(* IEC 61131-3 sources: SIMERLIFT/LOGICAD/SIMERLIFT/src_FBD/BCU/fbdBCU_bess, 5 files *)

(* ---- Balance_isz.iecfbd ---- *)
FUNCTION_BLOCK Balance_isz
  {
    Charge_Status {index := 0};
    Avarage_Cell_Voltage {index := 3};
    Balance_Threshold {index := 4};
    Difference_Tolerance {index := 5};
    Ballance_Interval {index := 6};
    Min_Cell_Voltage {index := 2};
    Max_Cell_Voltage {index := 1};
    Measure_Aux {index := 3};
    Measure_All {index := 2};
    width := 460;
    height := 138;
  }

  VAR
    RS3 : RS;
    TP3 : TP;
    TON4 : TON;
    R_TRIG5 : R_TRIG;
    Meas_Period : TIME := T#48ms;
    Ballance_Pending : BOOL := 0;
    maxVolt : UDINT;
    minVolt : UDINT;
    FLASH1 : FLASH;
    FLASH2 : FLASH;
  END_VAR
  VAR_INPUT
    Max_Cell_Voltage : UDINT := 0;
    Min_Cell_Voltage : UDINT := 0;
    Avarage_Cell_Voltage : UDINT := 0;
    Charge_Status : BOOL := 0;
    Ballance_Interval : TIME := T#30s;
    Difference_Tolerance : UDINT := 0;
    Balance_Threshold : UDINT := 0;
  END_VAR
  VAR_OUTPUT
    Balance_Enable : BOOL := 0;
    Measure_All : BOOL := 0;
    Measure_Aux : BOOL := 0;
    Ballance_Voltage : UDINT := 0;
  END_VAR

  (*

    // Network 1:
    ADD(IN1 := Avarage_Cell_Voltage, IN2 := 1, ADD => @C(4).ADD);
    GE(IN1 := @C(4).ADD, IN2 := Balance_Threshold, GE => @C(29).GE);
    SEL(G := @C(29).GE, IN0 := Balance_Threshold, IN1 := @C(4).ADD, SEL => Ballance_Voltage);

    // Network 2:
    GE(IN1 := Max_Cell_Voltage, IN2 := Balance_Threshold, GE => @C(41).GE);
    SUB(IN1 := Max_Cell_Voltage, IN2 := Min_Cell_Voltage, SUB => @C(20).SUB);
    GT(IN1 := @C(20).SUB, IN2 := Difference_Tolerance, GT => @C(45).GT);
    AND(IN1 := @C(41).GE, IN2 := @C(45).GT, AND => Ballance_Pending);

    // Network 3:
    MUL_TIME(IN1 := Meas_Period, IN2 := 20, MUL_TIME => @C(50).MUL_TIME);
    ADD(IN1 := @C(50).MUL_TIME, IN2 := Ballance_Interval, ADD => @C(54).ADD);
    TP3(IN := RS3.Q1, PT := Ballance_Interval);
    AND(IN1 := Charge_Status, IN2 := TP3.Q, AND => (@C(11).AND, Balance_Enable));
    FLASH1(IN := NOT @C(11).AND, PER := Meas_Period, OUT => Measure_All);
    TON4(IN := RS3.Q1, PT := @C(54).ADD);
    R_TRIG5(CLK := TON4.Q);
    RS3(S := Ballance_Pending, R1 := R_TRIG5.Q);
    FLASH2(IN := @C(11).AND, PER := T#1s, OUT => Measure_Aux);

  *)

  @C(4) : @F(ADD), @R(280.0, 20.0, 40.0, 38.0), UDINT, @I(@N(IN1), @L(9.5)), @I(@N(IN2), @L(29.5)), @O(@N(ADD), @R(9.5));
  @C(8) : @F(AND), @R(520.0, 120.0, 40.0, 38.0), BOOL, @I(@N(IN1), @L(9.5)), @I(@N(IN2), @L(29.5)), @O(@N(AND), @R(9.5));
  @C(11) : @F(AND), @R(1140.0, 250.0, 40.0, 38.0), BOOL, @I(@N(IN1), @L(9.5)), @I(@N(IN2), @L(29.5)), @O(@N(AND), @R(9.5));
  @C(20) : @F(SUB), @R(280.0, 160.0, 40.0, 38.0), UDINT, @I(@N(IN1), @L(9.5)), @I(@N(IN2), @L(29.5)), @O(@N(SUB), @R(9.5));
  @C(25) : @FB(RS3), @R(800.0, 290.0, 80.0, 38.0), @I(@N(S), @L(9.5)), @I(@N(R1), @L(29.5)), @O(@N(Q1), @R(9.5));
  @C(24) : @FB(TP3), @R(960.0, 290.0, 100.0, 38.0), @I(@N(IN), @L(9.5)), @I(@N(PT), @L(29.5)), @O(@N(Q), @R(9.5)), @O(@N(ET), @R(29.5));
  @C(27) : @FB(TON4), @R(480.0, 310.0, 100.0, 38.0), @I(@N(IN), @L(9.5)), @I(@N(PT), @L(29.5)), @O(@N(Q), @R(9.5)), @O(@N(ET), @R(29.5));
  @C(26) : @FB(R_TRIG5), @R(620.0, 310.0, 140.0, 18.0), @I(@N(CLK), @L(9.5)), @O(@N(Q), @R(9.5));
  @C(29) : @F(GE), @R(440.0, 20.0, 40.0, 38.0), UDINT, @I(@N(IN1), @L(9.5)), @I(@N(IN2), @L(29.5)), @O(@N(GE), @R(9.5));
  @C(33) : @F(SEL), @R(560.0, 40.0, 120.0, 58.0), UDINT, @I(@N(G), @L(9.5)), @I(@N(IN0), @L(29.5)), @I(@N(IN1), @L(49.5)), @O(@N(SEL), @R(9.5));
  @C(41) : @F(GE), @R(400.0, 120.0, 40.0, 38.0), UDINT, @I(@N(IN1), @L(9.5)), @I(@N(IN2), @L(29.5)), @O(@N(GE), @R(9.5));
  @C(45) : @F(GT), @R(400.0, 160.0, 40.0, 38.0), UDINT, @I(@N(IN1), @L(9.5)), @I(@N(IN2), @L(29.5)), @O(@N(GT), @R(9.5));
  @C(50) : @F(MUL_TIME), @R(280.0, 330.0, 40.0, 38.0), USINT, @I(@N(IN1), @L(9.5)), @I(@N(IN2), @L(29.5)), @O(@N(MUL_TIME), @R(9.5));
  @C(54) : @F(ADD), @R(400.0, 330.0, 40.0, 38.0), TIME, @I(@N(IN1), @L(9.5)), @I(@N(IN2), @L(29.5)), @O(@N(ADD), @R(9.5));
  @VF(69) : @E(Meas_Period), @R(1340.0, 320.0, 110.0, 19.0);
  @VF(3) : @E(Avarage_Cell_Voltage), @R(20.0, 20.0, 180.0, 19.0);
  @VF(6) : @E(1), @R(110.0, 40.0, 90.0, 19.0), UDINT;
  @VF(7) : @E(Balance_Enable), @R(1640.0, 250.0, 180.0, 19.0);
  @VF(10) : @E(Charge_Status), @R(20.0, 250.0, 180.0, 19.0);
  @VF(78) : @E(Ballance_Interval), @R(20.0, 370.0, 180.0, 19.0);
  @VF(72) : @E(Measure_All), @R(1650.0, 300.0, 180.0, 19.0);
  @VF(18) : @E(Difference_Tolerance), @R(20.0, 200.0, 180.0, 19.0);
  @VF(31) : @E(Balance_Threshold), @R(20.0, 60.0, 180.0, 19.0);
  @VF(239) : @E(Meas_Period), @R(20.0, 330.0, 180.0, 19.0);
  @VF(37) : @E(Ballance_Voltage), @R(750.0, 40.0, 180.0, 19.0);
  @VF(42) : @E(Balance_Threshold), @R(20.0, 140.0, 180.0, 19.0);
  @VF(48) : @E(Ballance_Pending), @R(750.0, 120.0, 180.0, 19.0);
  @VF(52) : @E(20), @R(110.0, 350.0, 90.0, 19.0), USINT;
  @VF(58) : @E(Ballance_Pending), @R(20.0, 290.0, 180.0, 19.0);
  @C(23) : @FB(FLASH1), @R(1480.0, 300.0, 120.0, 38.0), @I(@N(IN), @L(9.5), @NEG), @I(@N(PER), @L(29.5)), @O(@N(OUT), @R(9.5));
  @VF(74) : @E(Max_Cell_Voltage), @R(30.0, 160.0, 160.0, 19.0);
  @VF(83) : @E(Min_Cell_Voltage), @R(30.0, 180.0, 160.0, 19.0);
  @C(14) : @FB(FLASH2), @R(1480.0, 340.0, 120.0, 38.0), @I(@N(IN), @L(9.5)), @I(@N(PER), @L(29.5)), @O(@N(OUT), @R(9.5));
  @VF(15) : @E(T#1s), @R(1340.0, 360.0, 110.0, 19.0);
  @VF(16) : @E(Measure_Aux), @R(1650.0, 340.0, 180.0, 19.0);
  @CP(35) : 399.5, 69.5;
  @CP(36) : 359.5, 29.5;
  @CP(44) : 239.5, 169.5;
  @CP(64) : 359.5, 379.5;
  @CP(66) : 919.5, 299.5;
  @CP(2) : 1289.5, 259.5;

  @G(13) :
     @L(@C(11).AND, @CP(2)),
     @L(@CP(2), @VF(7).i),
     @L(@CP(2), @C(23).IN),
     @L(@CP(2), @C(14).IN)
    ;
  @G(5) :
     @L(@VF(3).o, @C(4).IN1)
    ;
  @G(28) :
     @L(@VF(6).o, @C(4).IN2)
    ;
  @G(30) :
     @L(@C(4).ADD, @CP(36)),
     @L(@CP(36), @C(29).IN1),
     @L(@CP(36), @C(33).IN1)
    ;
  @G(32) :
     @L(@VF(31).o, @CP(35)),
     @L(@CP(35), @C(29).IN2),
     @L(@CP(35), @C(33).IN0)
    ;
  @G(34) :
     @L(@C(29).GE, @C(33).G)
    ;
  @G(38) :
     @L(@C(33).SEL, @VF(37).i)
    ;
  @G(39) :
     @L(@CP(44), @C(20).IN1),
     @L(@CP(44), @C(41).IN1),
     @L(@VF(74).o, @CP(44))
    ;
  @G(46) :
     @L(@C(20).SUB, @C(45).IN1)
    ;
  @G(19) :
     @L(@VF(18).o, @C(45).IN2)
    ;
  @G(49) :
     @L(@C(8).AND, @VF(48).i)
    ;
  @G(51) :
     @L(@VF(239).o, @C(50).IN1)
    ;
  @G(53) :
     @L(@VF(52).o, @C(50).IN2)
    ;
  @G(56) :
     @L(@CP(64), @C(54).IN2),
     @L(@CP(64), @C(24).PT),
     @L(@VF(78).o, @CP(64))
    ;
  @G(57) :
     @L(@C(50).MUL_TIME, @C(54).IN1)
    ;
  @G(59) :
     @L(@VF(58).o, @C(25).S)
    ;
  @G(60) :
     @L(@C(26).Q, @C(25).R1)
    ;
  @G(61) :
     @L(@C(54).ADD, @C(27).PT)
    ;
  @G(62) :
     @L(@C(27).Q, @C(26).CLK)
    ;
  @G(63) :
     @L(@C(25).Q1, @CP(66)),
     @L(@CP(66), @C(24).IN),
     @L(@CP(66), @C(27).IN)
    ;
  @G(65) :
     @L(@C(24).Q, @C(11).IN2)
    ;
  @G(9) :
     @L(@C(41).GE, @C(8).IN1)
    ;
  @G(21) :
     @L(@C(45).GT, @C(8).IN2)
    ;
  @G(22) :
     @L(@VF(42).o, @C(41).IN2)
    ;
  @G(12) :
     @L(@VF(10).o, @C(11).IN1)
    ;
  @G(43) :
     @L(@VF(69).o, @C(23).PER)
    ;
  @G(75) :
     @L(@C(23).OUT, @VF(72).i)
    ;
  @G(1) :
     @L(@VF(83).o, @C(20).IN2)
    ;
  @G(17) :
     @L(@VF(15).o, @C(14).PER)
    ;
  @G(40) :
     @L(@C(14).OUT, @VF(16).i)
    ;
END_FUNCTION_BLOCK

(* ---- CurrentLimiter_ISZ.iecfbd ---- *)
FUNCTION_BLOCK CurrentLimiter_ISZ
  {
    width := 370;
  }

  VAR
    OverCurrent30sec : BOOL;
    OverCurrent10sec : BOOL;
    OverCurrentCont : BOOL;
    CounTimR1 : CounTimR;
    deratingToCont : BOOL;
    maxCurrent : INT;
    RS2 : RS;
    exceed30s : BOOL;
    SR1 : SR;
    FLASH5 : FLASH;
    FLASH6 : FLASH;
    CTUD2 : CTUD;
  END_VAR
  VAR_INPUT
    Lim30s : INT;
    LimCont : INT;
    Current : INT;
  END_VAR
  VAR_OUTPUT
    overCurrent : BOOL;
    Lim : INT;
  END_VAR

  (*

    // Network 1:
    GT(IN1 := Current, IN2 := Lim30s, GT => OverCurrent30sec);
    GT(IN1 := Current, IN2 := LimCont, GT => OverCurrentCont);

    // Network 2:
    CounTimR1(CU := OverCurrentCont, ACCper := T#500ms, DECper := T#2s, CD := NOT OverCurrentCont, PV := 25, QU => exceed30s);
    GE(IN1 := CounTimR1.CV, IN2 := 30, GE => @C(18).GE);
    SR1(S1 := @C(18).GE, R := CounTimR1.QD, Q1 => deratingToCont);

    // Network 3:
    SEL(G := deratingToCont, IN0 := Lim30s, IN1 := LimCont, SEL => maxCurrent);

    // Network 4:
    RS2(S := exceed30s, R1 := NOT OverCurrentCont);
    OR(IN1 := OverCurrent30sec, IN2 := RS2.Q1, OR => OverCurrent);

    // Network 5:
    TO_INT(IN := maxCurrent, TO_INT => @C(173).TO_INT);
    GT(IN1 := maxCurrent, IN2 := Lim, GT => @C(95).GT);
    FLASH5(IN := @C(95).GT, PER := T#5ms);
    LT(IN1 := maxCurrent, IN2 := Lim, LT => @C(98).LT);
    FLASH6(IN := @C(98).LT, PER := T#5ms);
    CTUD2(CU := FLASH5.OUT, CD := FLASH6.OUT, PV := @C(173).TO_INT, CV => Lim);

  *)

  @VF(1) : @E(Lim30s), @R(150.0, 80.0, 140.0, 19.0);
  @VF(2) : @E(LimCont), @R(150.0, 120.0, 140.0, 19.0);
  @VF(4) : @E(Current), @R(150.0, 60.0, 140.0, 19.0);
  @C(19) : @F(GT), @R(400.0, 60.0, 40.0, 38.0), INT, @I(@N(IN1), @L(9.5)), @I(@N(IN2), @L(29.5)), @O(@N(GT), @R(9.5));
  @C(20) : @F(GT), @R(400.0, 100.0, 40.0, 38.0), INT, @I(@N(IN1), @L(9.5)), @I(@N(IN2), @L(29.5)), @O(@N(GT), @R(9.5));
  @VF(28) : @E(OverCurrent30sec), @R(520.0, 60.0, 180.0, 19.0);
  @VF(32) : @E(OverCurrentCont), @R(520.0, 100.0, 180.0, 19.0);
  @C(8) : @FB(CounTimR1), @R(600.0, 250.0, 250.0, 118.0), @I(@N(CU), @L(9.5)), @I(@N(ACCper), @L(49.5)), @I(@N(DECper), @L(69.5)), @I(@N(CD), @L(29.5), @NEG), @I(@N(PV), @L(89.5)), @I(@N(R), @L(109.5)), @O(@N(CV), @R(9.5)), @O(@N(QD), @R(29.5)), @O(@N(QU), @R(49.5));
  @VF(9) : @E(OverCurrentCont), @R(340.0, 250.0, 180.0, 19.0);
  @VF(11) : @E(T#500ms), @R(490.0, 290.0, 80.0, 19.0);
  @VF(14) : @E(T#2s), @R(490.0, 310.0, 80.0, 19.0);
  @VF(16) : @E(25), @R(490.0, 330.0, 80.0, 19.0), INT;
  @C(18) : @F(GE), @R(1090.0, 250.0, 40.0, 38.0), INT, @I(@N(IN1), @L(9.5)), @I(@N(IN2), @L(29.5)), @O(@N(GE), @R(9.5));
  @VF(22) : @E(30), @R(1010.0, 270.0, 60.0, 19.0), INT;
  @VF(124) : @E(deratingToCont), @R(1290.0, 250.0, 140.0, 19.0);
  @C(79) : @F(SEL), @R(670.0, 420.0, 120.0, 58.0), INT, @I(@N(G), @L(9.5)), @I(@N(IN0), @L(29.5)), @I(@N(IN1), @L(49.5)), @O(@N(SEL), @R(9.5));
  @VF(25) : @E(deratingToCont), @R(470.0, 420.0, 140.0, 19.0);
  @VF(109) : @E(LimCont), @R(500.0, 460.0, 140.0, 19.0);
  @VF(76) : @E(maxCurrent), @R(830.0, 420.0, 140.0, 19.0);
  @VF(26) : @E(Lim30s), @R(500.0, 440.0, 140.0, 19.0);
  @C(84) : @FB(RS2), @R(1350.0, 480.0, 80.0, 38.0), @I(@N(S), @L(9.5)), @I(@N(R1), @L(29.5)), @O(@N(Q1), @R(9.5));
  @VF(29) : @E(OverCurrent), @R(1540.0, 460.0, 140.0, 19.0);
  @VF(30) : @E(exceed30s), @R(1170.0, 480.0, 140.0, 19.0);
  @VF(89) : @E(OverCurrentCont), @R(1130.0, 500.0, 180.0, 19.0), @ONEG;
  @C(31) : @F(OR), @R(1460.0, 460.0, 40.0, 38.0), BOOL, @I(@N(IN1), @L(9.5)), @I(@N(IN2), @L(29.5)), @O(@N(OR), @R(9.5));
  @VF(34) : @E(OverCurrent30sec), @R(1130.0, 460.0, 180.0, 19.0);
  @C(24) : @FB(SR1), @R(1180.0, 250.0, 80.0, 38.0), @I(@N(S1), @L(9.5)), @I(@N(R), @L(29.5)), @O(@N(Q1), @R(9.5));
  @C(95) : @F(GT), @R(550.0, 570.0, 40.0, 38.0), INT, @I(@N(IN1), @L(9.5)), @I(@N(IN2), @L(29.5)), @O(@N(GT), @R(9.5));
  @C(98) : @F(LT), @R(550.0, 610.0, 40.0, 38.0), INT, @I(@N(IN1), @L(9.5)), @I(@N(IN2), @L(29.5)), @O(@N(LT), @R(9.5));
  @C(101) : @FB(FLASH5), @R(770.0, 570.0, 120.0, 38.0), @I(@N(IN), @L(9.5)), @I(@N(PER), @L(29.5)), @O(@N(OUT), @R(9.5));
  @C(125) : @FB(FLASH6), @R(770.0, 610.0, 120.0, 38.0), @I(@N(IN), @L(9.5)), @I(@N(PER), @L(29.5)), @O(@N(OUT), @R(9.5));
  @C(173) : @F(TO_INT), @R(770.0, 650.0, 120.0, 18.0), INT, @I(@N(IN), @L(9.5)), @O(@N(TO_INT), @R(9.5));
  @C(1467) : @FB(CTUD2), @R(960.0, 570.0, 100.0, 98.0), @I(@N(CU), @L(9.5)), @I(@N(CD), @L(29.5)), @I(@N(R), @L(49.5)), @I(@N(LD), @L(69.5)), @I(@N(PV), @L(89.5)), @O(@N(QU), @R(9.5)), @O(@N(QD), @R(29.5)), @O(@N(CV), @R(89.5));
  @VF(94) : @E(maxCurrent), @R(320.0, 570.0, 140.0, 19.0);
  @VF(93) : @E(Lim), @R(320.0, 590.0, 140.0, 19.0);
  @VF(178) : @E(T#5ms), @R(600.0, 590.0, 90.0, 19.0);
  @VF(176) : @E(Lim), @R(1140.0, 650.0, 140.0, 19.0);
  @VF(40) : @E(exceed30s), @R(990.0, 300.0, 140.0, 19.0);
  @CP(7) : 369.5, 69.5;
  @CP(13) : 559.5, 259.5;
  @CP(100) : 499.5, 599.5;
  @CP(99) : 529.5, 579.5;
  @CP(172) : 529.5, 619.5;
  @CP(180) : 709.5, 599.5;

  @G(54) :
     @L(@C(19).GT, @VF(28).i)
    ;
  @G(56) :
     @L(@C(20).GT, @VF(32).i)
    ;
  @G(3) :
     @L(@VF(4).o, @CP(7)),
     @L(@CP(7), @C(19).IN1),
     @L(@CP(7), @C(20).IN1)
    ;
  @G(5) :
     @L(@VF(1).o, @C(19).IN2)
    ;
  @G(6) :
     @L(@VF(2).o, @C(20).IN2)
    ;
  @G(10) :
     @L(@VF(9).o, @CP(13)),
     @L(@CP(13), @C(8).CU),
     @L(@CP(13), @C(8).CD)
    ;
  @G(12) :
     @L(@VF(11).o, @C(8).ACCper)
    ;
  @G(15) :
     @L(@VF(14).o, @C(8).DECper)
    ;
  @G(17) :
     @L(@VF(16).o, @C(8).PV)
    ;
  @G(21) :
     @L(@C(8).CV, @C(18).IN1)
    ;
  @G(23) :
     @L(@VF(22).o, @C(18).IN2)
    ;
  @G(83) :
     @L(@VF(25).o, @C(79).G)
    ;
  @G(80) :
     @L(@C(79).SEL, @VF(76).i)
    ;
  @G(110) :
     @L(@VF(109).o, @C(79).IN1)
    ;
  @G(27) :
     @L(@VF(26).o, @C(79).IN0)
    ;
  @G(88) :
     @L(@VF(30).o, @C(84).S)
    ;
  @G(90) :
     @L(@VF(89).o, @C(84).R1)
    ;
  @G(33) :
     @L(@C(84).Q1, @C(31).IN2)
    ;
  @G(35) :
     @L(@VF(34).o, @C(31).IN1)
    ;
  @G(36) :
     @L(@C(31).OR, @VF(29).i)
    ;
  @G(37) :
     @L(@C(18).GE, @C(24).S1)
    ;
  @G(38) :
     @L(@C(24).Q1, @VF(124).i)
    ;
  @G(39) :
     @L(@C(8).QD, @C(24).R)
    ;
  @G(97) :
     @L(@VF(93).o, @CP(100)),
     @L(@CP(100), @C(95).IN2),
     @L(@CP(100), @C(98).IN2)
    ;
  @G(96) :
     @L(@CP(99), @C(95).IN1),
     @L(@CP(99), @CP(172)),
     @L(@CP(172), @C(98).IN1),
     @L(@CP(172), @C(173).IN),
     @L(@VF(94).o, @CP(99))
    ;
  @G(179) :
     @L(@VF(178).o, @CP(180)),
     @L(@CP(180), @C(101).PER),
     @L(@CP(180), @C(125).PER)
    ;
  @G(102) :
     @L(@C(95).GT, @C(101).IN)
    ;
  @G(170) :
     @L(@C(98).LT, @C(125).IN)
    ;
  @G(123) :
     @L(@C(101).OUT, @C(1467).CU)
    ;
  @G(171) :
     @L(@C(125).OUT, @C(1467).CD)
    ;
  @G(174) :
     @L(@C(173).TO_INT, @C(1467).PV)
    ;
  @G(177) :
     @L(@C(1467).CV, @VF(176).i)
    ;
  @G(41) :
     @L(@C(8).QU, @VF(40).i)
    ;
END_FUNCTION_BLOCK

(* ---- essBattState.iecst ---- *)
FUNCTION_BLOCK  essBattState  {
    width := 400;
    bgColor := "mediumseagreen";
  }

VAR_INPUT
	IGNITION : BOOL;
	chargerON:BOOL;
	prechargeOk:BOOL;
	dischargeComplete:BOOL;
	chargeComplete:BOOL;
	shutdownComplete:BOOL;
	contactFbk:BOOL;
	currentAmp:REAL;
	outVoltStatus:BOOL;
	OVfault:BOOL;
    UVfault:BOOL;
	fault:BOOL;
END_VAR

VAR_OUTPUT
	STATE : BATTSTATE;
	prechargeOn:BOOL;
	contact:BOOL;
	contactNeg:BOOL;
END_VAR

VAR
currentCharging:BOOL;
currentDischarging:BOOL;

CURRENTTIMERcharging:TON;
CURRENTTIMERdischarging:TON;

chargeVoltTimer:Tbuffer;
dischargeVoltTimer:Tbuffer;

BATTERYSTATE:BATTSTATE:=BATTSTATE#STANDBY;
PREVSTATE:BATTSTATE:=BATTSTATE#STANDBY;

BATTIMER:TON;
BATSTATEINTERVAL:TIME:=T#10s;
BATSTATETIMEOUT:BOOL;
BATSTATEELAPSEDTIME:TIME;
STANDBYINTERVAL:TIME:=T#2s;
END_VAR

CURRENTTIMERcharging(IN:=currentAmp<-0.5, PT:=T#500ms, Q=>currentCharging);
CURRENTTIMERdischarging(IN:=currentAmp>0.5, PT:=T#500ms, Q=>currentDischarging);
BATTIMER(IN:=BATTERYSTATE=PREVSTATE, PT:=BATSTATEINTERVAL, Q=>BATSTATETIMEOUT, ET=>BATSTATEELAPSEDTIME);

PREVSTATE:=BATTERYSTATE;

CASE BATTERYSTATE OF

	BATTSTATE#STANDBY:  // standby
		STATE:=BATTSTATE#STANDBY;
		BATSTATEINTERVAL:=T#12s;

		prechargeOn:=0;
		contact:=0;
		contactNeg:=0;

		// at the first time wait 2 sec
		IF BATSTATEELAPSEDTIME>STANDBYINTERVAL THEN
		    // then wait 100ms in next sessions
			STANDBYINTERVAL:=T#500ms;
			IF fault THEN
				BATTERYSTATE:=BATTSTATE#FAULT;
			ELSIF IGNITION THEN
				IF chargerON THEN
					IF OVfault OR chargeComplete THEN
						BATTERYSTATE:=BATTSTATE#CHARGECOMPLETE;
					ELSE
						BATTERYSTATE:=BATTSTATE#PRECHARGE;
					END_IF;
				ELSE
					BATTERYSTATE:=BATTSTATE#PRECHARGE;
				END_IF;
			END_IF;

		END_IF;

	BATTSTATE#PRECHARGE:  //discharge
		STATE:=BATTSTATE#PRECHARGE;
		BATSTATEINTERVAL:=T#5s;

		contactNeg:=1;

		IF BATSTATEELAPSEDTIME>T#50ms THEN
			prechargeOn:=1;
		ELSE
			prechargeOn:=0;
		END_IF;

		IF prechargeOk THEN
			contact:=1;
		ELSE
			contact:=0;
		END_IF;

		IF fault OR  NOT IGNITION  THEN
			BATTERYSTATE:=BATTSTATE#SHUTDOWN;
		ELSIF BATSTATETIMEOUT THEN
			BATTERYSTATE:=BATTSTATE#FAULT;
		ELSIF prechargeOk=TRUE AND contactFbk=TRUE THEN
			IF chargerON THEN
				IF OVfault OR chargeComplete THEN
					BATTERYSTATE:=BATTSTATE#CHARGECOMPLETE;
				ELSE
					BATTERYSTATE:=BATTSTATE#CHARGE;
				END_IF;
			ELSE
				BATTERYSTATE:=BATTSTATE#DISCHARGE;
			END_IF;
		END_IF;

	BATTSTATE#DISCHARGE:  //discharge
		STATE:=BATTSTATE#DISCHARGE;
		BATSTATEINTERVAL:=T#120s;

		prechargeOn:=0;
		contact:=1;
		contactNeg:=1;

		IF fault THEN
			BATTERYSTATE:=BATTSTATE#SHUTDOWN;
		ELSIF NOT IGNITION THEN
			BATTERYSTATE:=BATTSTATE#SHUTDOWN;
		ELSIF chargerON THEN
			IF OVfault OR chargeComplete THEN
				BATTERYSTATE:=BATTSTATE#CHARGECOMPLETE;
			ELSE
				BATTERYSTATE:=BATTSTATE#CHARGE;
			END_IF;
		ELSIF BATSTATEELAPSEDTIME>T#10s THEN
			IF currentDischarging THEN
				IF UVfault OR dischargeComplete THEN
					BATTERYSTATE:=BATTSTATE#DISCHARGECOMPLETE;
				END_IF;
			ELSIF currentCharging THEN
				IF OVfault THEN
					BATTERYSTATE:=BATTSTATE#CHARGECOMPLETE;
				END_IF;
			END_IF;
		ELSIF (UVfault OR dischargeComplete) AND currentAmp>10 THEN
			BATTERYSTATE:=BATTSTATE#DISCHARGECOMPLETE;
		ELSIF (OVfault OR chargeComplete) AND currentAmp<-10 THEN
			BATTERYSTATE:=BATTSTATE#CHARGECOMPLETE;
		END_IF;

	BATTSTATE#CHARGE:  // charge
		STATE:=BATTSTATE#CHARGE;
		BATSTATEINTERVAL:=T#120s;

		prechargeOn:=0;
		contact:=1;
		contactNeg:=1;

		IF fault THEN
			BATTERYSTATE:=BATTSTATE#SHUTDOWN;
		ELSIF NOT IGNITION THEN
			BATTERYSTATE:=BATTSTATE#SHUTDOWN;
		ELSIF NOT chargerON THEN
			IF UVfault THEN
				BATTERYSTATE:=BATTSTATE#DISCHARGECOMPLETE;
			ELSIF dischargeComplete THEN
				BATTERYSTATE:=BATTSTATE#DISCHARGECOMPLETE;
			ELSE
				BATTERYSTATE:=BATTSTATE#DISCHARGE;
			END_IF;
		ELSIF OVfault OR chargeComplete THEN
			BATTERYSTATE:=BATTSTATE#CHARGECOMPLETE;
		ELSIF  BATSTATEELAPSEDTIME>T#8s THEN
			IF currentDischarging THEN
				IF UVfault THEN
					BATTERYSTATE:=BATTSTATE#DISCHARGECOMPLETE;
				ELSIF dischargeComplete THEN
					BATTERYSTATE:=BATTSTATE#DISCHARGECOMPLETE;
				END_IF;
			END_IF;
		ELSIF (UVfault OR dischargeComplete) AND currentAmp>10THEN
			BATTERYSTATE:=BATTSTATE#DISCHARGECOMPLETE;
		END_IF;

	BATTSTATE#SHUTDOWN:  // shutdown
		STATE:=BATTSTATE#SHUTDOWN;
		BATSTATEINTERVAL:=T#3000ms;
		prechargeOn:=0;
		IF BATSTATETIMEOUT OR  (shutdownComplete AND (BATSTATEELAPSEDTIME>T#1000ms))  THEN
			contact:=0;
		 	contactNeg:=0;
		 	IF contactFbk=FALSE THEN
				IF fault THEN
					BATTERYSTATE:=BATTSTATE#FAULT;
				ELSIF UVfault THEN
					BATTERYSTATE:=BATTSTATE#DISCHARGECOMPLETE;
				ELSIF OVfault THEN
					BATTERYSTATE:=BATTSTATE#CHARGECOMPLETE;
				ELSIF NOT IGNITION THEN
					BATTERYSTATE:=BATTSTATE#STANDBY;
				END_IF;
			ELSIF BATSTATEELAPSEDTIME>T#2500ms THEN
				BATTERYSTATE:=BATTSTATE#FAULT;
			END_IF;

		END_IF;

	BATTSTATE#FAULT:  //fault
		STATE:=BATTSTATE#FAULT;
		BATSTATEINTERVAL:=T#10s;

		prechargeOn:=0;
		contact:=0;
		contactNeg:=0;

		IF NOT fault AND (NOT IGNITION OR BATSTATETIMEOUT) THEN
			BATTERYSTATE:=BATTSTATE#STANDBY;
		END_IF;

	BATTSTATE#CHARGECOMPLETE:  //charge complete
		STATE:=BATTSTATE#CHARGECOMPLETE;
		BATSTATEINTERVAL:=T#5s;

		prechargeOn:=0;
		contact:=0;
		contactNeg:=0;

		IF fault THEN
			BATTERYSTATE:=BATTSTATE#SHUTDOWN;
		ELSIF NOT IGNITION THEN
			BATTERYSTATE:=BATTSTATE#SHUTDOWN;
		ELSIF NOT outVoltStatus AND BATSTATETIMEOUT THEN
			IF UVfault THEN
				BATTERYSTATE:=BATTSTATE#DISCHARGECOMPLETE;
			ELSIF dischargeComplete THEN
				BATTERYSTATE:=BATTSTATE#DISCHARGECOMPLETE;
			ELSE
				BATTERYSTATE:=BATTSTATE#PRECHARGE;
			END_IF;
		END_IF;

	BATTSTATE#DISCHARGECOMPLETE:  //charge complete
		STATE:=BATTSTATE#DISCHARGECOMPLETE;
		BATSTATEINTERVAL:=T#5s;

		prechargeOn:=0;
		contact:=0;
		contactNeg:=0;

		IF fault THEN
			BATTERYSTATE:=BATTSTATE#SHUTDOWN;
		ELSIF NOT IGNITION THEN
			BATTERYSTATE:=BATTSTATE#SHUTDOWN;
		ELSIF outVoltStatus AND BATSTATETIMEOUT THEN
			IF OVfault THEN
				BATTERYSTATE:=BATTSTATE#CHARGECOMPLETE;
			ELSIF chargeComplete THEN
				BATTERYSTATE:=BATTSTATE#CHARGECOMPLETE;
			ELSE
				BATTERYSTATE:=BATTSTATE#PRECHARGE;   /// because no current will flow unless contact closed
			END_IF;
		END_IF;

END_CASE;

END_FUNCTION_BLOCK

(* ---- SOCisz.iecfbd ---- *)
FUNCTION_BLOCK SOCisz
  {
    width := 340;
  }

  VAR
    socState1 : socState;
    RMEM_REAL1 : RMEM_REAL;
    memReadWh : REAL;
    fMemW_REAL1 : fMemW_REAL;
  END_VAR
  VAR_INPUT
    capacityWh : REAL;
    instantWh : REAL;
    chargeCompleted : BOOL;
    memoryWrite : BOOL;
  END_VAR
  VAR_OUTPUT
    SOC : REAL;
    remainingWh : REAL;
    state : USINT;
  END_VAR

  (*

    // Network 1:
    socState1(whCap := capacityWh, whInstant := instantWh, whMem := memReadWh, chargeComplete := chargeCompleted, memWr := memoryWrite, SOC => SOC, whRem => remainingWh, socState => state);
    fMemW_REAL1(ADDR := 16#100, VAL := socState1.whRem, R := socState1.wrWh);
    RMEM_REAL1(ADDR := 16#100, R := socState1.rdWh, VAL => memReadWh);

  *)

  @VF(3) : @E(16#100), @R(1000.0, 180.0, 80.0, 19.0), UDINT;
  @C(2) : @FB(RMEM_REAL1), @R(1120.0, 240.0, 210.0, 38.0), @I(@N(ADDR), @L(9.5)), @I(@N(R), @L(29.5)), @O(@N(VAL), @R(9.5)), @O(@N(NXT), @R(29.5));
  @VF(6) : @E(memReadWh), @R(1370.0, 240.0, 140.0, 19.0);
  @VF(8) : @E(memReadWh), @R(180.0, 220.0, 140.0, 19.0);
  @VF(10) : @E(capacityWh), @R(180.0, 180.0, 140.0, 19.0);
  @VF(12) : @E(instantWh), @R(180.0, 200.0, 140.0, 19.0);
  @VF(14) : @E(chargeCompleted), @R(180.0, 240.0, 140.0, 19.0);
  @VF(16) : @E(memoryWrite), @R(180.0, 260.0, 140.0, 19.0);
  @C(18) : @FB(fMemW_REAL1), @R(1120.0, 180.0, 250.0, 58.0), @I(@N(ADDR), @L(9.5)), @I(@N(VAL), @L(29.5)), @I(@N(R), @L(49.5)), @O(@N(OK), @R(9.5)), @O(@N(RET), @R(29.5)), @O(@N(NXT), @R(49.5));
  @VF(22) : @E(SOC), @R(780.0, 180.0, 140.0, 19.0);
  @VF(24) : @E(remainingWh), @R(1210.0, 310.0, 140.0, 19.0);
  @C(1) : @FB(socState1), @R(360.0, 180.0, 400.0, 98.0), @I(@N(whCap), @L(9.5)), @I(@N(whInstant), @L(29.5)), @I(@N(whMem), @L(49.5)), @I(@N(chargeComplete), @L(69.5)), @I(@N(memWr), @L(89.5)), @O(@N(SOC), @R(9.5)), @O(@N(whRem), @R(29.5)), @O(@N(wrWh), @R(49.5)), @O(@N(rdWh), @R(69.5)), @O(@N(socState), @R(89.5));
  @VF(26) : @E(state), @R(780.0, 260.0, 140.0, 19.0);
  @CP(21) : 1099.5, 189.5;
  @CP(25) : 969.5, 209.5;

  @G(4) :
     @L(@C(1).rdWh, @C(2).R)
    ;
  @G(7) :
     @L(@C(2).VAL, @VF(6).i)
    ;
  @G(9) :
     @L(@VF(8).o, @C(1).whMem)
    ;
  @G(11) :
     @L(@VF(10).o, @C(1).whCap)
    ;
  @G(13) :
     @L(@VF(12).o, @C(1).whInstant)
    ;
  @G(15) :
     @L(@VF(14).o, @C(1).chargeComplete)
    ;
  @G(17) :
     @L(@VF(16).o, @C(1).memWr)
    ;
  @G(19) :
     @L(@C(1).wrWh, @C(18).R)
    ;
  @G(20) :
     @L(@C(1).whRem, @CP(25)),
     @L(@CP(25), @C(18).VAL),
     @L(@CP(25), @VF(24).i)
    ;
  @G(5) :
     @L(@VF(3).o, @CP(21)),
     @L(@CP(21), @C(18).ADDR),
     @L(@CP(21), @C(2).ADDR)
    ;
  @G(23) :
     @L(@C(1).SOC, @VF(22).i)
    ;
  @G(27) :
     @L(@C(1).socState, @VF(26).i)
    ;
END_FUNCTION_BLOCK

(* ---- HemaBattery.iecfbd ---- *)
PROGRAM HemaBattery
  VAR
    BATTSTACK1 : BATTSTACK;
    GUICFG_INT3 : GUICFG_INT;
    numOfCells1 : numOfCells;
    IOWR2 : IOWR;
    IOWR1 : IOWR;
    Max_Min_Voltage_Status1 : Max_Min_Voltage_Status;
    chargeState1 : chargeState;
    SOCisz1 : SOCisz;
    TON6 : TON;
    GUI1 : GUI;
    TON7 : TON;
    TOF12 : TOF;
    TOF13 : TOF;
    TOF14 : TOF;
    TOF7 : TOF;
    Buffer21 : Buffer;
    TOF5 : TOF;
    TOF4 : TOF;
    TOF3 : TOF;
    Balance_isz1 : Balance_isz;
    TOF2 : TOF;
    CAN_Test2 : CAN_Test;
    Buffer12 : Buffer;
    TOF1 : TOF;
    CAN_Test1 : CAN_Test;
    CMS_IVT1 : CMS_IVT;
    TON16 : TON;
    BCU_Fault_Codes1 : BCU_Fault_Codes;
    CTU2 : CTU;
    CTU1 : CTU;
    FLASH1 : FLASH;
    Buffer11 : Buffer;
    Buffer9 : Buffer;
    ISABELinit1 : ISABELinit;
    F_TRIG1 : F_TRIG;
    SR1 : SR;
    TON10 : TON;
    BCU_Cell_Status1 : BCU_Cell_Status;
    Buffer1 : Buffer;
    BCU_ID1 : BCU_ID;
    Buffer19 : Buffer;
    TON11 : TON;
    TON12 : TON;
    TON13 : TON;
    GUICFG_INT2 : GUICFG_INT;
    TON9 : TON;
    TON8 : TON;
    R_TRIG8 : R_TRIG;
    Buffer2 : Buffer;
    Buffer4 : Buffer;
    Buffer3 : Buffer;
    Cell_Voltage_Max_BMU_Loc : USINT := 0;
    Cell_Voltage_Max_Cell_Loc : USINT := 0;
    Cell_Voltage_Min_BMU_Loc : USINT := 0;
    Cell_Voltage_Min_Cell_Loc : USINT := 0;
    Cell_Voltage_Max : UDINT := 0;
    Number_Of_BMU_cfg : USINT;
    Cell_Voltage : UDINT := 0;
    Cell_Temp : REAL := 0;
    NumOfCells : ARRAY[0..15] OF USINT := [15,10,0,0,0,0,0,0,0,0,0,0,0,0,0,0];
    ChannelSelect : ARRAY[0..15] OF PLCHANNEL := [16#0F00,16#0F00,16#0100,16#0100,16#0100,16#0100,16#0100,16#0100,16#0100,16#0100,16#0100,16#0100,16#0F00,16#0100,16#0100,16#0100];
    Total_Voltage : REAL := 0;
    Number_Of_Cell : UINT;
    Cell_Voltage_Min : UDINT := 0;
    Cell_Voltage_Average : UDINT := 0;
    mainChargeComplete : BOOL;
    Balance_Register : UINT := 0;
    OutputVoltage : REAL;
    BatteryVoltage : REAL;
    Pack_DMDC : UINT := 0;
    Pack_DMCC : UINT := 0;
    forceCharge : BOOL;
    cmdBCU : USINT := 0;
    forceDischarge : BOOL;
    whInstant : REAL;
    Selected_BMU_Loc : USINT := 0;
    cellVolt_chargeOK : UINT;
    CAN_ID_10 : UDINT := 0;
    kWhCapacity : REAL := 0;
    voltSample1 : REAL;
    whCapacity : REAL;
    BMS_State : BATTSTATE := 0;
    SoH : USINT := 0;
    Number_Of_Parallel_Cell : USINT := 3;
    cellVolt_nominal : UDINT := 0;
    Cell_Current_Nominal : UDINT := 0;
    Number_Of_BMU : USINT := 0;
    BatteryCurrent : REAL;
    selectLastOne : BOOL;
    cellVolt_max : UINT := 3500;
    voltsample2 : REAL;
    BCU_Charge_Complete : BOOL := 0;
    SoC_CC : USINT := 0;
    Cell_Voltage_Min_Disharge : UINT := 0;
    Cell_Voltage_Max_Charge : UINT := 0;
    cellVolt_dischargeOK : UINT;
    OV_danger : BOOL;
    UV_danger : BOOL;
    CAN_ID_12 : UDINT := 0;
    CAN_ID_11 : UDINT := 0;
    dischargeComplete : BOOL;
    contactEnable_batt : BOOL;
    Cell_Temp_Min_Cell_Loc : USINT := 0;
    Balance_Enable_Rq : BOOL := 0;
    Cell_Temp_Max_BMU_Loc : USINT := 0;
    Cell_Temp_Max_Cell_Loc : USINT := 0;
    Fault_Cell_Under_Temp_Danger : BOOL := 0;
    Fault_Pack_Discharge_Contactor : BOOL := 0;
    Fault_Cell_Over_Temp_Danger : BOOL := 0;
    contactEnable : BOOL;
    CAN_ID_13 : UDINT := 0;
    Cell_Temp_Max : REAL := 0;
    Cell_Temp_Min : REAL := 0;
    Cell_Temp_Min_BMU_Loc : USINT := 0;
    cellVolt_maxCharge : UINT;
    Pack_Charge_Voltage : REAL;
    Selected_Cell_Loc : USINT := 0;
    contactFbk : BOOL;
    cellVolt_cutOffLow : UINT := 2600;
    cellVolt_balThres : UINT := 0;
    cellTemp_maxLim : REAL := 55;
    Pack_Discharge_Voltage : REAL;
    cellTemp_warningOT : REAL := 0;
    cellTemp_warningUT : REAL := 0;
    UV_fault : BOOL;
    UV_danger_risk : BOOL;
    OV_danger_risk : BOOL;
    OT_danger : BOOL;
    cellVolt_minDischarge : UINT;
    chargeCMD : BOOL;
    cellTemp_minLim : REAL := -5;
    Fault_Cell_Under_Temp_Warning : BOOL := 0;
    Fault_Cell_Over_Temp_Warning : BOOL := 0;
    Fault_Cell_Under_Voltage_Warning : BOOL := 0;
    Fault_Cell_Over_Voltage_Warning : BOOL := 0;
    Board_Fault_Messages : UDINT := 0;
    ChargeOK_Voltage_PACK : REAL := 0;
    Fault_Pack_HVIL_1 : BOOL := 0;
    BCU_CAN_CH : TMS570_CAN := TMS570_CAN#L1;
    BMSdmcc_main : REAL;
    CAN_ID_14 : UDINT := 0;
    Balance_Voltage : UDINT := 0;
    Fault_Pack_CMS : BOOL := 0;
    Pack_Temperature : REAL := 0;
    emergencyBtn : BOOL;
    BalanceStateEnb : BOOL;
    CAN_Fault_07 : BOOL := 0;
    Fault_CAN_Communication : BOOL := 0;
    isolationStatus : USINT;
    BCU_Fault_Warning : BOOL := 0;
    CAN_ID_16 : UDINT;
    Fault_Pack_BMU : BOOL := 0;
    cellVolt_min : UINT := 2800;
    CMD_Voltage_Sense_2 : REAL := 0;
    CMD_Voltage_Sense_3 : REAL := 0;
    Charge_Current : UINT := 0;
    CMD_Voltage_Sense_1 : REAL := 0;
    Measure_All : BOOL := 0;
    Measure_Aux : BOOL := 0;
    tauxCells : ARRAY[0..15] OF USINT := [0,0,0,0,1,1,1,1,2,2,2,2,3,3,3,3];
    BCU_Fault_Danger : BOOL := 0;
    CMD_Current_Sense : REAL := 0;
    Fault_DMDC_Exceed : BOOL := 0;
    Fault_DMCC_Exceed : BOOL := 0;
    Fault_Pack_Charge_Contactor : BOOL := 0;
    Board_Error_Messages : UDINT := 0;
    CMD_Counter_Current : REAL := 0;
    Selected_Pack_Number : USINT := 0;
    CMD_Power : REAL := 0;
    Fault_Pack_HVIL_2 : BOOL := 0;
    CMD_Temp : REAL := 0;
    CAN_Fault_05 : BOOL := 0;
    CAN_Fault_04 : BOOL := 0;
    CAN_Fault_02 : BOOL := 0;
    IGNITION : BOOL;
    balChargeSt : USINT;
    CAN_Fault_06 : BOOL := 0;
    Cell_Series_Connection : USINT := 0;
    GUI_Fault : UDINT := 0;
    cellVolt_cutOffHigh : UINT := 3600;
    EPCS_CAN_CH : TMS570_CAN := TMS570_CAN#L3;
    DichargeOK_Voltage_PACK : REAL := 0;
    batteryID : BYTE := 16#01;
    Fault_Cell_Over_Voltage_Danger : BOOL := 0;
    Fault_Cell_Under_Voltage_Danger : BOOL := 0;
    CAN_ID_15 : UDINT := 0;
    Duty_Cycle : UINT := 0;
    CMD_Overall_Power : LREAL := 0;
    UT_danger : BOOL;
    CMS0volt1 : REAL;
    prechargeComplete : BOOL;
    CMS1volt1 : REAL;
    prechargeEnable : BOOL;
    prechargeError : BOOL;
    prechargeCanErr : BOOL;
    prechargeStatus : USINT;
    sim100_ErrByte : BYTE;
    Pack_CutoffLow_Voltage : REAL;
    instantPower : REAL;
    faultsWord : LWORD;
    CAN_Fault_03 : BOOL := 0;
    masterID : BYTE := 16#80;
    HVCU_State : USINT := 0;
    dischargeTerminate : BOOL;
    OV_fault : BOOL;
    UT_danger_risk : BOOL;
    OT_danger_risk : BOOL;
    BMSdmdc_final : REAL;
    BMSdmcc_final : REAL;
    testRemWh : REAL;
    testSocState : USINT;
    inputSgn1 : BOOL;
    inputSgn2 : BOOL;
    inputSgn3 : BOOL;
    outputSgn1 : BOOL;
    outputSgn2 : BOOL;
    IOWR13 : IOWR;
    ANLG8 : ANLG;
    DoD_rate : REAL := 0;
    usableCapkwh : REAL;
    SoCreal : REAL;
    usableCapwh : REAL;
    PackRemCap_kWh : REAL;
    usableRemWh : REAL;
    usableRemkwh : REAL;
    HVIL1_status : BOOL;
    Buffer10 : Buffer;
    TOF6 : TOF;
    Pack_CutoffHigh_Voltage : REAL;
    GUICFG_INT4 : GUICFG_INT;
    GUICFG_INT5 : GUICFG_INT;
    maxDischargeAmprCfg : UINT;
    Tbuffer2 : Tbuffer;
    Tbuffer7 : Tbuffer;
    Pack_CutoffV_Low : REAL;
    CMD_Voltage_Sense1_volt : REAL;
    CMD_Voltage_Sense2_volt : REAL;
    cellVolt_warningOV : UINT;
    cellVolt_warningUV : UINT;
    PDUCAN : TMS570_CAN := TMS570_CAN#L2;
    GUICFG_INT6 : GUICFG_INT;
    OCwarningAmpr : UINT;
    Tbuffer1 : Tbuffer;
    OC_warning : BOOL;
    Tbuffer4 : Tbuffer;
    OC_fault : BOOL;
    contactNegEnable_batt : BOOL;
    contactEnableCharge_batt : BOOL;
    ChargeInVoltage : REAL;
    contactFbkDischarge : BOOL;
    contactFbkCharge : BOOL;
    TOF8 : TOF;
    Buffer22 : Buffer;
    TOF9 : TOF;
    Buffer23 : Buffer;
    Fault_Pack_Negative_Contactor : BOOL;
    dischargeCMD : BOOL;
    prechargeCompleteCharge : BOOL;
    prechargeEnableCharge : BOOL;
    shutdownComplete : BOOL;
    shutdownCMD : BOOL;
    dischargeOff : BOOL;
    chargeOff : BOOL;
    Tbuffer6 : Tbuffer;
    SR2 : SR;
    pduLED : BOOL;
    inputSgn1Status : USINT;
    inputSgn2Status : USINT;
    GUICFG_INT7 : GUICFG_INT;
    GUICFG_INT8 : GUICFG_INT;
    GUICFG_INT9 : GUICFG_INT;
    GUICFG_INT10 : GUICFG_INT;
    GUICFG_INT11 : GUICFG_INT;
    GUICFG_INT12 : GUICFG_INT;
    GUICFG_INT13 : GUICFG_INT;
    GUICFG_INT14 : GUICFG_INT;
    GUICFG_INT15 : GUICFG_INT;
    GUICFG_INT16 : GUICFG_INT;
    GUICFG_INT17 : GUICFG_INT;
    GUICFG_INT18 : GUICFG_INT;
    GUICFG_INT19 : GUICFG_INT;
    GUICFG_INT20 : GUICFG_INT;
    GUICFG_INT21 : GUICFG_INT;
    GUICFG_INT22 : GUICFG_INT;
    GUICFG_INT23 : GUICFG_INT;
    BalanceDiff_Threshold : UDINT;
    GUICFG_REAL1 : GUICFG_REAL;
    GUICFG_INT24 : GUICFG_INT;
    cyclesPerSOH : UINT;
    selClock : BOOL;
    bmuCellVolt : ARRAY[0..15] OF UINT;
    bmuCellTemp : ARRAY[0..15] OF SINT;
    bmuMaxCellV : UINT;
    bmuMinCellV : UINT;
    bmuMinCellT : SINT;
    bmuMaxCellT : SINT;
    warningMdlBalT : BOOL;
    faultMdlBalT : BOOL;
    FaultForState : BOOL;
    maxChargeAmprCfg : UINT;
    HVIL2_status : BOOL;
    TOF10 : TOF;
    Buffer13 : Buffer;
    IMDenable : BOOL;
    isoRp : UDINT;
    isoRn : UDINT;
    isoOhmPerV : UDINT;
    GUICFG_INT25 : GUICFG_INT;
    prechargeInterval : UDINT;
    forceNegative : BOOL;
    contactNegEnable : BOOL;
    contactEnableCharge : BOOL;
    GUICFG_INT26 : GUICFG_INT;
    ntcBETA : UDINT;
    GUICFG_INT27 : GUICFG_INT;
    OCfaultAmpr : UINT;
    Tbuffer15 : Tbuffer;
    Tbuffer16 : Tbuffer;
    SR5 : SR;
    batteryInCharge : BOOL;
    HVCU_Control_State2 : HVCU_Control_State;
    slaveMode : BOOL := TRUE;
    dischargeENB : BOOL;
    chargeENB : BOOL;
    bessStatus : bessSystemStatus;
    bessOperatingStatus : bessOprStatus;
    bessWorkingMode : bessWorkMode;
    batEpcsAlarm : bessAlarms;
    CMD_Current_Sense_Amp : REAL;
    BatteryCharging : BOOL;
    BatteryDischarging : BOOL;
    currentProtection : BOOL;
    Tbuffer20 : Tbuffer;
    Tbuffer19 : Tbuffer;
    TON17 : TON;
    TON2 : TON;
    TON19 : TON;
    TON18 : TON;
    chargeProtect : BOOL;
    dischargeProtect : BOOL;
    essState11 : essState1;
    shutdownEnb : BOOL := BOOL#FALSE;
    prechargeBoardErr : BOOL;
    sim100NotFound : BOOL;
    BatteryWatt : REAL;
    epcsReqData : BOOL;
    F_TRIG3 : F_TRIG;
    F_TRIG4 : F_TRIG;
    R_TRIG9 : R_TRIG;
    socChComp : REAL;
    R_TRIG2 : R_TRIG;
    socDchComp : REAL;
    R_TRIG3 : R_TRIG;
    HVCU_Config1 : HVCU_Config;
    cmdTmt : BOOL;
    ADDRbit0 : BOOL;
    ADDRbit1 : BOOL;
    multAmpChar : REAL;
    multAmpDisch : REAL;
    ampMultTemp1 : ampMultTemp;
    ampMultTemp2 : ampMultTemp;
    ampMultTempDis1 : ampMultTempDis;
    ampMultTempDis2 : ampMultTempDis;
    ampMultVoltDisc1 : ampMultVoltDisc;
    ampMultVoltChar1 : ampMultVoltChar;
    increaseChargeAmp : BOOL;
    increaseDischargeAmp : BOOL;
    decreaseChargeAmp : BOOL;
    decreaseDischargeAmp : BOOL;
    TON21 : TON;
    dischargeAmpEnb : BOOL;
    dischargeUnitAmp : REAL := 0.25;
    chargeAmpEnb : BOOL;
    TON22 : TON;
    chargeUnitAmp : REAL := 0.25;
    maxChargeAmp : REAL;
    maxDischargeAmp : REAL;
    UpDownCntTim1 : UpDownCntTim;
    UpDownCntTim2 : UpDownCntTim;
    BCU_status21 : BCU_status2;
    BCU_State_Message1 : BCU_State_Message;
    BCU_Battery_Status1 : BCU_Battery_Status;
    GUICFG_INT28 : GUICFG_INT;
    testValue0 : TIME;
    TON4 : TON;
    TON5 : TON;
    IOWR4 : IOWR;
    FLASH3 : FLASH;
    SAFETY_POWER1 : SAFETY_POWER;
    ANLG14 : ANLG;
    TON1 : TON;
    TOF15 : TOF;
    BATTSTACK_DISABLE : BOOL;
    CAN_DISABLE : BOOL;
    RDY_TO_SLEEP : BOOL;
    AN_KL15 : UINT;
    IOWR19 : IOWR;
    IOWR6 : IOWR;
    IOWR5 : IOWR;
    IOWR18 : IOWR;
    IOWR20 : IOWR;
    IOWR21 : IOWR;
    FLASH4 : FLASH;
    HW_version : BYTE;
    IOWR9 : IOWR;
    IOWR7 : IOWR;
    IOWR22 : IOWR;
    IOWR23 : IOWR;
    IOWR10 : IOWR;
    IOWR24 : IOWR;
    ANLG4 : ANLG;
    ANLG3 : ANLG;
    ANLG1 : ANLG;
    ANLG2 : ANLG;
    IORD5 : IORD;
    IORD4 : IORD;
    IORD1 : IORD;
    dgtIn8 : dgtIn;
    dgtIn3 : dgtIn;
    dgtIn4 : dgtIn;
    IORD2 : IORD;
    IORD3 : IORD;
    IGNITION_KL15 : BOOL;
    F_TRIG2 : F_TRIG;
    NTC2 : NTC;
    new_CHG_CONTACT : BOOL;
    new_DCHG_CONTACT : BOOL;
    new_contactFbk1 : BOOL;
    new_contactFbk2 : BOOL;
    hkm_DischargeContact : BOOL;
    hkm_DischargeInVoltage : REAL;
    DischargeInVoltage : REAL;
    Number_Of_MaxCell : UINT;
    Number_Of_MaxCell2 : USINT;
    ARR2VAL2 : ARR2VAL;
    NEWBMU_RESET : BOOL := FALSE;
    prechargeCAN1 : prechargeCAN;
    TON26 : TON;
    TON27 : TON;
    ChannelSelect2 : ARRAY[0..15] OF PLCHANNEL := [16#0700,16#0700,16#0700,16#0700,16#0700,16#0700,16#0700,16#0700,16#0700,16#0700,16#0700,16#0700,16#0700,16#0700,16#0700,16#0700];
    AllcontacstEnable : BOOL;
    GUICFG_INT1 : GUICFG_INT;
  END_VAR

  (*

    // Network 1:
    IOWR5(PORT := TMS570_GIO#HET1, PIN := 24, VAL := 1);

    // Network 2:
    IOWR6(PORT := TMS570_GIO#SPI3, PIN := 8, VAL := 1);

    // Network 3:
    ANLG14(ADC := TMSADC#A1, GRP := TMSADCGRP#G1, CH := 7, VAL => AN_KL15);
    GT(IN1 := ANLG14.VAL, IN2 := 100, GT => @C(1379).GT);
    TON1(IN := @C(1379).GT, PT := T#250ms);
    TOF15(IN := TON1.Q, PT := T#800ms, Q => IGNITION_KL15);

    // Network 4:
    TON5(IN := NOT IGNITION_KL15, PT := T#500ms, Q => BATTSTACK_DISABLE);
    TON4(IN := TON5.Q, PT := T#1500ms, Q => RDY_TO_SLEEP);

    // Network 5:
    SAFETY_POWER1(SLEEP_RDY := RDY_TO_SLEEP);

    // Network 6:
    FLASH3(IN := IGNITION_KL15, PER := T#250ms);
    IOWR4(PORT := TMS570_GIO#HET1, PIN := 28, VAL := FLASH3.OUT);

    // Network 7:
    GUICFG_INT1(CODE := 12, R := 1);
    TO_USINT(IN := GUICFG_INT1.VAL, TO_USINT => Number_Of_Parallel_Cell);

    // Network 8:
    GUICFG_INT16(CODE := 110, R := 1);
    TO_UINT(IN := GUICFG_INT16.VAL, TO_UINT => cellVolt_dischargeOK);

    // Network 9:
    BCU_ID1(PACK_ID => Selected_Pack_Number, CAN_ID_10 => CAN_ID_10, CAN_ID_11 => CAN_ID_11, CAN_ID_12 => CAN_ID_12, CAN_ID_13 => CAN_ID_13, CAN_ID_14 => CAN_ID_14, CAN_ID_15 => CAN_ID_15, CAN_ID_16 => CAN_ID_16);

    // Network 10:
    HVCU_Control_State2(CAN_ID := 16#18FF201E, CAN_CH := BCU_CAN_CH, IMDCtrl_BCU0 => IMDenable, CAN_Error => CAN_Fault_07);
    MUX_USINT(K := Selected_Pack_Number, IN0 := HVCU_Control_State2.Battey_State_BCU_00, IN1 := HVCU_Control_State2.Battey_State_BCU_01, IN2 := HVCU_Control_State2.Battey_State_BCU_02, IN3 := HVCU_Control_State2.Battey_State_BCU_03, MUX_USINT => HVCU_State);
    HVCU_Config1(CAN_CH := BCU_CAN_CH, CAN_ID := 16#18FF01F3, CAN_Error => cmdTmt);
    MUX_USINT(K := Selected_Pack_Number, IN0 := HVCU_Config1.cmd0, IN1 := HVCU_Config1.cmd1, IN2 := HVCU_Config1.cmd2, IN3 := HVCU_Config1.cmd3, MUX_USINT => cmdBCU);

    // Network 11:
    GUICFG_INT2(CODE := 10, R := 1);
    TO_UINT(IN := GUICFG_INT2.VAL, TO_UINT => Cell_Current_Nominal);

    // Network 12:
    GUICFG_INT17(CODE := 111, R := 1);
    TO_UINT(IN := GUICFG_INT17.VAL, TO_UINT => cellVolt_warningUV);

    // Network 13:
    GUICFG_INT3(CODE := 261, R := 1);
    TO_USINT(IN := GUICFG_INT3.VAL, TO_USINT => Number_Of_BMU_cfg);

    // Network 14:
    GUICFG_INT18(CODE := 112, R := 1);
    TO_REAL(IN := GUICFG_INT18.VAL, TO_REAL => cellTemp_maxLim);

    // Network 15:
    GUICFG_INT7(CODE := 101, R := 1);
    TO_UINT(IN := GUICFG_INT7.VAL, TO_UINT => cellVolt_cutOffHigh);

    // Network 16:
    GUICFG_INT19(CODE := 113, R := 1);
    TO_REAL(IN := GUICFG_INT19.VAL, TO_REAL => cellTemp_warningOT);

    // Network 17:
    GUICFG_INT8(CODE := 102, R := 1);
    TO_UINT(IN := GUICFG_INT8.VAL, TO_UINT => cellVolt_max);

    // Network 18:
    GUICFG_INT20(CODE := 114, R := 1);
    TO_REAL(IN := GUICFG_INT20.VAL, TO_REAL => cellTemp_minLim);

    // Network 19:
    GUICFG_INT9(CODE := 103, R := 1);
    TO_UINT(IN := GUICFG_INT9.VAL, TO_UINT => cellVolt_maxCharge);

    // Network 20:
    GUICFG_INT21(CODE := 115, R := 1);
    TO_REAL(IN := GUICFG_INT21.VAL, TO_REAL => cellTemp_warningUT);

    // Network 21:
    GUICFG_INT10(CODE := 104, R := 1);
    TO_UINT(IN := GUICFG_INT10.VAL, TO_UINT => cellVolt_chargeOK);

    // Network 22:
    GUICFG_INT22(CODE := 200, R := 1);
    TO_UINT(IN := GUICFG_INT22.VAL, TO_UINT => cellVolt_nominal);

    // Network 23:
    GUICFG_INT11(CODE := 105, R := 1);
    TO_UINT(IN := GUICFG_INT11.VAL, TO_UINT => cellVolt_warningOV);

    // Network 24:
    GUICFG_INT23(CODE := 253, R := 1);
    TO_UINT(IN := GUICFG_INT23.VAL, TO_UINT => BalanceDiff_Threshold);

    // Network 25:
    GUICFG_INT12(CODE := 254, R := 1);
    TO_UINT(IN := GUICFG_INT12.VAL, TO_UINT => cellVolt_balThres);

    // Network 26:
    GUICFG_REAL1(CODE := 120, R := 1, VAL => DoD_rate);

    // Network 27:
    EQ(IN1 := HVCU_State, IN2 := BATTSTATE#CHARGE, EQ => (@C(1658).EQ, chargeCMD));
    EQ(IN1 := HVCU_State, IN2 := BATTSTATE#DISCHARGE, EQ => (@C(1713).EQ, dischargeCMD));
    OR(IN1 := @C(1658).EQ, IN2 := @C(1713).EQ, OR => IGNITION);

    // Network 28:
    GUICFG_INT13(CODE := 107, R := 1);
    TO_UINT(IN := GUICFG_INT13.VAL, TO_UINT => cellVolt_cutOffLow);

    // Network 29:
    GUICFG_INT24(CODE := 121, R := 1);
    TO_UINT(IN := GUICFG_INT24.VAL, TO_UINT => cyclesPerSOH);

    // Network 30:
    GUICFG_INT14(CODE := 108, R := 1);
    TO_UINT(IN := GUICFG_INT14.VAL, TO_UINT => cellVolt_min);

    // Network 31:
    GUICFG_INT25(CODE := 130, R := 1);
    TO_UDINT(IN := GUICFG_INT25.VAL, TO_UDINT => prechargeInterval);

    // Network 32:
    GUICFG_INT15(CODE := 109, R := 1);
    TO_UINT(IN := GUICFG_INT15.VAL, TO_UINT => cellVolt_minDischarge);

    // Network 33:
    GUICFG_INT26(CODE := 266, R := 1);
    TO_UDINT(IN := GUICFG_INT26.VAL, TO_UDINT => ntcBETA);

    // Network 34:
    numOfCells1(numofBMU := Number_Of_BMU_cfg, cellMap := NumOfCells, numofCell => Number_Of_Cell);

    // Network 35:
    GUICFG_INT27(CODE := 2004, R := 1);
    TO_UINT(IN := GUICFG_INT27.VAL, TO_UINT => OCfaultAmpr);

    // Network 36:
    IOWR1(PORT := TMS570_GIO#A, PIN := 0, VAL := 0);

    // Network 37:
    GUICFG_INT4(CODE := 2001, R := 1);
    TO_UINT(IN := GUICFG_INT4.VAL, TO_UINT => @C(1169).TO_UINT);
    MIN(IN1 := @C(1169).TO_UINT, IN2 := 200, MIN => maxChargeAmprCfg);

    // Network 38:
    GUICFG_INT28(CODE := 400, R := 1);
    TO_UDINT(IN := GUICFG_INT28.VAL, TO_UDINT => @C(733).TO_UDINT);
    TO_TIME(IN := @C(733).TO_UDINT, TO_TIME => @C(1172).TO_TIME);
    DIV_TIME(IN1 := @C(1172).TO_TIME, IN2 := 1000, DIV_TIME => testValue0);

    // Network 39:
    GUICFG_INT5(CODE := 2002, R := 1);
    TO_UINT(IN := GUICFG_INT5.VAL, TO_UINT => @C(1538).TO_UINT);
    MIN(IN1 := @C(1538).TO_UINT, IN2 := 300, MIN => maxDischargeAmprCfg);

    // Network 40:
    IOWR2(PORT := TMS570_GIO#B, PIN := 3, VAL := 1);

    // Network 41:
    EQ(IN1 := cmdBCU, IN2 := 16#AB, EQ => forceDischarge);

    // Network 42:
    GUICFG_INT6(CODE := 2003, R := 1);
    TO_UINT(IN := GUICFG_INT6.VAL, TO_UINT => @C(869).TO_UINT);
    MIN(IN1 := @C(869).TO_UINT, IN2 := 250, MIN => OCwarningAmpr);

    // Network 43:
    EQ(IN1 := cmdBCU, IN2 := 16#AC, EQ => forceCharge);

    // Network 44:
    EQ(IN1 := cmdBCU, IN2 := 16#AD, EQ => forceNegative);

    // Network 45:
    TO_REAL(IN := cellVolt_chargeOK, TO_REAL => @C(962).TO_REAL);
    MUL(IN1 := Number_Of_Cell, IN2 := @C(962).TO_REAL, MUL => @C(958).MUL);
    DIV(IN1 := @C(958).MUL, IN2 := 1000, DIV => ChargeOK_Voltage_PACK);
    TO_REAL(IN := cellVolt_dischargeOK, TO_REAL => @C(972).TO_REAL);
    MUL(IN1 := Number_Of_Cell, IN2 := @C(972).TO_REAL, MUL => @C(971).MUL);
    DIV(IN1 := @C(971).MUL, IN2 := 1000, DIV => DichargeOK_Voltage_PACK);
    MUL(IN1 := Number_Of_Cell, IN2 := cellVolt_maxCharge, MUL => @C(502).MUL);
    DIV(IN1 := @C(502).MUL, IN2 := 1000, DIV => Pack_Charge_Voltage);
    MUL(IN1 := Number_Of_Cell, IN2 := cellVolt_minDischarge, MUL => @C(517).MUL);
    DIV(IN1 := @C(517).MUL, IN2 := 1000, DIV => Pack_Discharge_Voltage);
    MUL(IN1 := Number_Of_Cell, IN2 := cellVolt_cutOffLow, MUL => @C(1353).MUL);
    DIV(IN1 := @C(1353).MUL, IN2 := 1000, DIV => Pack_CutoffLow_Voltage);
    MUL(IN1 := Number_Of_Cell, IN2 := cellVolt_cutOffHigh, MUL => @C(479).MUL);
    DIV(IN1 := @C(479).MUL, IN2 := 1000, DIV => Pack_CutoffHigh_Voltage);

    // Network 46:
    TO_UINT(IN := bmuCellVolt[0], TO_UINT => @C(415).TO_UINT);
    TO_UINT(IN := bmuCellVolt[1], TO_UINT => @C(419).TO_UINT);
    TO_UINT(IN := bmuCellVolt[2], TO_UINT => @C(420).TO_UINT);
    TO_UINT(IN := bmuCellVolt[3], TO_UINT => @C(421).TO_UINT);
    CAN_Test1(IN_1 := @C(415).TO_UINT, IN_2 := @C(419).TO_UINT, IN_3 := @C(420).TO_UINT, IN_4 := @C(421).TO_UINT, CAN_CH := BCU_CAN_CH, CAN_ID := 16#10000001);
    TO_UINT(IN := bmuCellVolt[4], TO_UINT => @C(422).TO_UINT);
    TO_UINT(IN := bmuCellVolt[5], TO_UINT => @C(423).TO_UINT);
    TO_UINT(IN := bmuCellVolt[6], TO_UINT => @C(424).TO_UINT);
    TO_UINT(IN := sim100NotFound, TO_UINT => @C(425).TO_UINT);
    CAN_Test2(IN_1 := @C(422).TO_UINT, IN_2 := @C(423).TO_UINT, IN_3 := @C(424).TO_UINT, IN_4 := @C(425).TO_UINT, CAN_CH := BCU_CAN_CH, CAN_ID := 16#10000002);

    // Network 47:
    SEL();

    // Network 48:
    AND(IN1 := slaveMode, IN2 := CAN_Fault_07, AND => Fault_CAN_Communication);

    // Network 49:
    ISABELinit1(CH := PDUCAN, ENB := 1);
    CMS_IVT1(CAN_CH := PDUCAN, Current_mA => CMD_Current_Sense, Voltage1_mV => CMD_Voltage_Sense_1, Voltage2_mV => CMD_Voltage_Sense_2, Voltage3_mV => CMD_Voltage_Sense_3, Temp => CMD_Temp, Power_kWh => CMD_Power, Current_Counter_Ah => CMD_Counter_Current, Power_Counter_Wh => whInstant, CAN_Error => Fault_Pack_CMS, Overall_Power_kWh => CMD_Overall_Power);
    DIV(IN1 := CMD_Current_Sense, IN2 := 1000, DIV => BatteryCurrent);
    DIV(IN1 := CMD_Voltage_Sense_1, IN2 := 1000, DIV => BatteryVoltage);
    DIV(IN1 := CMD_Voltage_Sense_2, IN2 := 1000, DIV => (OutputVoltage, ChargeInVoltage));
    DIV(IN1 := CMD_Voltage_Sense_3, IN2 := 1000, DIV => DischargeInVoltage);

    // Network 50:
    GE(IN1 := BatteryCurrent, IN2 := 0.5, GE => @C(2595).GE);
    Tbuffer19(I := @C(2595).GE, D := T#500ms, O => BatteryDischarging);
    LE(IN1 := BatteryCurrent, IN2 := -0.5, LE => @C(2605).LE);
    Tbuffer20(I := @C(2605).LE, D := T#500ms, O => BatteryCharging);

    // Network 51:
    LT(IN1 := BatteryCurrent, IN2 := -0.2, LT => @C(753).LT);
    Tbuffer15(I := @C(753).LT, D := T#1s);
    GT(IN1 := BatteryCurrent, IN2 := 0.1, GT => @C(755).GT);
    Tbuffer16(I := @C(755).GT, D := T#1s);
    SR5(S1 := Tbuffer15.O, R := Tbuffer16.O, Q1 => batteryInCharge);

    // Network 52:
    ABS(IN := BatteryCurrent, ABS => @C(2251).ABS);
    GE(IN1 := @C(2251).ABS, IN2 := OCwarningAmpr, GE => @C(897).GE);
    Tbuffer1(I := @C(897).GE, D := T#100ms, O => OC_warning);
    GE(IN1 := @C(2251).ABS, IN2 := OCfaultAmpr, GE => @C(917).GE);
    Tbuffer4(I := @C(917).GE, D := T#100ms, O => OC_fault);

    // Network 53:
    TO_TIME(IN := prechargeInterval, TO_TIME => @C(3224).TO_TIME);
    DIV_TIME(IN1 := @C(3224).TO_TIME, IN2 := 1000, DIV_TIME => @C(3225).DIV_TIME);
    GT(IN1 := BatteryVoltage, IN2 := Pack_CutoffLow_Voltage, GT => @C(3228).GT);
    SUB(IN1 := BatteryVoltage, IN2 := OutputVoltage, SUB => @C(3231).SUB);
    ABS(IN := @C(3231).SUB, ABS => @C(3229).ABS);
    LT(IN1 := @C(3229).ABS, IN2 := 8, LT => @C(3232).LT);
    TON26(IN := @C(3232).LT, PT := @C(3225).DIV_TIME);
    AND(IN1 := @C(3228).GT, IN2 := TON26.Q, AND => prechargeComplete);
    GT(IN1 := BatteryVoltage, IN2 := Pack_CutoffLow_Voltage, GT => @C(3233).GT);
    SUB(IN1 := BatteryVoltage, IN2 := ChargeInVoltage, SUB => @C(3236).SUB);
    ABS(IN := @C(3236).SUB, ABS => @C(3235).ABS);
    LT(IN1 := @C(3235).ABS, IN2 := 8, LT => @C(3237).LT);
    TON27(IN := @C(3237).LT, PT := @C(3225).DIV_TIME);
    AND(IN1 := @C(3233).GT, IN2 := TON27.Q, AND => prechargeCompleteCharge);

    // Network 54:
    ABS(IN := BatteryCurrent, ABS => @C(1258).ABS);
    LT(IN1 := @C(1258).ABS, IN2 := 3, LT => shutdownComplete);

    // Network 55:
    IOWR13(PORT := TMS570_GIO#HET1, PIN := 24, VAL := 1);

    // Network 56:
    ANLG8(ADC := TMSADC#A1, GRP := TMSADCGRP#G1, CH := 10);

    // Network 57:
    IOWR22(PORT := TMS570_GIO#A, PIN := 7);

    // Network 58:
    IOWR23(PORT := TMS570_GIO#A, PIN := 6);

    // Network 59:
    IOWR7(PORT := TMS570_GIO#HET1, PIN := 22);

    // Network 60:
    IOWR9(PORT := TMS570_GIO#HET1, PIN := 8);

    // Network 61:
    dgtIn4(ch := 2);
    EQ(IN1 := 1, IN2 := dgtIn4.stat, EQ => contactFbkDischarge);
    dgtIn3(ch := 3);
    EQ(IN1 := dgtIn3.stat, IN2 := 1, EQ => contactFbkCharge);

    // Network 62:
    EQ(IN1 := HW_version, IN2 := 1, EQ => @C(1957).EQ);
    SEL(G := @C(1957).EQ, IN0 := 0, IN1 := 1, SEL => @C(1958).SEL);
    IOWR19(PORT := TMS570_GIO#SPI2, PIN := 10, VAL := @C(1958).SEL);

    // Network 63:
    dgtIn8(ch := 4);

    // Network 64:
    IORD1(PORT := TMS570_GIO#HET1, PIN := 12);

    // Network 65:
    IORD4(PORT := TMS570_GIO#HET1, PIN := 16);

    // Network 66:
    IORD5(PORT := TMS570_GIO#HET1, PIN := 14);

    // Network 67:
    IORD2(PORT := TMS570_GIO#HET1, PIN := 18);

    // Network 68:
    HVIL1_status := 1;

    // Network 69:
    NOT(IN := HVIL1_status, NOT => @C(510).NOT);
    Buffer10(I := @C(510).NOT);
    TOF6(IN := Buffer10.O, PT := T#3s, Q => Fault_Pack_HVIL_1);

    // Network 70:
    HVIL2_status := 1;

    // Network 71:
    NOT(IN := HVIL2_status, NOT => @C(2154).NOT);
    Buffer13(I := @C(2154).NOT);
    TOF10(IN := Buffer13.O, PT := T#3s, Q => Fault_Pack_HVIL_2);

    // Network 72:
    IORD3(PORT := TMS570_GIO#HET1, PIN := 17);

    // Network 73:
    ANLG1(ADC := TMSADC#A1, GRP := TMSADCGRP#G1, CH := 6);
    NTC2(VOLT := ANLG1.VAL, VSUP := 7000, RS := 10000, BETA := 3950, TNOM := 298.15, RNOM := 10000, TEMP => Pack_Temperature);

    // Network 74:
    IOWR18(PORT := TMS570_GIO#SPI2, PIN := 0, VAL := 1);

    // Network 75:
    ANLG2(ADC := TMSADC#A1, GRP := TMSADCGRP#G1, CH := 5);

    // Network 76:
    OR(IN1 := contactFbkCharge, IN2 := contactFbkDischarge, OR => contactFbk);

    // Network 77:
    IOWR20(PORT := TMS570_GIO#SPI2, PIN := 11, VAL := 1);

    // Network 78:
    ANLG3(ADC := TMSADC#A1, GRP := TMSADCGRP#G1, CH := 8);

    // Network 79:
    FLASH4(IN := 1, PER := T#3s);
    IOWR21(PORT := TMS570_GIO#SPI2, PIN := 9, VAL := FLASH4.OUT);

    // Network 80:
    ANLG4(ADC := TMSADC#A1, GRP := TMSADCGRP#G1, CH := 11);

    // Network 81:
    BCU_State_Message1(CAN_ID := CAN_ID_10, State := BMS_State, Contactor_Status := contactFbk, ChargeContact := contactFbkCharge, Ambient_Temp := Cell_Temp_Min, DMDC := Pack_DMDC, DMCC := Pack_DMCC, CAN_CH := BCU_CAN_CH, NegContact := contactFbkDischarge, isolationStatus := isolationStatus, chargeComplete := chargeProtect, dischargeComplete := dischargeProtect, emergencyButton := prechargeBoardErr, in1Status := inputSgn1Status, in2Status := inputSgn2Status);
    BCU_Cell_Status1(Selected_BMU_Loc := Selected_BMU_Loc, Selected_Cell_Loc := Selected_Cell_Loc, Cell_Voltage := Cell_Voltage, Cell_Temp := Cell_Temp, CAN_ID := CAN_ID_11, CAN_CH := BCU_CAN_CH, Total_Voltage := Total_Voltage, Instant_Current := BatteryCurrent, CAN_Error => CAN_Fault_03);
    Max_Min_Voltage_Status1(Max_Volt_BMU_Loc := Cell_Voltage_Max_BMU_Loc, Max_Volt_Cell_Loc := Cell_Voltage_Max_Cell_Loc, Min_Volt_BMU_Loc := Cell_Voltage_Min_BMU_Loc, Min_Volt_Cell_Loc := Cell_Voltage_Min_Cell_Loc, Max_Cell_Voltage := Cell_Voltage_Max, Min_Cell_Voltage := Cell_Voltage_Min, Average_Cell_Voltage := Cell_Voltage_Average, CAN_ID := CAN_ID_12, CAN_CH := BCU_CAN_CH, CAN_Error => CAN_Fault_04);
    BCU_status21(Max_Temp_BMU_Loc := Cell_Temp_Max_BMU_Loc, Max_Temp_Cell_Loc := Cell_Temp_Max_Cell_Loc, Min_Temp_BMU_Loc := Cell_Temp_Min_BMU_Loc, Min_Temp_Cell_Loc := Cell_Temp_Min_Cell_Loc, Max_Cell_Temp := Cell_Temp_Max, Min_Cell_Temp := Cell_Temp_Min, CAN_ID := CAN_ID_13, CAN_CH := BCU_CAN_CH, outVolt := OutputVoltage, CAN_Error => CAN_Fault_05);
    BCU_Battery_Status1(SoC := SoC_CC, SoH := SoH, Duty_Cycle := Duty_Cycle, Remain_Energy := usableRemkwh, CAN_ID := CAN_ID_14, CAN_CH := BCU_CAN_CH, Available_Energy := usableCapkwh, CAN_Error => CAN_Fault_06);

    // Network 82:
    OR(IN1 := UV_danger, IN2 := dischargeComplete, OR => (@C(1278).OR, dischargeProtect));
    GT(IN1 := BatteryCurrent, IN2 := 5, GT => @C(1296).GT);
    AND(IN1 := @C(1296).GT, IN2 := @C(1278).OR, AND => @C(1291).AND);
    TON17(IN := @C(1291).AND, PT := T#3s);
    AND(IN1 := BatteryDischarging, IN2 := @C(1278).OR, AND => @C(2358).AND);
    TON2(IN := @C(2358).AND, PT := T#120s);
    OR(IN1 := TON17.Q, IN2 := TON2.Q, OR => @C(1304).OR);
    AND(IN1 := @C(1278).OR, IN2 := @C(1304).OR, AND => dischargeOff);

    // Network 83:
    OR(IN1 := OV_danger, IN2 := BCU_Charge_Complete, OR => (@C(1315).OR, chargeProtect));
    LT(IN1 := BatteryCurrent, IN2 := -5, LT => @C(1283).LT);
    AND(IN1 := @C(1283).LT, IN2 := @C(1315).OR, AND => @C(1375).AND);
    TON19(IN := @C(1375).AND, PT := T#3s);
    AND(IN1 := BatteryCharging, IN2 := @C(1315).OR, AND => @C(1313).AND);
    TON18(IN := @C(1313).AND, PT := T#120s);
    OR(IN1 := TON19.Q, IN2 := TON18.Q, OR => @C(1282).OR);
    AND(IN1 := @C(1315).OR, IN2 := @C(1282).OR, AND => chargeOff);

    // Network 84:
    OR(IN1 := chargeOff, IN2 := dischargeOff, IN3 := emergencyBtn, OR => currentProtection);

    // Network 85:
    SEL(G := slaveMode, IN0 := NOT batteryInCharge, IN1 := dischargeCMD, SEL => @C(1642).SEL);
    AND(IN1 := NOT currentProtection, IN2 := @C(1642).SEL, AND => dischargeENB);
    SEL(G := slaveMode, IN0 := batteryInCharge, IN1 := chargeCMD, SEL => @C(1648).SEL);
    AND(IN1 := NOT currentProtection, IN2 := @C(1648).SEL, AND => chargeENB);

    // Network 86:
    TO_REAL(IN := ntcBETA, TO_REAL => @C(265).TO_REAL);
    BATTSTACK1(NBOARDS := Number_Of_BMU_cfg, BAUD := 250000, OVTHRES := Cell_Voltage_Max_Charge, UVTHRES := Cell_Voltage_Min_Disharge, M_ALL_R := Measure_All, M_AUX_R := Measure_Aux, N_CELLS := NumOfCells, T_CELLS := tauxCells, CHSEL := ChannelSelect, BRD := Selected_BMU_Loc, CELL := Selected_Cell_Loc, CH := PLCHANNEL#AUX0, BALV := Balance_Voltage, BALENB := Balance_Enable_Rq, NTCBETA := @C(265).TO_REAL, NTCNOMT_KLV := 298.15, NTCNOMR_OHM := 10000.0, ENB := 1, N_BRD => Number_Of_BMU, VCELL => Cell_Voltage, VAV => Cell_Voltage_Average, VMINCELL => Cell_Voltage_Min, VMAXCELL => Cell_Voltage_Max, VSTACK => Total_Voltage, MAXCELLBRD => Cell_Voltage_Max_BMU_Loc, MAXCELLNUM => Cell_Voltage_Max_Cell_Loc, MINCELLBRD => Cell_Voltage_Min_BMU_Loc, MINCELLNUM => Cell_Voltage_Min_Cell_Loc, BALREG => Balance_Register, TEMPCELL => Cell_Temp, MAXTEMP => Cell_Temp_Max, MINTEMP => Cell_Temp_Min, MAXTEMPBRD => Cell_Temp_Max_BMU_Loc, MAXTEMPCELL => Cell_Temp_Max_Cell_Loc, MINTEMPBRD => Cell_Temp_Min_BMU_Loc, MINTEMPCELL => Cell_Temp_Min_Cell_Loc, FAULT => Board_Fault_Messages, ERR => Board_Error_Messages);

    // Network 87:
    LT(IN1 := Cell_Voltage_Min, IN2 := cellVolt_cutOffLow, LT => @C(803).LT);
    Buffer1(I := @C(803).LT);
    LT(IN1 := Total_Voltage, IN2 := Pack_CutoffLow_Voltage, LT => @C(1669).LT);
    Buffer3(I := @C(1669).LT);
    OR(IN1 := Buffer1.O, IN2 := Buffer3.O, OR => UV_fault);
    GT(IN1 := Cell_Voltage_Max, IN2 := cellVolt_cutOffHigh, GT => @C(1684).GT);
    Buffer2(I := @C(1684).GT);
    GT(IN1 := Total_Voltage, IN2 := Pack_CutoffHigh_Voltage, GT => @C(1825).GT);
    Buffer4(I := @C(1825).GT);
    OR(IN1 := Buffer2.O, IN2 := Buffer4.O, OR => OV_fault);

    // Network 88:
    GE(IN1 := Cell_Voltage_Max, IN2 := cellVolt_warningOV, GE => @C(364).GE);
    TON6(IN := @C(364).GE, PT := T#100ms, Q => OV_danger_risk);
    GE(IN1 := Cell_Voltage_Max, IN2 := cellVolt_max, GE => @C(1580).GE);
    TON8(IN := @C(1580).GE, PT := T#20s, Q => OV_danger);

    // Network 89:
    LE(IN1 := Cell_Voltage_Min, IN2 := cellVolt_warningUV, LE => @C(404).LE);
    TON7(IN := @C(404).LE, PT := T#100ms, Q => UV_danger_risk);
    LE(IN1 := Cell_Voltage_Min, IN2 := cellVolt_min, LE => @C(1582).LE);
    TON9(IN := @C(1582).LE, PT := T#20s, Q => UV_danger);

    // Network 90:
    SUB(IN1 := cellTemp_maxLim, IN2 := 1, SUB => @C(276).SUB);
    GE(IN1 := Cell_Temp_Max, IN2 := @C(276).SUB, GE => @C(279).GE);
    TON10(IN := @C(279).GE, PT := T#500ms, Q => OT_danger_risk);
    GE(IN1 := Cell_Temp_Max, IN2 := cellTemp_maxLim, GE => @C(920).GE);
    TON12(IN := @C(920).GE, PT := T#2s, Q => OT_danger);

    // Network 91:
    ADD(IN1 := cellTemp_minLim, IN2 := 1, ADD => @C(277).ADD);
    LE(IN1 := Cell_Temp_Min, IN2 := @C(277).ADD, LE => @C(919).LE);
    TON11(IN := @C(919).LE, PT := T#500ms, Q => UT_danger_risk);
    LE(IN1 := Cell_Temp_Min, IN2 := cellTemp_minLim, LE => @C(1073).LE);
    TON13(IN := @C(1073).LE, PT := T#2s, Q => UT_danger);

    // Network 92:
    Buffer12(I := OV_danger_risk);
    TOF1(IN := Buffer12.O, PT := T#3s, Q => Fault_Cell_Over_Voltage_Warning);

    // Network 93:
    OR(IN1 := OV_danger, IN2 := OV_fault, OR => @C(259).OR);
    TOF12(IN := @C(259).OR, PT := T#3s, Q => Fault_Cell_Over_Voltage_Danger);

    // Network 94:
    Buffer19(I := UV_danger_risk);
    TOF14(IN := Buffer19.O, PT := T#3s, Q => Fault_Cell_Under_Voltage_Warning);

    // Network 95:
    OR(IN1 := UV_danger, IN2 := UV_fault, OR => @C(1813).OR);
    TOF13(IN := @C(1813).OR, PT := T#3s, Q => Fault_Cell_Under_Voltage_Danger);

    // Network 96:
    GE(IN1 := Cell_Temp_Max, IN2 := cellTemp_warningOT, GE => @C(288).GE);
    Buffer11(I := @C(288).GE);
    TOF3(IN := Buffer11.O, PT := T#3s, Q => Fault_Cell_Over_Temp_Warning);

    // Network 97:
    TOF2(IN := OT_danger, PT := T#3s, Q => Fault_Cell_Over_Temp_Danger);

    // Network 98:
    LE(IN1 := Cell_Temp_Min, IN2 := cellTemp_warningUT, LE => @C(286).LE);
    Buffer9(I := @C(286).LE);
    TOF5(IN := Buffer9.O, PT := T#3s, Q => Fault_Cell_Under_Temp_Warning);

    // Network 99:
    OR(IN1 := Fault_Cell_Over_Voltage_Warning, IN2 := Fault_Cell_Under_Voltage_Warning, IN3 := Fault_Cell_Over_Temp_Warning, IN4 := Fault_Cell_Under_Temp_Warning, IN5 := warningMdlBalT, OR => BCU_Fault_Warning);

    // Network 100:
    NE(IN1 := Number_Of_BMU, IN2 := Number_Of_BMU_cfg, NE => @C(932).NE);
    Tbuffer2(I := @C(932).NE, D := T#3s);
    TO_DWORD(IN := Board_Error_Messages, TO_DWORD => @C(1213).TO_DWORD);
    AND(IN1 := @C(1213).TO_DWORD, IN2 := 16#00000001, AND => @C(1215).AND);
    TO_BOOL(IN := @C(1215).AND, TO_BOOL => @C(1239).TO_BOOL);
    AND(IN1 := @C(1213).TO_DWORD, IN2 := 16#00000002, AND => @C(934).AND);
    TO_BOOL(IN := @C(934).AND, TO_BOOL => @C(1233).TO_BOOL);
    AND(IN1 := @C(1213).TO_DWORD, IN2 := 16#00000004, AND => @C(1229).AND);
    TO_BOOL(IN := @C(1229).AND, TO_BOOL => @C(1227).TO_BOOL);
    OR(IN1 := @C(1239).TO_BOOL, IN2 := @C(1233).TO_BOOL, IN3 := @C(1227).TO_BOOL, OR => @C(1243).OR);
    Tbuffer7(I := @C(1243).OR, D := T#3s);
    OR(IN1 := Tbuffer2.O, IN2 := Tbuffer7.O, OR => Fault_Pack_BMU);

    // Network 101:
    TOF4(IN := UT_danger, PT := T#3s, Q => Fault_Cell_Under_Temp_Danger);

    // Network 102:
    ampMultTemp1(temp := Cell_Temp_Max);
    ampMultTemp2(temp := Cell_Temp_Min);
    MIN(IN1 := ampMultTemp1.mult, IN2 := ampMultTemp2.mult, MIN => @C(838).MIN);
    ampMultVoltChar1(chargeOn := BatteryCharging, maxCell := Cell_Voltage_Max);
    MUL(IN1 := @C(838).MIN, IN2 := ampMultVoltChar1.mult, MUL => multAmpChar);

    // Network 103:
    ampMultTempDis1(temp := Cell_Temp_Max);
    ampMultTempDis2(temp := Cell_Temp_Min);
    MIN(IN1 := ampMultTempDis1.mult, IN2 := ampMultTempDis2.mult, MIN => @C(1195).MIN);
    ampMultVoltDisc1(discOn := BatteryDischarging, minCell := Cell_Voltage_Min);
    MUL(IN1 := @C(1195).MIN, IN2 := ampMultVoltDisc1.mult, MUL => multAmpDisch);

    // Network 104:
    MUL(IN1 := multAmpChar, IN2 := maxChargeAmprCfg, MUL => maxChargeAmp);

    // Network 105:
    MUL(IN1 := multAmpDisch, IN2 := maxDischargeAmprCfg, MUL => maxDischargeAmp);

    // Network 106:
    GT(IN1 := cmdBCU, IN2 := 16#AA, GT => @C(657).GT);
    AND(IN1 := NOT cmdTmt, IN2 := @C(657).GT, AND => @C(672).AND);
    SEL(G := @C(672).AND, IN0 := AllcontacstEnable, IN1 := forceDischarge, SEL => contactEnable);
    SEL(G := @C(672).AND, IN0 := contactNegEnable_batt, IN1 := forceNegative, SEL => contactNegEnable);
    SEL(G := @C(672).AND, IN0 := contactEnable_batt, IN1 := forceCharge, SEL => contactEnableCharge);

    // Network 107:
    NE(IN1 := contactEnable, IN2 := contactFbk, NE => @C(243).NE);
    Buffer21(I := @C(243).NE);
    TOF7(IN := Buffer21.O, PT := T#3s, Q => Fault_Pack_Discharge_Contactor);

    // Network 108:
    NE(IN1 := contactNegEnable, IN2 := contactFbkDischarge, NE => @C(1092).NE);
    Buffer22(I := @C(1092).NE);
    TOF8(IN := Buffer22.O, PT := T#3s, Q => Fault_Pack_Negative_Contactor);

    // Network 109:
    NE(IN1 := contactEnableCharge, IN2 := contactFbkCharge, NE => @C(1109).NE);
    Buffer23(I := @C(1109).NE);
    TOF9(IN := Buffer23.O, PT := T#3s, Q => Fault_Pack_Charge_Contactor);

    // Network 110:
    OR(IN1 := Fault_Cell_Over_Temp_Danger, IN2 := Fault_Cell_Under_Temp_Danger, IN3 := Fault_CAN_Communication, IN4 := Fault_Pack_HVIL_1, IN5 := Fault_Pack_BMU, IN6 := Fault_Pack_Discharge_Contactor, IN7 := Fault_Cell_Over_Voltage_Danger, IN8 := Fault_Cell_Under_Voltage_Danger, IN9 := OC_fault, IN10 := faultMdlBalT, IN11 := Fault_Pack_HVIL_2, IN12 := Fault_Pack_Negative_Contactor, IN13 := Fault_Pack_Charge_Contactor, IN14 := Fault_Pack_CMS, OR => BCU_Fault_Danger);

    // Network 111:
    BCU_Fault_Codes1(CAN_ID := CAN_ID_16, Fault_00 := BCU_Fault_Warning, Fault_01 := BCU_Fault_Danger, Fault_02 := Fault_Cell_Over_Voltage_Warning, Fault_03 := Fault_Cell_Over_Voltage_Danger, Fault_04 := Fault_Cell_Under_Voltage_Warning, Fault_05 := Fault_Cell_Under_Voltage_Danger, Fault_06 := Fault_Cell_Over_Temp_Warning, Fault_07 := Fault_Cell_Over_Temp_Danger, Fault_08 := Fault_Cell_Under_Temp_Warning, Fault_09 := Fault_Cell_Under_Temp_Danger, Fault_10 := OC_warning, Fault_11 := OC_fault, Fault_12 := Fault_Pack_CMS, Fault_13 := Fault_Pack_Discharge_Contactor, Fault_14 := Fault_Pack_Charge_Contactor, Fault_15 := Fault_Pack_HVIL_1, Fault_16 := Fault_Pack_HVIL_2, Fault_20 := Fault_Pack_BMU, Fault_21 := Fault_Pack_Negative_Contactor, Fault_22 := prechargeError, Fault_25 := warningMdlBalT, Fault_26 := faultMdlBalT, Fault_33 := Fault_CAN_Communication, Fault_Byte_5 := Board_Error_Messages, CAN_CH := BCU_CAN_CH, Fault_Byte_6_7 := Board_Fault_Messages, GUI_Fault => GUI_Fault, sum => faultsWord);

    // Network 112:
    OR(IN1 := Fault_Cell_Over_Temp_Danger, IN2 := Fault_Cell_Under_Temp_Danger, IN3 := Fault_CAN_Communication, IN4 := Fault_Pack_HVIL_1, IN5 := Fault_Pack_BMU, IN6 := Fault_Pack_Discharge_Contactor, IN7 := OV_fault, IN8 := UV_fault, IN9 := OC_fault, IN11 := Fault_Pack_Negative_Contactor, IN12 := Fault_Pack_Charge_Contactor, IN13 := Fault_Pack_CMS, OR => FaultForState);

    // Network 113:
    GUI1(Voltage := CMD_Voltage_Sense_1, Current := CMD_Current_Sense, Temp := Pack_Temperature, Humidity := BMSdmcc_final, Fault := GUI_Fault, SoC := SoC_CC, SoH := SoH, Cycle := Duty_Cycle, State := BMS_State, ID := Selected_Pack_Number, CH := BCU_CAN_CH);

    // Network 114:
    MUL(IN1 := Number_Of_Cell, IN2 := Number_Of_Parallel_Cell, IN3 := Cell_Current_Nominal, IN4 := cellVolt_nominal, MUL => @C(74).MUL);
    TO_REAL(IN := @C(74).MUL, TO_REAL => @C(73).TO_REAL);
    DIV(IN1 := @C(73).TO_REAL, IN2 := 1000000, DIV => kWhCapacity);
    MUL(IN1 := kWhCapacity, IN2 := SoCreal, MUL => @C(2073).MUL);
    DIV(IN1 := @C(2073).MUL, IN2 := 100, DIV => PackRemCap_kWh);

    // Network 115:
    MUL(IN1 := DoD_rate, IN2 := kWhCapacity, MUL => (@C(1367).MUL, usableCapkwh));
    MUL(IN1 := @C(1367).MUL, IN2 := 1000, MUL => usableCapwh);

    // Network 116:
    DIV(IN1 := CMD_Overall_Power, IN2 := kWhCapacity, DIV => @C(1978).DIV);
    TO_USINT(IN := @C(1978).DIV, TO_USINT => Duty_Cycle);

    // Network 117:
    DIV(IN1 := Duty_Cycle, IN2 := cyclesPerSOH, DIV => @C(1985).DIV);
    SUB(IN1 := 100, IN2 := @C(1985).DIV, SUB => @C(1990).SUB);
    LIMIT(MN := 0, IN := @C(1990).SUB, MX := 100, LIMIT => @C(1993).LIMIT);
    TO_USINT(IN := @C(1993).LIMIT, TO_USINT => SoH);

    // Network 118:
    ARR2VAL2(MaxBMU := Number_Of_BMU_cfg, indx := Selected_BMU_Loc, Map := NumOfCells, CellCounter := Selected_Cell_Loc, numofCell => Number_Of_MaxCell, Reset => NEWBMU_RESET);

    // Network 119:
    FLASH1(IN := 1, PER := T#250ms, OUT => selClock);
    TO_USINT(IN := Number_Of_MaxCell, TO_USINT => @C(1002).TO_USINT);
    CTU2(CU := CTU1.Q, R := NEWBMU_RESET, PV := Number_Of_BMU_cfg);
    CTU1(CU := FLASH1.OUT, R := CTU1.Q, PV := @C(1002).TO_USINT);
    TO_USINT(IN := CTU2.CV, TO_USINT => Selected_BMU_Loc);
    TO_USINT(IN := CTU1.CV, TO_USINT => Selected_Cell_Loc);

    // Network 120:
    GE(IN1 := Total_Voltage, IN2 := ChargeOK_Voltage_PACK, GE => @C(887).GE);
    GE(IN1 := Cell_Voltage_Max, IN2 := cellVolt_chargeOK, GE => @C(544).GE);
    OR(IN1 := @C(887).GE, IN2 := @C(544).GE, OR => @C(542).OR);
    SUB(IN1 := socChComp, IN2 := SoCreal, SUB => @C(582).SUB);
    GT(IN1 := @C(582).SUB, IN2 := 2, GT => @C(742).GT);
    GE(IN1 := BatteryCurrent, IN2 := -5, GE => @C(757).GE);
    AND(IN1 := @C(542).OR, IN2 := @C(757).GE, AND => @C(1702).AND);
    TON16(IN := @C(1702).AND, PT := T#15s);
    SR1(S1 := TON16.Q, R := @C(742).GT, Q1 => mainChargeComplete);

    // Network 121:
    F_TRIG1(CLK := IGNITION);
    F_TRIG2(CLK := IGNITION_KL15);
    OR(IN1 := F_TRIG1.Q, IN2 := F_TRIG2.Q, OR => @C(223).OR);
    SOCisz1(capacityWh := usableCapwh, instantWh := whInstant, chargeCompleted := mainChargeComplete, memoryWrite := @C(223).OR, SOC => SoCreal, remainingWh => usableRemWh, state => testSocState);
    TO_USINT(IN := SOCisz1.SOC, TO_USINT => SoC_CC);
    DIV(IN1 := SOCisz1.remainingWh, IN2 := 1000, DIV => usableRemkwh);

    // Network 122:
    R_TRIG2(CLK := mainChargeComplete);
    SEL(G := R_TRIG2.Q, IN0 := socChComp, IN1 := SoCreal, SEL => socChComp);

    // Network 123:
    LT(IN1 := Cell_Voltage_Min, IN2 := cellVolt_dischargeOK, LT => @C(246).LT);
    LT(IN1 := Total_Voltage, IN2 := DichargeOK_Voltage_PACK, LT => @C(1324).LT);
    OR(IN1 := @C(246).LT, IN2 := @C(1324).LT, OR => @C(906).OR);
    SUB(IN1 := SoCreal, IN2 := socDchComp, SUB => @C(944).SUB);
    GT(IN1 := @C(944).SUB, IN2 := 4, GT => @C(926).GT);
    LT(IN1 := BatteryCurrent, IN2 := 10, LT => @C(341).LT);
    AND(IN1 := @C(906).OR, IN2 := @C(341).LT, AND => @C(328).AND);
    Tbuffer6(I := @C(328).AND, D := T#500ms);
    SR2(S1 := Tbuffer6.O, R := @C(926).GT, Q1 => dischargeComplete);

    // Network 124:
    R_TRIG3(CLK := dischargeComplete);
    SEL(G := R_TRIG3.Q, IN0 := socDchComp, IN1 := SoCreal, SEL => socDchComp);

    // Network 125:
    EQ(IN1 := BMS_State, IN2 := BATTSTATE#CHARGE, EQ => @C(793).EQ);
    chargeState1(chargeOn := @C(793).EQ, mainComplete := mainChargeComplete, dmcc := BMSdmcc_main, battAmpr := BatteryCurrent, balAmpr := 1, balDiff := BalanceDiff_Threshold, maxCell := Cell_Voltage_Max, minCell := Cell_Voltage_Min, complete => BCU_Charge_Complete, balance => BalanceStateEnb, chargeAmpr => BMSdmcc_final, chState => balChargeSt);

    // Network 126:
    Balance_isz1(Max_Cell_Voltage := Cell_Voltage_Max, Min_Cell_Voltage := Cell_Voltage_Min, Avarage_Cell_Voltage := Cell_Voltage_Average, Charge_Status := BalanceStateEnb, Ballance_Interval := T#15s, Difference_Tolerance := 10, Balance_Threshold := cellVolt_balThres, Balance_Enable => Balance_Enable_Rq, Measure_All => Measure_All, Measure_Aux => Measure_Aux, Ballance_Voltage => Balance_Voltage);

    // Network 127:
    TO_UINT(IN := BMSdmcc_final, TO_UINT => Pack_DMCC);

    // Network 128:
    AND(IN1 := prechargeEnable, IN2 := NOT prechargeBoardErr, AND => @C(1083).AND);
    prechargeCAN1(CAN_CH := PDUCAN, ENB := prechargeEnable, RST := NOT @C(1083).AND, CANerr => prechargeBoardErr);

    // Network 129:
    essState11(discharge := dischargeENB, charge := chargeENB, shutdown := shutdownEnb, prechargeOk := prechargeComplete, contactFbk := contactFbkCharge, contactFbkNeg := contactFbkDischarge, dischargeProtect := dischargeProtect, chargeProtect := chargeProtect, shutdownComplete := shutdownComplete, fault := FaultForState, STATE => BMS_State, prechargeOn => prechargeEnable, contact => contactEnable_batt, contactNeg => contactNegEnable_batt);

    // Network 130:
    OR(IN1 := contactEnable_batt, IN2 := contactNegEnable_batt, OR => AllcontacstEnable);

    // Network 131:
    new_CHG_CONTACT := contactEnable_batt;

    // Network 132:
    new_DCHG_CONTACT := contactNegEnable_batt;

    // Network 133:
    prechargeComplete := prechargeEnable;

    // Network 134:
    IOWR24(PORT := TMS570_GIO#HET1, PIN := 2, VAL := new_DCHG_CONTACT);

    // Network 135:
    IOWR10(PORT := TMS570_GIO#HET1, PIN := 0, VAL := new_CHG_CONTACT);

    // Network 136:
    EQ(IN1 := BMS_State, IN2 := BATTSTATE#DISCHARGE, EQ => @C(303).EQ);
    TON21(IN := @C(303).EQ, PT := T#5s, Q => dischargeAmpEnb);

    // Network 137:
    EQ(IN1 := BMS_State, IN2 := BATTSTATE#CHARGE, EQ => @C(1795).EQ);
    TON22(IN := @C(1795).EQ, PT := T#5s, Q => chargeAmpEnb);

    // Network 138:
    GE(IN1 := Cell_Voltage_Min, IN2 := cellVolt_dischargeOK, GE => @C(874).GE);
    AND(IN1 := @C(874).GE, IN2 := dischargeAmpEnb, AND => increaseDischargeAmp);

    // Network 139:
    LE(IN1 := Cell_Voltage_Max, IN2 := cellVolt_chargeOK, LE => @C(1847).LE);
    AND(IN1 := @C(1847).LE, IN2 := chargeAmpEnb, IN3 := NOT Balance_Enable_Rq, AND => increaseChargeAmp);

    // Network 140:
    LT(IN1 := BatteryVoltage, IN2 := Pack_Discharge_Voltage, LT => @C(1274).LT);
    OR(IN1 := OT_danger_risk, IN2 := UT_danger_risk, OR => @C(1450).OR);
    LE(IN1 := Cell_Voltage_Min, IN2 := cellVolt_minDischarge, LE => @C(1319).LE);
    AND(IN1 := @C(1319).LE, IN2 := dischargeAmpEnb, AND => @C(1640).AND);
    OR(IN1 := @C(1274).LT, IN2 := @C(1450).OR, IN3 := @C(1640).AND, OR => decreaseDischargeAmp);

    // Network 141:
    GT(IN1 := BatteryVoltage, IN2 := Pack_Charge_Voltage, GT => @C(2092).GT);
    GE(IN1 := Cell_Voltage_Max, IN2 := cellVolt_maxCharge, GE => @C(2028).GE);
    AND(IN1 := @C(2028).GE, IN2 := chargeAmpEnb, IN3 := NOT Balance_Enable_Rq, AND => @C(2103).AND);
    OR(IN1 := OT_danger_risk, IN2 := UT_danger_risk, OR => @C(2110).OR);
    OR(IN1 := @C(2092).GT, IN2 := @C(2103).AND, IN3 := @C(2110).OR, OR => decreaseChargeAmp);

    // Network 142:
    DIV(IN1 := maxDischargeAmp, IN2 := dischargeUnitAmp, DIV => @C(1762).DIV);
    TO_INT(IN := @C(1762).DIV, TO_INT => @C(1771).TO_INT);
    R_TRIG9(CLK := dischargeAmpEnb);
    F_TRIG4(CLK := dischargeAmpEnb);
    OR(IN1 := R_TRIG9.Q, IN2 := F_TRIG4.Q, OR => @C(2322).OR);
    UpDownCntTim1(CU := increaseDischargeAmp, CD := decreaseDischargeAmp, uPer := T#125ms, dPer := T#60ms, PV := @C(1771).TO_INT, RST := @C(2322).OR);
    TO_REAL(IN := UpDownCntTim1.CV, TO_REAL => @C(1780).TO_REAL);
    MUL(IN1 := @C(1780).TO_REAL, IN2 := dischargeUnitAmp, MUL => @C(1783).MUL);
    MAX(IN1 := 2, IN2 := @C(1783).MUL, MAX => @C(64).MAX);
    SEL(G := dischargeAmpEnb, IN0 := 2, IN1 := @C(64).MAX, SEL => BMSdmdc_final);

    // Network 143:
    DIV(IN1 := maxChargeAmp, IN2 := chargeUnitAmp, DIV => @C(1770).DIV);
    TO_INT(IN := @C(1770).DIV, TO_INT => @C(1772).TO_INT);
    R_TRIG8(CLK := chargeAmpEnb);
    F_TRIG3(CLK := chargeAmpEnb);
    OR(IN1 := R_TRIG8.Q, IN2 := F_TRIG3.Q, OR => @C(1887).OR);
    UpDownCntTim2(CU := increaseChargeAmp, CD := decreaseChargeAmp, uPer := T#125ms, dPer := T#60ms, PV := @C(1772).TO_INT, RST := @C(1887).OR);
    TO_REAL(IN := UpDownCntTim2.CV, TO_REAL => @C(1781).TO_REAL);
    MUL(IN1 := @C(1781).TO_REAL, IN2 := chargeUnitAmp, MUL => @C(1782).MUL);
    MAX(IN1 := 2, IN2 := @C(1782).MUL, MAX => @C(1848).MAX);
    SEL(G := chargeAmpEnb, IN0 := 2, IN1 := @C(1848).MAX, SEL => BMSdmcc_main);

    // Network 144:
    TO_UINT(IN := BMSdmdc_final, TO_UINT => Pack_DMDC);

  *)

  @C(1) : @FB(BATTSTACK1), @R(1330.0, 640.0, 310.0, 418.0), @I(@N(NBOARDS), @L(9.5)), @I(@N(BAUD), @L(29.5)), @I(@N(OVTHRES), @L(49.5)), @I(@N(UVTHRES), @L(69.5)), @I(@N(M_ALL_R), @L(89.5)), @I(@N(M_AUX_R), @L(109.5)), @I(@N(N_CELLS), @L(129.5)), @I(@N(T_CELLS), @L(149.5)), @I(@N(CHSEL), @L(169.5)), @I(@N(BRD), @L(189.5)), @I(@N(CELL), @L(209.5)), @I(@N(CH), @L(229.5)), @I(@N(BALV), @L(249.5)), @I(@N(BALENB), @L(269.5)), @I(@N(NTCBETA), @L(289.5)), @I(@N(NTCNOMT_KLV), @L(309.5)), @I(@N(NTCNOMR_OHM), @L(329.5)), @I(@N(ENB), @L(349.5)), @O(@N(N_BRD), @R(369.5)), @O(@N(VCH), @R(329.5)), @O(@N(VCELL), @R(269.5)), @O(@N(VAV), @R(129.5)), @O(@N(VMINCELL), @R(109.5)), @O(@N(VMAXCELL), @R(89.5)), @O(@N(VSTACK), @R(309.5)), @O(@N(MAXCELLBRD), @R(9.5)), @O(@N(MAXCELLNUM), @R(29.5)), @O(@N(MINCELLBRD), @R(49.5)), @O(@N(MINCELLNUM), @R(69.5)), @O(@N(BALREG), @R(349.5)), @O(@N(TEMPCELL), @R(289.5)), @O(@N(MAXTEMP), @R(229.5)), @O(@N(MINTEMP), @R(249.5)), @O(@N(MAXTEMPBRD), @R(149.5)), @O(@N(MAXTEMPCELL), @R(169.5)), @O(@N(MINTEMPBRD), @R(189.5)), @O(@N(MINTEMPCELL), @R(209.5)), @O(@N(FAULT), @R(389.5)), @O(@N(ERR), @R(409.5));
  @C(15) : @FB(GUICFG_INT3), @R(70.0, 90.0, 180.0, 38.0), @I(@N(CODE), @L(9.5)), @I(@N(R), @L(29.5)), @O(@N(VAL), @R(9.5));
  @C(32) : @FB(numOfCells1), @R(210.0, 490.0, 220.0, 38.0), @I(@N(numofBMU), @L(9.5)), @I(@N(cellMap), @L(29.5)), @O(@N(numofCell), @R(9.5));
  @C(81) : @FB(IOWR2), @R(1760.0, 570.0, 120.0, 58.0), @I(@N(PORT), @L(9.5)), @I(@N(PIN), @L(29.5)), @I(@N(VAL), @L(49.5));
  @C(97) : @FB(IOWR1), @R(1760.0, 510.0, 120.0, 58.0), @I(@N(PORT), @L(9.5)), @I(@N(PIN), @L(29.5)), @I(@N(VAL), @L(49.5));
  @C(104) : @FB(Max_Min_Voltage_Status1), @R(2220.0, 510.0, 500.0, 178.0), @I(@N(Max_Volt_BMU_Loc), @L(69.5)), @I(@N(Max_Volt_Cell_Loc), @L(49.5)), @I(@N(Min_Volt_BMU_Loc), @L(109.5)), @I(@N(Min_Volt_Cell_Loc), @L(89.5)), @I(@N(Max_Cell_Voltage), @L(149.5)), @I(@N(Min_Cell_Voltage), @L(169.5)), @I(@N(Average_Cell_Voltage), @L(129.5)), @I(@N(CAN_ID), @L(29.5)), @I(@N(CAN_CH), @L(9.5)), @O(@N(CAN_Error), @R(169.5));
  @C(125) : @FB(chargeState1), @R(430.0, 1700.0, 400.0, 158.0), @I(@N(chargeOn), @L(9.5)), @I(@N(mainComplete), @L(29.5)), @I(@N(dmcc), @L(49.5)), @I(@N(battAmpr), @L(69.5)), @I(@N(balAmpr), @L(89.5)), @I(@N(balDiff), @L(109.5)), @I(@N(maxCell), @L(129.5)), @I(@N(minCell), @L(149.5)), @O(@N(complete), @R(9.5)), @O(@N(balance), @R(29.5)), @O(@N(chargeAmpr), @R(49.5)), @O(@N(chState), @R(69.5));
  @C(146) : @FB(SOCisz1), @R(390.0, 1590.0, 340.0, 78.0), @I(@N(capacityWh), @L(9.5)), @I(@N(instantWh), @L(29.5)), @I(@N(chargeCompleted), @L(49.5)), @I(@N(memoryWrite), @L(69.5)), @O(@N(SOC), @R(9.5)), @O(@N(remainingWh), @R(29.5)), @O(@N(state), @R(49.5));
  @C(161) : @FB(TON6), @R(2300.0, 1710.0, 100.0, 38.0), @I(@N(IN), @L(9.5)), @I(@N(PT), @L(29.5)), @O(@N(Q), @R(9.5)), @O(@N(ET), @R(29.5));
  @C(218) : @FB(GUI1), @R(1670.0, 1090.0, 200.0, 218.0), @I(@N(Voltage), @L(49.5)), @I(@N(Current), @L(69.5)), @I(@N(Temp), @L(89.5)), @I(@N(Humidity), @L(109.5)), @I(@N(Fault), @L(129.5)), @I(@N(SoC), @L(9.5)), @I(@N(SoH), @L(29.5)), @I(@N(Cycle), @L(149.5)), @I(@N(State), @L(169.5)), @I(@N(ID), @L(189.5)), @I(@N(CH), @L(209.5));
  @C(234) : @FB(TON7), @R(2300.0, 1790.0, 100.0, 38.0), @I(@N(IN), @L(9.5)), @I(@N(PT), @L(29.5)), @O(@N(Q), @R(9.5)), @O(@N(ET), @R(29.5));
  @C(243) : @F(NE), @R(2090.0, 2080.0, 40.0, 38.0), BOOL, @I(@N(IN1), @L(9.5)), @I(@N(IN2), @L(29.5)), @O(@N(NE), @R(9.5));
  @C(279) : @F(GE), @R(2160.0, 1880.0, 40.0, 38.0), REAL, @I(@N(IN1), @L(9.5)), @I(@N(IN2), @L(29.5)), @O(@N(GE), @R(9.5));
  @C(277) : @F(ADD), @R(2100.0, 2000.0, 40.0, 38.0), REAL, @I(@N(IN1), @L(9.5)), @I(@N(IN2), @L(29.5)), @O(@N(ADD), @R(9.5));
  @C(276) : @F(SUB), @R(2100.0, 1900.0, 40.0, 38.0), REAL, @I(@N(IN1), @L(9.5)), @I(@N(IN2), @L(29.5)), @O(@N(SUB), @R(9.5));
  @C(281) : @FB(TOF12), @R(2300.0, 2240.0, 100.0, 38.0), @I(@N(IN), @L(9.5)), @I(@N(PT), @L(29.5)), @O(@N(Q), @R(9.5)), @O(@N(ET), @R(29.5));
  @C(286) : @F(LE), @R(2090.0, 2440.0, 40.0, 38.0), REAL, @I(@N(IN1), @L(9.5)), @I(@N(IN2), @L(29.5)), @O(@N(LE), @R(9.5));
  @C(258) : @FB(TOF13), @R(2300.0, 2320.0, 100.0, 38.0), @I(@N(IN), @L(9.5)), @I(@N(PT), @L(29.5)), @O(@N(Q), @R(9.5)), @O(@N(ET), @R(29.5));
  @C(259) : @F(OR), @R(2090.0, 2240.0, 40.0, 38.0), BOOL, @I(@N(IN1), @L(9.5)), @I(@N(IN2), @L(29.5)), @O(@N(OR), @R(9.5));
  @C(288) : @F(GE), @R(2090.0, 2360.0, 40.0, 38.0), REAL, @I(@N(IN1), @L(9.5)), @I(@N(IN2), @L(29.5)), @O(@N(GE), @R(9.5));
  @C(297) : @FB(TOF14), @R(2300.0, 2280.0, 100.0, 38.0), @I(@N(IN), @L(9.5)), @I(@N(PT), @L(29.5)), @O(@N(Q), @R(9.5)), @O(@N(ET), @R(29.5));
  @C(336) : @F(DIV), @R(760.0, 790.0, 40.0, 38.0), REAL, @I(@N(IN1), @L(9.5)), @I(@N(IN2), @L(29.5)), @O(@N(DIV), @R(9.5));
  @C(324) : @FB(TOF7), @R(2300.0, 2080.0, 100.0, 38.0), @I(@N(IN), @L(9.5)), @I(@N(PT), @L(29.5)), @O(@N(Q), @R(9.5)), @O(@N(ET), @R(29.5));
  @C(322) : @FB(Buffer21), @R(2170.0, 2080.0, 100.0, 18.0), @I(@N(I), @L(9.5)), @O(@N(O), @R(9.5));
  @C(369) : @FB(TOF5), @R(2300.0, 2440.0, 100.0, 38.0), @I(@N(IN), @L(9.5)), @I(@N(PT), @L(29.5)), @O(@N(Q), @R(9.5)), @O(@N(ET), @R(29.5));
  @C(368) : @FB(TOF4), @R(2300.0, 2480.0, 100.0, 38.0), @I(@N(IN), @L(9.5)), @I(@N(PT), @L(29.5)), @O(@N(Q), @R(9.5)), @O(@N(ET), @R(29.5));
  @C(364) : @F(GE), @R(2160.0, 1710.0, 40.0, 38.0), UDINT, @I(@N(IN1), @L(9.5)), @I(@N(IN2), @L(29.5)), @O(@N(GE), @R(9.5));
  @C(366) : @FB(TOF3), @R(2300.0, 2360.0, 100.0, 38.0), @I(@N(IN), @L(9.5)), @I(@N(PT), @L(29.5)), @O(@N(Q), @R(9.5)), @O(@N(ET), @R(29.5));
  @C(415) : @F(TO_UINT), @R(1460.0, 1610.0, 120.0, 18.0), UINT, @I(@N(IN), @L(9.5)), @O(@N(TO_UINT), @R(9.5));
  @C(413) : @FB(Balance_isz1), @R(430.0, 1870.0, 460.0, 138.0), @I(@N(Max_Cell_Voltage), @L(29.5)), @I(@N(Min_Cell_Voltage), @L(49.5)), @I(@N(Avarage_Cell_Voltage), @L(69.5)), @I(@N(Charge_Status), @L(9.5)), @I(@N(Ballance_Interval), @L(129.5)), @I(@N(Difference_Tolerance), @L(109.5)), @I(@N(Balance_Threshold), @L(89.5)), @O(@N(Balance_Enable), @R(9.5)), @O(@N(Measure_All), @R(49.5)), @O(@N(Measure_Aux), @R(69.5)), @O(@N(Ballance_Voltage), @R(29.5));
  @C(404) : @F(LE), @R(2160.0, 1790.0, 40.0, 38.0), UDINT, @I(@N(IN1), @L(9.5)), @I(@N(IN2), @L(29.5)), @O(@N(LE), @R(9.5));
  @C(405) : @FB(TOF2), @R(2300.0, 2400.0, 100.0, 38.0), @I(@N(IN), @L(9.5)), @I(@N(PT), @L(29.5)), @O(@N(Q), @R(9.5)), @O(@N(ET), @R(29.5));
  @C(395) : @FB(CAN_Test2), @R(1640.0, 1690.0, 200.0, 118.0), @I(@N(IN_1), @L(49.5)), @I(@N(IN_2), @L(69.5)), @I(@N(IN_3), @L(89.5)), @I(@N(IN_4), @L(109.5)), @I(@N(CAN_CH), @L(9.5)), @I(@N(CAN_ID), @L(29.5));
  @C(394) : @FB(Buffer12), @R(2170.0, 2200.0, 100.0, 18.0), @I(@N(I), @L(9.5)), @O(@N(O), @R(9.5));
  @C(393) : @FB(TOF1), @R(2300.0, 2200.0, 100.0, 38.0), @I(@N(IN), @L(9.5)), @I(@N(PT), @L(29.5)), @O(@N(Q), @R(9.5)), @O(@N(ET), @R(29.5));
  @C(388) : @FB(CAN_Test1), @R(1640.0, 1570.0, 200.0, 118.0), @I(@N(IN_1), @L(49.5)), @I(@N(IN_2), @L(69.5)), @I(@N(IN_3), @L(89.5)), @I(@N(IN_4), @L(109.5)), @I(@N(CAN_CH), @L(9.5)), @I(@N(CAN_ID), @L(29.5));
  @C(425) : @F(TO_UINT), @R(1460.0, 1790.0, 120.0, 18.0), BOOL, @I(@N(IN), @L(9.5)), @O(@N(TO_UINT), @R(9.5));
  @C(424) : @F(TO_UINT), @R(1460.0, 1770.0, 120.0, 18.0), UINT, @I(@N(IN), @L(9.5)), @O(@N(TO_UINT), @R(9.5));
  @C(419) : @F(TO_UINT), @R(1460.0, 1630.0, 120.0, 18.0), UINT, @I(@N(IN), @L(9.5)), @O(@N(TO_UINT), @R(9.5));
  @C(421) : @F(TO_UINT), @R(1460.0, 1670.0, 120.0, 18.0), UINT, @I(@N(IN), @L(9.5)), @O(@N(TO_UINT), @R(9.5));
  @C(420) : @F(TO_UINT), @R(1460.0, 1650.0, 120.0, 18.0), UINT, @I(@N(IN), @L(9.5)), @O(@N(TO_UINT), @R(9.5));
  @C(423) : @F(TO_UINT), @R(1460.0, 1750.0, 120.0, 18.0), UINT, @I(@N(IN), @L(9.5)), @O(@N(TO_UINT), @R(9.5));
  @C(422) : @F(TO_UINT), @R(1460.0, 1730.0, 120.0, 18.0), UINT, @I(@N(IN), @L(9.5)), @O(@N(TO_UINT), @R(9.5));
  @C(466) : @FB(CMS_IVT1), @R(140.0, 2760.0, 300.0, 278.0), @I(@N(CAN_CH), @L(9.5)), @O(@N(Current_mA), @R(9.5)), @O(@N(Voltage1_mV), @R(29.5)), @O(@N(Voltage2_mV), @R(49.5)), @O(@N(Voltage3_mV), @R(69.5)), @O(@N(Temp), @R(109.5)), @O(@N(Power_kWh), @R(129.5)), @O(@N(Current_Counter_Ah), @R(169.5)), @O(@N(Power_Counter_Wh), @R(189.5)), @O(@N(CMS_Error), @R(249.5)), @O(@N(CAN_Error), @R(269.5)), @O(@N(Overall_Power_kWh), @R(209.5));
  @C(509) : @F(DIV), @R(760.0, 750.0, 40.0, 38.0), REAL, @I(@N(IN1), @L(9.5)), @I(@N(IN2), @L(29.5)), @O(@N(DIV), @R(9.5));
  @C(502) : @F(MUL), @R(660.0, 750.0, 40.0, 38.0), REAL, @I(@N(IN1), @L(9.5)), @I(@N(IN2), @L(29.5)), @O(@N(MUL), @R(9.5));
  @C(548) : @FB(TON16), @R(500.0, 1360.0, 100.0, 38.0), @I(@N(IN), @L(9.5)), @I(@N(PT), @L(29.5)), @O(@N(Q), @R(9.5)), @O(@N(ET), @R(29.5));
  @C(544) : @F(GE), @R(240.0, 1400.0, 40.0, 38.0), UDINT, @I(@N(IN1), @L(9.5)), @I(@N(IN2), @L(29.5)), @O(@N(GE), @R(9.5));
  @C(570) : @FB(BCU_Fault_Codes1), @R(3360.0, 1400.0, 300.0, 878.0), @I(@N(CAN_ID), @L(29.5)), @I(@N(Fault_00), @L(49.5)), @I(@N(Fault_01), @L(69.5)), @I(@N(Fault_02), @L(89.5)), @I(@N(Fault_03), @L(109.5)), @I(@N(Fault_04), @L(129.5)), @I(@N(Fault_05), @L(149.5)), @I(@N(Fault_06), @L(169.5)), @I(@N(Fault_07), @L(189.5)), @I(@N(Fault_08), @L(209.5)), @I(@N(Fault_09), @L(229.5)), @I(@N(Fault_10), @L(249.5)), @I(@N(Fault_11), @L(269.5)), @I(@N(Fault_12), @L(289.5)), @I(@N(Fault_13), @L(309.5)), @I(@N(Fault_14), @L(329.5)), @I(@N(Fault_15), @L(349.5)), @I(@N(Fault_16), @L(369.5)), @I(@N(Fault_17), @L(389.5)), @I(@N(Fault_18), @L(409.5)), @I(@N(Fault_19), @L(429.5)), @I(@N(Fault_20), @L(449.5)), @I(@N(Fault_21), @L(469.5)), @I(@N(Fault_22), @L(489.5)), @I(@N(Fault_23), @L(509.5)), @I(@N(Fault_24), @L(529.5)), @I(@N(Fault_25), @L(549.5)), @I(@N(Fault_26), @L(569.5)), @I(@N(Fault_27), @L(589.5)), @I(@N(Fault_28), @L(609.5)), @I(@N(Fault_29), @L(629.5)), @I(@N(Fault_30), @L(649.5)), @I(@N(Fault_31), @L(669.5)), @I(@N(Fault_32), @L(689.5)), @I(@N(Fault_33), @L(709.5)), @I(@N(Fault_34), @L(729.5)), @I(@N(Fault_35), @L(749.5)), @I(@N(Fault_36), @L(769.5)), @I(@N(Fault_37), @L(789.5)), @I(@N(Fault_38), @L(809.5)), @I(@N(Fault_39), @L(829.5)), @I(@N(Fault_Byte_5), @L(849.5)), @I(@N(CAN_CH), @L(9.5)), @I(@N(Fault_Byte_6_7), @L(869.5)), @O(@N(CAN_Error), @R(29.5)), @O(@N(GUI_Fault), @R(9.5)), @O(@N(sum), @R(49.5));
  @C(517) : @F(MUL), @R(660.0, 790.0, 40.0, 38.0), REAL, @I(@N(IN1), @L(9.5)), @I(@N(IN2), @L(29.5)), @O(@N(MUL), @R(9.5));
  @C(542) : @F(OR), @R(300.0, 1360.0, 40.0, 38.0), BOOL, @I(@N(IN1), @L(9.5)), @I(@N(IN2), @L(29.5)), @O(@N(OR), @R(9.5));
  @C(762) : @FB(CTU2), @R(540.0, 980.0, 100.0, 58.0), @I(@N(CU), @L(9.5)), @I(@N(R), @L(29.5)), @I(@N(PV), @L(49.5)), @O(@N(Q), @R(9.5)), @O(@N(CV), @R(49.5));
  @C(763) : @FB(CTU1), @R(340.0, 990.0, 100.0, 58.0), @I(@N(CU), @L(9.5)), @I(@N(R), @L(29.5)), @I(@N(PV), @L(49.5)), @O(@N(Q), @R(9.5)), @O(@N(CV), @R(49.5));
  @C(766) : @F(TO_USINT), @R(650.0, 1030.0, 120.0, 18.0), INT, @I(@N(IN), @L(9.5)), @O(@N(TO_USINT), @R(9.5));
  @C(765) : @F(TO_USINT), @R(650.0, 1010.0, 120.0, 18.0), INT, @I(@N(IN), @L(9.5)), @O(@N(TO_USINT), @R(9.5));
  @C(706) : @FB(FLASH1), @R(180.0, 990.0, 120.0, 38.0), @I(@N(IN), @L(9.5)), @I(@N(PER), @L(29.5)), @O(@N(OUT), @R(9.5));
  @C(728) : @FB(Buffer11), @R(2170.0, 2360.0, 100.0, 18.0), @I(@N(I), @L(9.5)), @O(@N(O), @R(9.5));
  @C(826) : @FB(Buffer9), @R(2170.0, 2440.0, 100.0, 18.0), @I(@N(I), @L(9.5)), @O(@N(O), @R(9.5));
  @C(800) : @FB(ISABELinit1), @R(140.0, 2720.0, 300.0, 38.0), @I(@N(CH), @L(9.5)), @I(@N(ENB), @L(29.5)), @O(@N(ERR), @R(9.5));
  @C(803) : @F(LT), @R(2170.0, 1400.0, 40.0, 38.0), UDINT, @I(@N(IN1), @L(9.5)), @I(@N(IN2), @L(29.5)), @O(@N(LT), @R(9.5));
  @C(815) : @FB(F_TRIG1), @R(180.0, 1650.0, 140.0, 18.0), @I(@N(CLK), @L(9.5)), @O(@N(Q), @R(9.5));
  @C(793) : @F(EQ), @R(200.0, 1700.0, 40.0, 38.0), USINT, @I(@N(IN1), @L(9.5)), @I(@N(IN2), @L(29.5)), @O(@N(EQ), @R(9.5));
  @C(778) : @F(DIV), @R(740.0, 2760.0, 40.0, 38.0), REAL, @I(@N(IN1), @L(9.5)), @I(@N(IN2), @L(29.5)), @O(@N(DIV), @R(9.5));
  @C(887) : @F(GE), @R(240.0, 1360.0, 40.0, 38.0), REAL, @I(@N(IN1), @L(9.5)), @I(@N(IN2), @L(29.5)), @O(@N(GE), @R(9.5));
  @C(895) : @FB(SR1), @R(660.0, 1360.0, 80.0, 38.0), @I(@N(S1), @L(9.5)), @I(@N(R), @L(29.5)), @O(@N(Q1), @R(9.5));
  @C(958) : @F(MUL), @R(660.0, 670.0, 40.0, 38.0), REAL, @I(@N(IN1), @L(9.5)), @I(@N(IN2), @L(29.5)), @O(@N(MUL), @R(9.5));
  @C(959) : @F(DIV), @R(760.0, 670.0, 40.0, 38.0), REAL, @I(@N(IN1), @L(9.5)), @I(@N(IN2), @L(29.5)), @O(@N(DIV), @R(9.5));
  @C(933) : @F(TO_USINT), @R(780.0, 1570.0, 120.0, 18.0), REAL, @I(@N(IN), @L(9.5)), @O(@N(TO_USINT), @R(9.5));
  @C(920) : @F(GE), @R(2100.0, 1940.0, 40.0, 38.0), REAL, @I(@N(IN1), @L(9.5)), @I(@N(IN2), @L(29.5)), @O(@N(GE), @R(9.5));
  @C(921) : @FB(TON10), @R(2300.0, 1880.0, 100.0, 38.0), @I(@N(IN), @L(9.5)), @I(@N(PT), @L(29.5)), @O(@N(Q), @R(9.5)), @O(@N(ET), @R(29.5));
  @C(919) : @F(LE), @R(2160.0, 1980.0, 40.0, 38.0), REAL, @I(@N(IN1), @L(9.5)), @I(@N(IN2), @L(29.5)), @O(@N(LE), @R(9.5));
  @C(1004) : @FB(BCU_Cell_Status1), @R(2220.0, 350.0, 500.0, 158.0), @I(@N(Selected_BMU_Loc), @L(89.5)), @I(@N(Selected_Cell_Loc), @L(109.5)), @I(@N(Cell_Voltage), @L(129.5)), @I(@N(Cell_Temp), @L(149.5)), @I(@N(CAN_ID), @L(29.5)), @I(@N(CAN_CH), @L(9.5)), @I(@N(Total_Voltage), @L(49.5)), @I(@N(Instant_Current), @L(69.5)), @O(@N(CAN_Error), @R(149.5));
  @C(997) : @FB(Buffer1), @R(2220.0, 1400.0, 100.0, 18.0), @I(@N(I), @L(9.5)), @O(@N(O), @R(9.5));
  @C(979) : @FB(BCU_ID1), @R(1400.0, 10.0, 290.0, 158.0), @I(@N(ADDR_BIT0), @L(9.5)), @I(@N(ADDR_BIT1), @L(29.5)), @I(@N(ADDR_BIT2), @L(49.5)), @O(@N(PACK_ID), @R(9.5)), @O(@N(CAN_ID_10), @R(29.5)), @O(@N(CAN_ID_11), @R(49.5)), @O(@N(CAN_ID_12), @R(69.5)), @O(@N(CAN_ID_13), @R(89.5)), @O(@N(CAN_ID_14), @R(109.5)), @O(@N(CAN_ID_15), @R(129.5)), @O(@N(CAN_ID_16), @R(149.5));
  @C(971) : @F(MUL), @R(660.0, 710.0, 40.0, 38.0), REAL, @I(@N(IN1), @L(9.5)), @I(@N(IN2), @L(29.5)), @O(@N(MUL), @R(9.5));
  @C(975) : @F(DIV), @R(760.0, 710.0, 40.0, 38.0), REAL, @I(@N(IN1), @L(9.5)), @I(@N(IN2), @L(29.5)), @O(@N(DIV), @R(9.5));
  @C(972) : @F(TO_REAL), @R(510.0, 730.0, 120.0, 18.0), UINT, @I(@N(IN), @L(9.5)), @O(@N(TO_REAL), @R(9.5));
  @C(962) : @F(TO_REAL), @R(510.0, 690.0, 120.0, 18.0), UINT, @I(@N(IN), @L(9.5)), @O(@N(TO_REAL), @R(9.5));
  @C(1071) : @FB(Buffer19), @R(2170.0, 2280.0, 100.0, 18.0), @I(@N(I), @L(9.5)), @O(@N(O), @R(9.5));
  @C(1058) : @FB(TON11), @R(2300.0, 1980.0, 100.0, 38.0), @I(@N(IN), @L(9.5)), @I(@N(PT), @L(29.5)), @O(@N(Q), @R(9.5)), @O(@N(ET), @R(29.5));
  @C(1060) : @FB(TON12), @R(2300.0, 1940.0, 100.0, 38.0), @I(@N(IN), @L(9.5)), @I(@N(PT), @L(29.5)), @O(@N(Q), @R(9.5)), @O(@N(ET), @R(29.5));
  @C(1073) : @F(LE), @R(2100.0, 2040.0, 40.0, 38.0), REAL, @I(@N(IN1), @L(9.5)), @I(@N(IN2), @L(29.5)), @O(@N(LE), @R(9.5));
  @C(1352) : @F(DIV), @R(760.0, 830.0, 40.0, 38.0), REAL, @I(@N(IN1), @L(9.5)), @I(@N(IN2), @L(29.5)), @O(@N(DIV), @R(9.5));
  @C(1353) : @F(MUL), @R(660.0, 830.0, 40.0, 38.0), REAL, @I(@N(IN1), @L(9.5)), @I(@N(IN2), @L(29.5)), @O(@N(MUL), @R(9.5));
  @C(1347) : @FB(TON13), @R(2300.0, 2040.0, 100.0, 38.0), @I(@N(IN), @L(9.5)), @I(@N(PT), @L(29.5)), @O(@N(Q), @R(9.5)), @O(@N(ET), @R(29.5));
  @C(1520) : @F(DIV), @R(740.0, 2840.0, 40.0, 38.0), REAL, @I(@N(IN1), @L(9.5)), @I(@N(IN2), @L(29.5)), @O(@N(DIV), @R(9.5));
  @C(1530) : @FB(GUICFG_INT2), @R(70.0, 50.0, 180.0, 38.0), @I(@N(CODE), @L(9.5)), @I(@N(R), @L(29.5)), @O(@N(VAL), @R(9.5));
  @C(1658) : @F(EQ), @R(3230.0, 370.0, 40.0, 38.0), USINT, @I(@N(IN1), @L(9.5)), @I(@N(IN2), @L(29.5)), @O(@N(EQ), @R(9.5));
  @C(1582) : @F(LE), @R(2160.0, 1830.0, 40.0, 38.0), UDINT, @I(@N(IN1), @L(9.5)), @I(@N(IN2), @L(29.5)), @O(@N(LE), @R(9.5));
  @C(1583) : @FB(TON9), @R(2300.0, 1830.0, 100.0, 38.0), @I(@N(IN), @L(9.5)), @I(@N(PT), @L(29.5)), @O(@N(Q), @R(9.5)), @O(@N(ET), @R(29.5));
  @C(1580) : @F(GE), @R(2160.0, 1750.0, 40.0, 38.0), UDINT, @I(@N(IN1), @L(9.5)), @I(@N(IN2), @L(29.5)), @O(@N(GE), @R(9.5));
  @C(1581) : @FB(TON8), @R(2300.0, 1750.0, 100.0, 38.0), @I(@N(IN), @L(9.5)), @I(@N(PT), @L(29.5)), @O(@N(Q), @R(9.5)), @O(@N(ET), @R(29.5));
  @C(1762) : @F(DIV), @R(240.0, 3550.0, 40.0, 38.0), REAL, @I(@N(IN1), @L(9.5)), @I(@N(IN2), @L(29.5)), @O(@N(DIV), @R(9.5));
  @C(1771) : @F(TO_INT), @R(300.0, 3550.0, 120.0, 18.0), REAL, @I(@N(IN), @L(9.5)), @O(@N(TO_INT), @R(9.5));
  @C(1770) : @F(DIV), @R(250.0, 3780.0, 40.0, 38.0), REAL, @I(@N(IN1), @L(9.5)), @I(@N(IN2), @L(29.5)), @O(@N(DIV), @R(9.5));
  @C(1772) : @F(TO_INT), @R(310.0, 3780.0, 120.0, 18.0), REAL, @I(@N(IN), @L(9.5)), @O(@N(TO_INT), @R(9.5));
  @C(1779) : @FB(R_TRIG8), @R(250.0, 3830.0, 140.0, 18.0), @I(@N(CLK), @L(9.5)), @O(@N(Q), @R(9.5));
  @C(1782) : @F(MUL), @R(840.0, 3770.0, 40.0, 38.0), REAL, @I(@N(IN1), @L(9.5)), @I(@N(IN2), @L(29.5)), @O(@N(MUL), @R(9.5));
  @C(1783) : @F(MUL), @R(840.0, 3540.0, 40.0, 38.0), REAL, @I(@N(IN1), @L(9.5)), @I(@N(IN2), @L(29.5)), @O(@N(MUL), @R(9.5));
  @C(1780) : @F(TO_REAL), @R(710.0, 3540.0, 120.0, 18.0), INT, @I(@N(IN), @L(9.5)), @O(@N(TO_REAL), @R(9.5));
  @C(1781) : @F(TO_REAL), @R(710.0, 3770.0, 120.0, 18.0), INT, @I(@N(IN), @L(9.5)), @O(@N(TO_REAL), @R(9.5));
  @C(1787) : @F(SEL), @R(1020.0, 3710.0, 120.0, 58.0), REAL, @I(@N(G), @L(9.5)), @I(@N(IN0), @L(29.5)), @I(@N(IN1), @L(49.5)), @O(@N(SEL), @R(9.5));
  @C(1790) : @F(SEL), @R(1010.0, 3480.0, 120.0, 58.0), REAL, @I(@N(G), @L(9.5)), @I(@N(IN0), @L(29.5)), @I(@N(IN1), @L(49.5)), @O(@N(SEL), @R(9.5));
  @C(1788) : @F(TO_UINT), @R(840.0, 3970.0, 120.0, 18.0), REAL, @I(@N(IN), @L(9.5)), @O(@N(TO_UINT), @R(9.5));
  @C(1789) : @F(TO_UINT), @R(840.0, 3950.0, 120.0, 18.0), REAL, @I(@N(IN), @L(9.5)), @O(@N(TO_UINT), @R(9.5));
  @C(1702) : @F(AND), @R(360.0, 1360.0, 40.0, 38.0), BOOL, @I(@N(IN1), @L(9.5)), @I(@N(IN2), @L(29.5)), @O(@N(AND), @R(9.5));
  @C(1706) : @F(OR), @R(2340.0, 1500.0, 40.0, 38.0), BOOL, @I(@N(IN1), @L(9.5)), @I(@N(IN2), @L(29.5)), @O(@N(OR), @R(9.5));
  @C(1719) : @F(OR), @R(3380.0, 330.0, 40.0, 38.0), BOOL, @I(@N(IN1), @L(9.5)), @I(@N(IN2), @L(29.5)), @O(@N(OR), @R(9.5));
  @C(1713) : @F(EQ), @R(3230.0, 410.0, 40.0, 38.0), USINT, @I(@N(IN1), @L(9.5)), @I(@N(IN2), @L(29.5)), @O(@N(EQ), @R(9.5));
  @C(1669) : @F(LT), @R(2170.0, 1440.0, 40.0, 38.0), REAL, @I(@N(IN1), @L(9.5)), @I(@N(IN2), @L(29.5)), @O(@N(LT), @R(9.5));
  @C(1684) : @F(GT), @R(2170.0, 1500.0, 40.0, 38.0), UDINT, @I(@N(IN1), @L(9.5)), @I(@N(IN2), @L(29.5)), @O(@N(GT), @R(9.5));
  @C(1683) : @FB(Buffer2), @R(2220.0, 1500.0, 100.0, 18.0), @I(@N(I), @L(9.5)), @O(@N(O), @R(9.5));
  @C(1880) : @F(DIV), @R(740.0, 2880.0, 40.0, 38.0), REAL, @I(@N(IN1), @L(9.5)), @I(@N(IN2), @L(29.5)), @O(@N(DIV), @R(9.5));
  @C(1830) : @FB(Buffer4), @R(2220.0, 1550.0, 100.0, 18.0), @I(@N(I), @L(9.5)), @O(@N(O), @R(9.5));
  @C(1825) : @F(GT), @R(2170.0, 1550.0, 40.0, 38.0), REAL, @I(@N(IN1), @L(9.5)), @I(@N(IN2), @L(29.5)), @O(@N(GT), @R(9.5));
  @C(1819) : @F(OR), @R(2340.0, 1400.0, 40.0, 38.0), BOOL, @I(@N(IN1), @L(9.5)), @I(@N(IN2), @L(29.5)), @O(@N(OR), @R(9.5));
  @C(1817) : @FB(Buffer3), @R(2220.0, 1440.0, 100.0, 18.0), @I(@N(I), @L(9.5)), @O(@N(O), @R(9.5));
  @C(1813) : @F(OR), @R(2090.0, 2320.0, 40.0, 38.0), BOOL, @I(@N(IN1), @L(9.5)), @I(@N(IN2), @L(29.5)), @O(@N(OR), @R(9.5));
  @C(1985) : @F(DIV), @R(200.0, 1290.0, 40.0, 38.0), UINT, @I(@N(IN1), @L(9.5)), @I(@N(IN2), @L(29.5)), @O(@N(DIV), @R(9.5));
  @C(1990) : @F(SUB), @R(340.0, 1270.0, 40.0, 38.0), UINT, @I(@N(IN1), @L(9.5)), @I(@N(IN2), @L(29.5)), @O(@N(SUB), @R(9.5));
  @C(1995) : @F(TO_USINT), @R(730.0, 1250.0, 120.0, 18.0), UINT, @I(@N(IN), @L(9.5)), @O(@N(TO_USINT), @R(9.5));
  @C(1993) : @F(LIMIT), @R(600.0, 1250.0, 120.0, 58.0), UINT, @I(@N(MN), @L(9.5)), @I(@N(IN), @L(29.5)), @I(@N(MX), @L(49.5)), @O(@N(LIMIT), @R(9.5));
  @C(1981) : @F(TO_USINT), @R(260.0, 1250.0, 120.0, 18.0), LREAL, @I(@N(IN), @L(9.5)), @O(@N(TO_USINT), @R(9.5));
  @C(1978) : @F(DIV), @R(200.0, 1250.0, 40.0, 38.0), LREAL, @I(@N(IN1), @L(9.5)), @I(@N(IN2), @L(29.5)), @O(@N(DIV), @R(9.5));
  @VF(4) : @E(Cell_Voltage_Max_BMU_Loc), @R(1660.0, 640.0, 220.0, 19.0);
  @VF(5) : @E(Cell_Voltage_Max_Cell_Loc), @R(1660.0, 660.0, 220.0, 19.0);
  @VF(6) : @E(Cell_Voltage_Min_BMU_Loc), @R(1660.0, 680.0, 220.0, 19.0);
  @VF(7) : @E(Cell_Voltage_Min_Cell_Loc), @R(1660.0, 700.0, 220.0, 19.0);
  @VF(12) : @E(Cell_Voltage_Max), @R(1660.0, 720.0, 220.0, 19.0);
  @VF(17) : @E(Number_Of_BMU_cfg), @R(410.0, 90.0, 160.0, 19.0);
  @VF(16) : @E(1), @R(10.0, 110.0, 50.0, 19.0), BOOL;
  @VF(19) : @E(250000), @R(1210.0, 660.0, 100.0, 19.0), UDINT;
  @VF(18) : @E(Cell_Voltage), @R(1660.0, 900.0, 220.0, 19.0);
  @VF(20) : @E(261), @R(10.0, 90.0, 50.0, 19.0), UDINT;
  @VF(25) : @E(Cell_Temp), @R(1660.0, 920.0, 220.0, 19.0);
  @VF(24) : @E(NumOfCells), @R(1100.0, 760.0, 210.0, 19.0);
  @VF(26) : @E(ChannelSelect), @R(1100.0, 800.0, 210.0, 19.0);
  @VF(29) : @E(Total_Voltage), @R(1660.0, 940.0, 220.0, 19.0);
  @VF(28) : @E(Number_Of_Cell), @R(460.0, 490.0, 140.0, 19.0);
  @VF(30) : @E(Cell_Voltage_Min), @R(1660.0, 740.0, 220.0, 19.0);
  @VF(34) : @E(Number_Of_BMU_cfg), @R(20.0, 490.0, 160.0, 19.0);
  @VF(35) : @E(PLCHANNEL#AUX0), @R(1100.0, 860.0, 210.0, 19.0);
  @VF(39) : @E(Number_Of_BMU_cfg), @R(1110.0, 640.0, 200.0, 19.0);
  @VF(37) : @E(NumOfCells), @R(20.0, 510.0, 160.0, 19.0);
  @VF(40) : @E(1), @R(1210.0, 980.0, 100.0, 19.0), BOOL;
  @VF(48) : @E(Cell_Voltage_Average), @R(1660.0, 760.0, 220.0, 19.0);
  @VF(68) : @E(mainChargeComplete), @R(750.0, 1360.0, 170.0, 19.0);
  @VF(66) : @E(Cell_Voltage_Max), @R(230.0, 1890.0, 180.0, 19.0);
  @VF(72) : @E(Balance_Register), @R(1660.0, 980.0, 220.0, 19.0);
  @VF(85) : @E(Pack_DMDC), @R(1960.0, 170.0, 220.0, 19.0);
  @VF(87) : @E(Pack_DMCC), @R(1960.0, 190.0, 220.0, 19.0);
  @VF(94) : @E(Cell_Voltage_Max_Cell_Loc), @R(1960.0, 550.0, 220.0, 19.0);
  @VF(103) : @E(Cell_Voltage_Max_BMU_Loc), @R(1960.0, 570.0, 220.0, 19.0);
  @VF(100) : @E(TMS570_GIO#B), @R(1590.0, 570.0, 140.0, 19.0);
  @VF(101) : @E(1), @R(1590.0, 610.0, 140.0, 19.0), BOOL;
  @VF(98) : @E(0), @R(1590.0, 550.0, 140.0, 19.0), BOOL;
  @VF(99) : @E(3), @R(1590.0, 590.0, 140.0, 19.0), UINT;
  @VF(111) : @E(2500), @R(1530.0, 330.0, 80.0, 19.0), WORD;
  @VF(108) : @E(Cell_Voltage_Min_BMU_Loc), @R(1960.0, 610.0, 220.0, 19.0);
  @VF(105) : @E(Cell_Voltage_Min_Cell_Loc), @R(1960.0, 590.0, 220.0, 19.0);
  @VF(119) : @E(298.15), @R(1210.0, 940.0, 100.0, 19.0), REAL;
  @VF(115) : @E(Cell_Voltage_Min), @R(1960.0, 670.0, 220.0, 19.0);
  @VF(114) : @E(Cell_Voltage_Max), @R(1960.0, 650.0, 220.0, 19.0);
  @VF(113) : @E(Cell_Voltage_Average), @R(1960.0, 630.0, 220.0, 19.0);
  @VF(126) : @E(Selected_BMU_Loc), @R(1100.0, 820.0, 210.0, 19.0);
  @VF(124) : @E(cellVolt_chargeOK), @R(320.0, 690.0, 180.0, 19.0);
  @VF(122) : @E(CAN_ID_10), @R(1960.0, 70.0, 220.0, 19.0);
  @VF(121) : @E(10000.0), @R(1210.0, 960.0, 100.0, 19.0), REAL;
  @VF(143) : @E(BMS_State), @R(1960.0, 90.0, 220.0, 19.0);
  @VF(129) : @E(SoH), @R(860.0, 1250.0, 90.0, 19.0);
  @VF(154) : @E(Number_Of_BMU), @R(1660.0, 1000.0, 220.0, 19.0);
  @VF(156) : @E(BatteryCurrent), @R(250.0, 1760.0, 160.0, 19.0);
  @VF(157) : @E(cellVolt_max), @R(1640.0, 230.0, 150.0, 19.0);
  @VF(158) : @E(whInstant), @R(200.0, 1610.0, 170.0, 19.0);
  @VF(159) : @E(mainChargeComplete), @R(200.0, 1630.0, 170.0, 19.0);
  @VF(151) : @E(BCU_Charge_Complete), @R(850.0, 1700.0, 170.0, 19.0);
  @VF(168) : @E(3660), @R(1530.0, 230.0, 80.0, 19.0), WORD;
  @VF(172) : @E(SoC_CC), @R(910.0, 1570.0, 80.0, 19.0);
  @VF(160) : @E(BMS_State), @R(40.0, 1700.0, 150.0, 19.0);
  @VF(167) : @E(Cell_Voltage_Min_Disharge), @R(1100.0, 700.0, 210.0, 19.0);
  @VF(165) : @E(Cell_Voltage_Max_Charge), @R(1100.0, 680.0, 210.0, 19.0);
  @VF(164) : @E(cellVolt_dischargeOK), @R(320.0, 730.0, 180.0, 19.0);
  @VF(190) : @E(CAN_ID_12), @R(1960.0, 530.0, 220.0, 19.0);
  @VF(188) : @E(CAN_ID_11), @R(1960.0, 370.0, 220.0, 19.0);
  @VF(182) : @E(BatteryCurrent), @R(430.0, 2480.0, 130.0, 19.0);
  @VF(205) : @E(contactEnable_batt), @R(780.0, 2110.0, 190.0, 19.0);
  @VF(204) : @E(Cell_Temp_Min_Cell_Loc), @R(1960.0, 770.0, 220.0, 19.0);
  @VF(201) : @E(Balance_Enable_Rq), @R(1100.0, 900.0, 210.0, 19.0);
  @VF(203) : @E(Cell_Temp_Max_BMU_Loc), @R(1960.0, 750.0, 220.0, 19.0);
  @VF(202) : @E(Cell_Temp_Max_Cell_Loc), @R(1960.0, 730.0, 220.0, 19.0);
  @VF(220) : @E(CAN_ID_13), @R(1960.0, 710.0, 220.0, 19.0);
  @VF(216) : @E(Cell_Temp_Max), @R(1960.0, 810.0, 220.0, 19.0);
  @VF(219) : @E(Cell_Temp_Min), @R(1960.0, 830.0, 220.0, 19.0);
  @VF(215) : @E(Cell_Temp_Min_BMU_Loc), @R(1960.0, 790.0, 220.0, 19.0);
  @VF(235) : @E(Selected_Cell_Loc), @R(1100.0, 840.0, 210.0, 19.0);
  @VF(250) : @E(contactFbk), @R(1910.0, 2100.0, 140.0, 19.0);
  @VF(251) : @E(cellVolt_cutOffLow), @R(1640.0, 330.0, 160.0, 19.0);
  @VF(248) : @E(contactEnable), @R(1910.0, 2080.0, 140.0, 19.0);
  @VF(249) : @E(3400), @R(1530.0, 310.0, 80.0, 19.0), WORD;
  @VF(244) : @E(SoC_CC), @R(1960.0, 910.0, 220.0, 19.0);
  @VF(245) : @E(cellVolt_balThres), @R(1640.0, 310.0, 220.0, 19.0);
  @VF(275) : @E(cellTemp_maxLim), @R(1640.0, 430.0, 140.0, 19.0);
  @VF(274) : @E(Cell_Temp_Min), @R(1910.0, 2440.0, 140.0, 19.0);
  @VF(273) : @E(Cell_Temp_Max), @R(1910.0, 2360.0, 140.0, 19.0);
  @VF(278) : @E(Pack_Discharge_Voltage), @R(810.0, 790.0, 200.0, 19.0);
  @VF(282) : @E(cellTemp_warningOT), @R(1910.0, 2380.0, 140.0, 19.0);
  @VF(280) : @E(cellTemp_warningUT), @R(1910.0, 2460.0, 140.0, 19.0);
  @VF(284) : @E(56), @R(1530.0, 430.0, 70.0, 19.0), BYTE;
  @VF(262) : @E(UV_fault), @R(1910.0, 2340.0, 140.0, 19.0);
  @VF(263) : @E(UV_danger_risk), @R(1910.0, 2280.0, 140.0, 19.0);
  @VF(260) : @E(SoH), @R(1960.0, 930.0, 220.0, 19.0);
  @VF(261) : @E(T#3s), @R(2170.0, 2340.0, 100.0, 19.0);
  @VF(266) : @E(OV_danger_risk), @R(1910.0, 2200.0, 140.0, 19.0);
  @VF(267) : @E(UT_danger), @R(1910.0, 2480.0, 140.0, 19.0);
  @VF(264) : @E(UV_danger), @R(1910.0, 2320.0, 140.0, 19.0);
  @VF(270) : @E(cellVolt_dischargeOK), @R(1640.0, 410.0, 220.0, 19.0);
  @VF(268) : @E(OV_danger), @R(1910.0, 2240.0, 140.0, 19.0);
  @VF(269) : @E(cellVolt_minDischarge), @R(1640.0, 390.0, 220.0, 19.0);
  @VF(313) : @E(54), @R(1530.0, 450.0, 70.0, 19.0), BYTE;
  @VF(315) : @E(cellTemp_minLim), @R(1640.0, 470.0, 140.0, 19.0);
  @VF(316) : @E(-30), @R(1530.0, 470.0, 70.0, 19.0), SINT;
  @VF(319) : @E(-10), @R(1530.0, 490.0, 70.0, 19.0), SINT;
  @VF(318) : @E(cellTemp_warningUT), @R(1640.0, 490.0, 220.0, 19.0);
  @VF(291) : @E(cellTemp_warningOT), @R(1640.0, 450.0, 220.0, 19.0);
  @VF(292) : @E(OT_danger), @R(1910.0, 2400.0, 140.0, 19.0);
  @VF(295) : @E(cellVolt_maxCharge), @R(1640.0, 270.0, 220.0, 19.0);
  @VF(296) : @E(3640), @R(1530.0, 270.0, 80.0, 19.0), WORD;
  @VF(300) : @E(T#3s), @R(2170.0, 2300.0, 100.0, 19.0);
  @VF(340) : @E(Fault_Cell_Under_Temp_Danger), @R(2430.0, 2480.0, 260.0, 19.0);
  @VF(339) : @E(Fault_Cell_Under_Temp_Warning), @R(2430.0, 2440.0, 260.0, 19.0);
  @VF(338) : @E(Fault_Cell_Over_Temp_Danger), @R(2430.0, 2400.0, 260.0, 19.0);
  @VF(337) : @E(Fault_Cell_Over_Temp_Warning), @R(2430.0, 2360.0, 260.0, 19.0);
  @VF(346) : @E(Cell_Temp_Min), @R(1660.0, 880.0, 220.0, 19.0);
  @VF(344) : @E(Cell_Temp_Max), @R(1660.0, 860.0, 220.0, 19.0);
  @VF(325) : @E(T#3s), @R(2170.0, 2100.0, 100.0, 19.0);
  @VF(334) : @E(Fault_Cell_Under_Voltage_Warning), @R(2430.0, 2280.0, 260.0, 19.0);
  @VF(332) : @E(Fault_Cell_Over_Voltage_Warning), @R(2430.0, 2200.0, 260.0, 19.0);
  @VF(372) : @E(Board_Fault_Messages), @R(1660.0, 1020.0, 220.0, 19.0);
  @VF(371) : @E(T#3s), @R(2170.0, 2460.0, 100.0, 19.0);
  @VF(370) : @E(T#3s), @R(2170.0, 2500.0, 100.0, 19.0);
  @VF(361) : @E(Fault_Pack_Discharge_Contactor), @R(2430.0, 2080.0, 260.0, 19.0);
  @VF(414) : @E(Balance_Enable_Rq), @R(910.0, 1870.0, 220.0, 19.0);
  @VF(398) : @E(T#3s), @R(2170.0, 2220.0, 100.0, 19.0);
  @VF(391) : @E(16#10000002), @R(1460.0, 1710.0, 120.0, 19.0), UDINT;
  @VF(390) : @E(16#10000001), @R(1460.0, 1590.0, 120.0, 19.0), UDINT;
  @VF(389) : @E(BCU_CAN_CH), @R(1460.0, 1570.0, 120.0, 19.0);
  @VF(440) : @E(BMSdmcc_main), @R(250.0, 1740.0, 160.0, 19.0);
  @VF(441) : @E(CAN_ID_14), @R(1960.0, 890.0, 220.0, 19.0);
  @VF(445) : @E(Balance_Voltage), @R(1100.0, 880.0, 210.0, 19.0);
  @VF(447) : @E(Balance_Voltage), @R(910.0, 1890.0, 220.0, 19.0);
  @VF(2348) : @E(T#125ms), @R(350.0, 3740.0, 80.0, 19.0);
  @VF(2349) : @E(T#60ms), @R(350.0, 3760.0, 80.0, 19.0);
  @VF(2355) : @E(2), @R(840.0, 3730.0, 40.0, 19.0), REAL;
  @VF(478) : @E(Fault_Pack_CMS), @R(470.0, 3020.0, 220.0, 19.0);
  @VF(470) : @E(Cell_Voltage_Average), @R(230.0, 1930.0, 180.0, 19.0);
  @VF(465) : @E(Cell_Voltage_Min), @R(230.0, 1910.0, 180.0, 19.0);
  @VF(463) : @E(TMS570_GIO#A), @R(1590.0, 510.0, 140.0, 19.0);
  @VF(462) : @E(0), @R(1590.0, 530.0, 140.0, 19.0), UINT;
  @VF(506) : @E(Pack_Charge_Voltage), @R(810.0, 750.0, 200.0, 19.0);
  @VF(497) : @E(cellVolt_maxCharge), @R(320.0, 770.0, 180.0, 19.0);
  @VF(499) : @E(mainChargeComplete), @R(250.0, 1720.0, 160.0, 19.0);
  @VF(493) : @E(1000), @R(710.0, 810.0, 40.0, 19.0), REAL;
  @VF(492) : @E(BalanceStateEnb), @R(270.0, 1870.0, 140.0, 19.0);
  @VF(495) : @E(cellVolt_balThres), @R(230.0, 1950.0, 180.0, 19.0);
  @VF(485) : @E(1000), @R(710.0, 770.0, 40.0, 19.0), REAL;
  @VF(483) : @E(1000), @R(710.0, 730.0, 40.0, 19.0), REAL;
  @VF(550) : @E(3600), @R(1530.0, 290.0, 80.0, 19.0), WORD;
  @VF(551) : @E(Cell_Voltage_Max), @R(30.0, 1400.0, 190.0, 19.0);
  @VF(549) : @E(cellVolt_chargeOK), @R(1640.0, 290.0, 220.0, 19.0);
  @VF(558) : @E(CAN_Fault_07), @R(2110.0, 2550.0, 140.0, 19.0);
  @VF(556) : @E(Fault_CAN_Communication), @R(2410.0, 2530.0, 210.0, 19.0);
  @VF(575) : @E(BCU_Fault_Warning), @R(3060.0, 1440.0, 260.0, 19.0);
  @VF(574) : @E(CAN_ID_16), @R(3100.0, 1420.0, 220.0, 19.0);
  @VF(573) : @E(BCU_CAN_CH), @R(3100.0, 1400.0, 220.0, 19.0);
  @VF(572) : @E(Fault_Cell_Under_Voltage_Warning), @R(3060.0, 1520.0, 260.0, 19.0);
  @VF(571) : @E(Fault_Cell_Over_Voltage_Warning), @R(3060.0, 1480.0, 260.0, 19.0);
  @VF(516) : @E(3050), @R(1530.0, 410.0, 80.0, 19.0), WORD;
  @VF(519) : @E(2720), @R(1530.0, 350.0, 80.0, 19.0), WORD;
  @VF(514) : @E(cellVolt_min), @R(1640.0, 350.0, 150.0, 19.0);
  @VF(515) : @E(3000), @R(1530.0, 390.0, 80.0, 19.0), WORD;
  @VF(524) : @E(CMD_Voltage_Sense_2), @R(460.0, 2800.0, 170.0, 19.0);
  @VF(525) : @E(CMD_Voltage_Sense_3), @R(460.0, 2820.0, 170.0, 19.0);
  @VF(523) : @E(CMD_Voltage_Sense_1), @R(460.0, 2780.0, 170.0, 19.0);
  @VF(532) : @E(Measure_All), @R(910.0, 1910.0, 220.0, 19.0);
  @VF(534) : @E(Measure_Aux), @R(910.0, 1930.0, 220.0, 19.0);
  @VF(530) : @E(T#15s), @R(330.0, 1990.0, 80.0, 19.0);
  @VF(537) : @E(Measure_Aux), @R(1100.0, 740.0, 210.0, 19.0);
  @VF(536) : @E(Measure_All), @R(1100.0, 720.0, 210.0, 19.0);
  @VF(610) : @E(Cell_Current_Nominal), @R(410.0, 50.0, 180.0, 19.0);
  @VF(638) : @E(BCU_CAN_CH), @R(1960.0, 50.0, 220.0, 19.0);
  @VF(636) : @E(tauxCells), @R(1100.0, 780.0, 210.0, 19.0);
  @VF(576) : @E(BCU_Fault_Danger), @R(3060.0, 1460.0, 260.0, 19.0);
  @VF(577) : @E(Fault_Cell_Over_Temp_Warning), @R(3060.0, 1560.0, 260.0, 19.0);
  @VF(578) : @E(Fault_Cell_Over_Temp_Danger), @R(3060.0, 1580.0, 260.0, 19.0);
  @VF(579) : @E(Fault_Cell_Under_Temp_Warning), @R(3060.0, 1600.0, 260.0, 19.0);
  @VF(581) : @E(Number_Of_Parallel_Cell), @R(410.0, 10.0, 200.0, 19.0);
  @VF(583) : @E(Fault_Cell_Under_Temp_Danger), @R(3060.0, 1620.0, 260.0, 19.0);
  @VF(584) : @E(CMD_Current_Sense), @R(460.0, 2760.0, 170.0, 19.0);
  @VF(587) : @E(Fault_DMDC_Exceed), @R(3130.0, 2010.0, 180.0, 19.0);
  @VF(588) : @E(Fault_DMCC_Exceed), @R(3140.0, 2030.0, 180.0, 19.0);
  @VF(589) : @E(Fault_Pack_CMS), @R(3060.0, 1680.0, 260.0, 19.0);
  @VF(590) : @E(Fault_Pack_Discharge_Contactor), @R(3060.0, 1700.0, 260.0, 19.0);
  @VF(591) : @E(Fault_Pack_Charge_Contactor), @R(3060.0, 1720.0, 260.0, 19.0);
  @VF(593) : @E(T#3s), @R(2170.0, 2420.0, 100.0, 19.0);
  @VF(594) : @E(Fault_Pack_HVIL_1), @R(3060.0, 1740.0, 260.0, 19.0);
  @VF(596) : @E(Board_Fault_Messages), @R(3060.0, 2260.0, 260.0, 19.0);
  @VF(602) : @E(T#3s), @R(2170.0, 2380.0, 100.0, 19.0);
  @VF(605) : @E(cellVolt_nominal), @R(1640.0, 170.0, 220.0, 19.0);
  @VF(606) : @E(3200), @R(1530.0, 170.0, 80.0, 19.0), WORD;
  @VF(679) : @E(Board_Error_Messages), @R(3060.0, 2240.0, 260.0, 19.0);
  @VF(678) : @E(CMD_Counter_Current), @R(460.0, 2920.0, 170.0, 19.0);
  @VF(677) : @E(T#3s), @R(2170.0, 2260.0, 100.0, 19.0);
  @VF(676) : @E(Total_Voltage), @R(2040.0, 390.0, 140.0, 19.0);
  @VF(693) : @E(Number_Of_Cell), @R(360.0, 670.0, 140.0, 19.0);
  @VF(653) : @E(Total_Voltage), @R(30.0, 1360.0, 190.0, 19.0);
  @VF(654) : @E(Board_Error_Messages), @R(1660.0, 1040.0, 220.0, 19.0);
  @VF(664) : @E(CMD_Power), @R(460.0, 2880.0, 170.0, 19.0);
  @VF(660) : @E(Fault_Pack_HVIL_2), @R(3060.0, 1760.0, 260.0, 19.0);
  @VF(663) : @E(CMD_Temp), @R(460.0, 2860.0, 170.0, 19.0);
  @VF(746) : @E(CAN_Fault_05), @R(2730.0, 830.0, 120.0, 19.0);
  @VF(745) : @E(CAN_Fault_04), @R(2740.0, 670.0, 120.0, 19.0);
  @VF(736) : @E(Fault_CAN_Communication), @R(3060.0, 2100.0, 260.0, 19.0);
  @VF(743) : @E(CAN_Fault_02), @R(2730.0, 190.0, 120.0, 19.0);
  @VF(767) : @E(1), @R(350.0, 1780.0, 60.0, 19.0), REAL;
  @VF(709) : @E(cellVolt_minDischarge), @R(320.0, 810.0, 180.0, 19.0);
  @VF(824) : @E(1), @R(20.0, 2740.0, 80.0, 19.0), BOOL;
  @VF(814) : @E(IGNITION), @R(30.0, 1650.0, 130.0, 19.0);
  @VF(786) : @E(Selected_Cell_Loc), @R(780.0, 1030.0, 160.0, 19.0);
  @VF(785) : @E(Selected_BMU_Loc), @R(780.0, 1010.0, 160.0, 19.0);
  @VF(797) : @E(BMS_State), @R(780.0, 2050.0, 160.0, 19.0);
  @VF(792) : @E(BATTSTATE#CHARGE), @R(40.0, 1720.0, 150.0, 19.0), USINT;
  @VF(774) : @E(T#250ms), @R(80.0, 1010.0, 80.0, 19.0);
  @VF(772) : @E(BalanceStateEnb), @R(850.0, 1720.0, 170.0, 19.0);
  @VF(773) : @E(balChargeSt), @R(850.0, 1760.0, 170.0, 19.0);
  @VF(768) : @E(1), @R(110.0, 990.0, 50.0, 19.0), BOOL;
  @VF(769) : @E(Cell_Voltage_Max), @R(230.0, 1820.0, 180.0, 19.0);
  @VF(780) : @E(CAN_Fault_06), @R(2730.0, 990.0, 120.0, 19.0);
  @VF(781) : @E(1000), @R(660.0, 2790.0, 40.0, 19.0), REAL;
  @VF(779) : @E(BatteryCurrent), @R(800.0, 2760.0, 140.0, 19.0);
  @VF(877) : @E(3670), @R(1530.0, 210.0, 80.0, 19.0), WORD;
  @VF(862) : @E(GUI_Fault), @R(3440.0, 1350.0, 220.0, 19.0);
  @VF(860) : @E(cellVolt_cutOffHigh), @R(1640.0, 210.0, 200.0, 19.0);
  @VF(832) : @E(cellVolt_chargeOK), @R(30.0, 1420.0, 190.0, 19.0);
  @VF(954) : @E(ChargeOK_Voltage_PACK), @R(810.0, 670.0, 200.0, 19.0);
  @VF(955) : @E(DichargeOK_Voltage_PACK), @R(810.0, 710.0, 200.0, 19.0);
  @VF(929) : @E(Fault_Cell_Over_Voltage_Danger), @R(3060.0, 1500.0, 260.0, 19.0);
  @VF(928) : @E(Fault_Cell_Under_Voltage_Danger), @R(3060.0, 1540.0, 260.0, 19.0);
  @VF(924) : @E(Fault_Cell_Over_Voltage_Danger), @R(2430.0, 2240.0, 260.0, 19.0);
  @VF(925) : @E(Fault_Cell_Under_Voltage_Danger), @R(2430.0, 2320.0, 260.0, 19.0);
  @VF(993) : @E(CAN_ID_10), @R(1710.0, 30.0, 180.0, 19.0);
  @VF(992) : @E(CAN_ID_11), @R(1710.0, 50.0, 180.0, 19.0);
  @VF(995) : @E(CAN_ID_15), @R(1710.0, 130.0, 180.0, 19.0);
  @VF(994) : @E(CAN_ID_14), @R(1710.0, 110.0, 180.0, 19.0);
  @VF(996) : @E(CAN_ID_16), @R(1710.0, 150.0, 180.0, 19.0);
  @VF(986) : @E(Duty_Cycle), @R(390.0, 1250.0, 110.0, 19.0);
  @VF(984) : @E(CMD_Overall_Power), @R(20.0, 1250.0, 160.0, 19.0);
  @VF(990) : @E(Duty_Cycle), @R(1960.0, 950.0, 220.0, 19.0);
  @VF(988) : @E(CAN_ID_12), @R(1710.0, 70.0, 180.0, 19.0);
  @VF(982) : @E(CMD_Overall_Power), @R(460.0, 2960.0, 170.0, 19.0);
  @VF(980) : @E(Selected_Pack_Number), @R(1710.0, 10.0, 180.0, 19.0);
  @VF(981) : @E(CAN_ID_13), @R(1710.0, 90.0, 180.0, 19.0);
  @VF(968) : @E(1000), @R(710.0, 690.0, 40.0, 19.0), REAL;
  @VF(964) : @E(ChargeOK_Voltage_PACK), @R(30.0, 1380.0, 190.0, 19.0);
  @VF(1100) : @E(Cell_Temp_Min_Cell_Loc), @R(1660.0, 840.0, 220.0, 19.0);
  @VF(1101) : @E(Cell_Temp_Min_BMU_Loc), @R(1660.0, 820.0, 220.0, 19.0);
  @VF(1102) : @E(Cell_Temp_Max_BMU_Loc), @R(1660.0, 780.0, 220.0, 19.0);
  @VF(1103) : @E(Cell_Temp_Max_Cell_Loc), @R(1660.0, 800.0, 220.0, 19.0);
  @VF(1118) : @E(dischargeComplete), @R(1730.0, 1360.0, 160.0, 19.0);
  @VF(1128) : @E(Cell_Voltage), @R(1960.0, 470.0, 220.0, 19.0);
  @VF(1124) : @E(Selected_BMU_Loc), @R(1960.0, 430.0, 220.0, 19.0);
  @VF(1123) : @E(Selected_Cell_Loc), @R(1960.0, 450.0, 220.0, 19.0);
  @VF(1120) : @E(BatteryCurrent), @R(1960.0, 410.0, 220.0, 19.0);
  @VF(1147) : @E(Cell_Temp), @R(1960.0, 490.0, 220.0, 19.0);
  @VF(1141) : @E(Cell_Voltage_Min), @R(230.0, 1840.0, 180.0, 19.0);
  @VF(1038) : @E(BCU_CAN_CH), @R(1430.0, 1290.0, 220.0, 19.0);
  @VF(1050) : @E(cellVolt_cutOffLow), @R(1960.0, 1420.0, 160.0, 19.0);
  @VF(1056) : @E(Cell_Voltage_Min), @R(1960.0, 1400.0, 160.0, 19.0);
  @VF(1356) : @E(cellVolt_cutOffLow), @R(320.0, 850.0, 180.0, 19.0);
  @VF(1354) : @E(1000), @R(710.0, 850.0, 40.0, 19.0), REAL;
  @VF(1355) : @E(Pack_CutoffLow_Voltage), @R(810.0, 830.0, 200.0, 19.0);
  @VF(1348) : @E(1), @R(1960.0, 1920.0, 90.0, 19.0), REAL;
  @VF(1399) : @E(faultsWord), @R(3680.0, 1440.0, 110.0, 19.0);
  @VF(1389) : @E(Duty_Cycle), @R(1430.0, 1230.0, 220.0, 19.0);
  @VF(1390) : @E(BMS_State), @R(1430.0, 1250.0, 220.0, 19.0);
  @VF(1391) : @E(Selected_Pack_Number), @R(1430.0, 1270.0, 220.0, 19.0);
  @VF(1290) : @E(prechargeEnable), @R(780.0, 2090.0, 190.0, 19.0);
  @VF(1325) : @E(CAN_Fault_03), @R(2740.0, 490.0, 120.0, 19.0);
  @VF(1492) : @E(Pack_Temperature), @R(1430.0, 1170.0, 220.0, 19.0);
  @VF(1490) : @E(CMD_Current_Sense), @R(1430.0, 1150.0, 220.0, 19.0);
  @VF(1500) : @E(SoH), @R(1430.0, 1110.0, 220.0, 19.0);
  @VF(1498) : @E(CMD_Voltage_Sense_1), @R(1430.0, 1130.0, 220.0, 19.0);
  @VF(1499) : @E(GUI_Fault), @R(1430.0, 1210.0, 220.0, 19.0);
  @VF(1476) : @E(12), @R(10.0, 10.0, 50.0, 19.0), UDINT;
  @VF(1526) : @E(SoC_CC), @R(1430.0, 1090.0, 220.0, 19.0);
  @VF(1532) : @E(10), @R(10.0, 50.0, 50.0, 19.0), UDINT;
  @VF(1533) : @E(1), @R(10.0, 70.0, 50.0, 19.0), BOOL;
  @VF(1528) : @E(1), @R(10.0, 30.0, 50.0, 19.0), BOOL;
  @VF(1519) : @E(BatteryVoltage), @R(800.0, 2840.0, 140.0, 19.0);
  @VF(1659) : @E(Cell_Temp_Max), @R(1910.0, 1880.0, 140.0, 19.0);
  @VF(1663) : @E(1), @R(1960.0, 2020.0, 90.0, 19.0), REAL;
  @VF(1662) : @E(cellTemp_maxLim), @R(1910.0, 1900.0, 140.0, 19.0);
  @VF(1661) : @E(cellTemp_minLim), @R(1910.0, 2000.0, 140.0, 19.0);
  @VF(1660) : @E(Cell_Temp_Min), @R(1910.0, 1980.0, 140.0, 19.0);
  @VF(1575) : @E(T#100ms), @R(2210.0, 1730.0, 80.0, 19.0);
  @VF(1569) : @E(cellVolt_max), @R(1900.0, 1770.0, 150.0, 19.0);
  @VF(1594) : @E(UV_danger), @R(2420.0, 1830.0, 140.0, 19.0);
  @VF(1593) : @E(OV_danger), @R(2420.0, 1750.0, 140.0, 19.0);
  @VF(1591) : @E(T#20s), @R(2220.0, 1850.0, 70.0, 19.0);
  @VF(1588) : @E(T#20s), @R(2220.0, 1770.0, 70.0, 19.0);
  @VF(1564) : @E(T#100ms), @R(2210.0, 1810.0, 80.0, 19.0);
  @VF(1560) : @E(Cell_Voltage_Min), @R(1900.0, 1790.0, 150.0, 19.0);
  @VF(1556) : @E(UV_danger_risk), @R(2420.0, 1790.0, 140.0, 19.0);
  @VF(1559) : @E(cellVolt_min), @R(1900.0, 1850.0, 150.0, 19.0);
  @VF(1558) : @E(Cell_Voltage_Max), @R(1900.0, 1710.0, 150.0, 19.0);
  @VF(1555) : @E(OV_danger_risk), @R(2420.0, 1710.0, 140.0, 19.0);
  @VF(1730) : @E(BatteryCurrent), @R(30.0, 1440.0, 190.0, 19.0);
  @VF(1743) : @E(-5), @R(170.0, 1460.0, 50.0, 19.0), REAL;
  @VF(1751) : @E(contactFbk), @R(2070.0, 110.0, 110.0, 19.0);
  @VF(1701) : @E(BATTSTATE#CHARGE), @R(3000.0, 390.0, 170.0, 19.0), USINT;
  @VF(1699) : @E(OV_fault), @R(2390.0, 1500.0, 90.0, 19.0);
  @VF(1711) : @E(T#15s), @R(430.0, 1380.0, 50.0, 19.0);
  @VF(1718) : @E(IGNITION), @R(3440.0, 330.0, 140.0, 19.0);
  @VF(1715) : @E(BATTSTATE#DISCHARGE), @R(3000.0, 430.0, 170.0, 19.0), USINT;
  @VF(1668) : @E(T#2s), @R(2210.0, 1960.0, 80.0, 19.0);
  @VF(1671) : @E(T#2s), @R(2210.0, 2060.0, 80.0, 19.0);
  @VF(1670) : @E(UV_fault), @R(2390.0, 1400.0, 90.0, 19.0);
  @VF(1665) : @E(T#500ms), @R(2210.0, 1900.0, 80.0, 19.0);
  @VF(1666) : @E(T#500ms), @R(2210.0, 2000.0, 80.0, 19.0);
  @VF(1673) : @E(UT_danger_risk), @R(2420.0, 1980.0, 140.0, 19.0);
  @VF(1672) : @E(OT_danger_risk), @R(2420.0, 1880.0, 140.0, 19.0);
  @VF(1675) : @E(UT_danger), @R(2420.0, 2040.0, 140.0, 19.0);
  @VF(1674) : @E(OT_danger), @R(2420.0, 1940.0, 140.0, 19.0);
  @VF(1685) : @E(Cell_Voltage_Max), @R(1960.0, 1500.0, 160.0, 19.0);
  @VF(1695) : @E(cellVolt_cutOffHigh), @R(1960.0, 1520.0, 160.0, 19.0);
  @VF(1882) : @E(OutputVoltage), @R(800.0, 2880.0, 140.0, 19.0);
  @VF(1838) : @E(OV_fault), @R(1910.0, 2260.0, 140.0, 19.0);
  @VF(1829) : @E(BMSdmdc_final), @R(1150.0, 3480.0, 130.0, 19.0);
  @VF(1826) : @E(Pack_DMDC), @R(980.0, 3950.0, 140.0, 19.0);
  @VF(1827) : @E(Pack_DMCC), @R(980.0, 3970.0, 140.0, 19.0);
  @VF(1816) : @E(BMSdmcc_main), @R(1160.0, 3710.0, 120.0, 19.0);
  @VF(1815) : @E(BMSdmcc_final), @R(680.0, 3970.0, 140.0, 19.0);
  @VF(1814) : @E(BMSdmdc_final), @R(680.0, 3950.0, 140.0, 19.0);
  @VF(1810) : @E(2), @R(830.0, 3500.0, 40.0, 19.0), REAL;
  @VF(1806) : @E(T#60ms), @R(340.0, 3530.0, 80.0, 19.0);
  @VF(1805) : @E(T#125ms), @R(340.0, 3510.0, 80.0, 19.0);
  @VF(2000) : @E(0), @R(520.0, 1250.0, 60.0, 19.0), UINT;
  @VF(2006) : @E(testSocState), @R(910.0, 1630.0, 140.0, 19.0);
  @VF(1984) : @E(Duty_Cycle), @R(70.0, 1290.0, 110.0, 19.0);
  @VF(1989) : @E(100), @R(260.0, 1270.0, 60.0, 19.0), UINT;
  @VF(1998) : @E(100), @R(520.0, 1290.0, 60.0, 19.0), UINT;
  @VF(1977) : @E(kWhCapacity), @R(30.0, 1270.0, 150.0, 19.0);
  @CF(457) : @R(1020.0, 1740.0, 100.0, 19.0), @T("charger Amp");
  @CF(725) : @R(510.0, 2690.0, 370.0, 49.0), @T("sense_1: total voltage$Nsense_2: charge contactor (battery side)$Nsense_3: charge contactor (charge input side)");
  @CF(1842) : @R(740.0, 3500.0, 90.0, 19.0), @T("testAmper");
  @C(1419) : @FB(IOWR13), @R(3120.0, 2740.0, 120.0, 58.0), @I(@N(PORT), @L(9.5)), @I(@N(PIN), @L(29.5)), @I(@N(VAL), @L(49.5));
  @C(1344) : @FB(ANLG8), @R(3120.0, 2810.0, 120.0, 58.0), @I(@N(ADC), @L(9.5)), @I(@N(GRP), @L(29.5)), @I(@N(CH), @L(49.5)), @O(@N(VAL), @R(9.5));
  @VF(1420) : @E(TMS570_GIO#HET1), @R(2940.0, 2740.0, 140.0, 19.0);
  @VF(1421) : @E(24), @R(3020.0, 2760.0, 60.0, 19.0), UINT;
  @VF(1422) : @E(1), @R(3020.0, 2780.0, 60.0, 19.0), BOOL;
  @VF(1346) : @E(TMSADC#A1), @R(2960.0, 2810.0, 120.0, 19.0);
  @VF(1349) : @E(TMSADCGRP#G1), @R(2960.0, 2830.0, 120.0, 19.0);
  @VF(1351) : @E(10), @R(3020.0, 2850.0, 60.0, 19.0), USINT;
  @CF(1403) : @R(2960.0, 2850.0, 60.0, 19.0), @T("AIN8");
  @C(73) : @F(TO_REAL), @R(290.0, 1100.0, 120.0, 18.0), UDINT, @I(@N(IN), @L(9.5)), @O(@N(TO_REAL), @R(9.5));
  @C(74) : @F(MUL), @R(240.0, 1100.0, 40.0, 78.0), UDINT, @I(@N(IN1), @L(9.5)), @I(@N(IN2), @L(29.5)), @I(@N(IN3), @L(49.5)), @I(@N(IN4), @L(69.5)), @O(@N(MUL), @R(9.5));
  @C(75) : @F(DIV), @R(420.0, 1100.0, 40.0, 38.0), REAL, @I(@N(IN1), @L(9.5)), @I(@N(IN2), @L(29.5)), @O(@N(DIV), @R(9.5));
  @C(2073) : @F(MUL), @R(620.0, 1100.0, 40.0, 38.0), REAL, @I(@N(IN1), @L(9.5)), @I(@N(IN2), @L(29.5)), @O(@N(MUL), @R(9.5));
  @C(2077) : @F(DIV), @R(740.0, 1100.0, 40.0, 38.0), REAL, @I(@N(IN1), @L(9.5)), @I(@N(IN2), @L(29.5)), @O(@N(DIV), @R(9.5));
  @C(1367) : @F(MUL), @R(240.0, 1180.0, 40.0, 38.0), REAL, @I(@N(IN1), @L(9.5)), @I(@N(IN2), @L(29.5)), @O(@N(MUL), @R(9.5));
  @C(77) : @F(MUL), @R(380.0, 1200.0, 40.0, 38.0), REAL, @I(@N(IN1), @L(9.5)), @I(@N(IN2), @L(29.5)), @O(@N(MUL), @R(9.5));
  @VF(78) : @E(Number_Of_Cell), @R(90.0, 1100.0, 140.0, 19.0);
  @VF(79) : @E(Number_Of_Parallel_Cell), @R(30.0, 1120.0, 200.0, 19.0);
  @VF(80) : @E(Cell_Current_Nominal), @R(30.0, 1140.0, 200.0, 19.0);
  @VF(96) : @E(1000000), @R(310.0, 1120.0, 100.0, 19.0), REAL;
  @VF(102) : @E(cellVolt_nominal), @R(30.0, 1160.0, 200.0, 19.0);
  @VF(177) : @E(DoD_rate), @R(60.0, 1180.0, 160.0, 19.0);
  @VF(179) : @E(usableCapkwh), @R(450.0, 1180.0, 140.0, 19.0);
  @VF(2075) : @E(SoCreal), @R(510.0, 1120.0, 90.0, 19.0);
  @VF(186) : @E(usableCapwh), @R(450.0, 1200.0, 140.0, 19.0);
  @VF(2079) : @E(100), @R(680.0, 1120.0, 50.0, 19.0), REAL;
  @VF(2081) : @E(PackRemCap_kWh), @R(800.0, 1100.0, 140.0, 19.0);
  @VF(1452) : @E(1000), @R(310.0, 1220.0, 50.0, 19.0), REAL;
  @VF(183) : @E(kWhCapacity), @R(480.0, 1100.0, 120.0, 19.0);
  @VF(187) : @E(kWhCapacity), @R(100.0, 1200.0, 120.0, 19.0);
  @VF(456) : @E(DoD_rate), @R(1640.0, 190.0, 140.0, 19.0);
  @VF(460) : @E(0.90), @R(1530.0, 190.0, 80.0, 19.0), REAL;
  @VF(468) : @E(SoCreal), @R(910.0, 1590.0, 80.0, 19.0);
  @VF(2002) : @E(usableRemWh), @R(910.0, 1610.0, 140.0, 19.0);
  @VF(173) : @E(usableCapwh), @R(200.0, 1590.0, 170.0, 19.0);
  @VF(58) : @E(usableCapkwh), @R(2040.0, 970.0, 140.0, 19.0);
  @C(816) : @F(DIV), @R(770.0, 1650.0, 40.0, 38.0), REAL, @I(@N(IN1), @L(9.5)), @I(@N(IN2), @L(29.5)), @O(@N(DIV), @R(9.5));
  @VF(118) : @E(usableRemkwh), @R(910.0, 1650.0, 140.0, 19.0);
  @VF(120) : @E(1000), @R(670.0, 1670.0, 60.0, 19.0), REAL;
  @VF(133) : @E(usableRemkwh), @R(2040.0, 990.0, 140.0, 19.0);
  @VF(137) : @E(chargeCMD), @R(3440.0, 370.0, 140.0, 19.0);
  @VF(149) : @E(HVIL1_status), @R(2410.0, 3370.0, 140.0, 19.0);
  @VF(504) : @E(HVIL1_status), @R(1910.0, 2590.0, 140.0, 19.0);
  @C(505) : @FB(Buffer10), @R(2170.0, 2590.0, 100.0, 18.0), @I(@N(I), @L(9.5)), @O(@N(O), @R(9.5));
  @C(507) : @FB(TOF6), @R(2300.0, 2590.0, 100.0, 38.0), @I(@N(IN), @L(9.5)), @I(@N(PT), @L(29.5)), @O(@N(Q), @R(9.5)), @O(@N(ET), @R(29.5));
  @VF(511) : @E(Fault_Pack_HVIL_1), @R(2430.0, 2590.0, 220.0, 19.0);
  @VF(547) : @E(T#3s), @R(2220.0, 2610.0, 50.0, 19.0);
  @C(510) : @F(NOT), @R(2080.0, 2590.0, 60.0, 18.0), BOOL, @I(@N(IN), @L(9.5)), @O(@N(NOT), @R(9.5));
  @VF(628) : @E(BMSdmcc_final), @R(850.0, 1740.0, 140.0, 19.0);
  @VF(635) : @E(BMSdmcc_final), @R(1510.0, 1190.0, 140.0, 19.0);
  @CF(627) : @R(2340.0, 1440.0, 200.0, 29.0), @T("cut-off voltage faults");
  @VF(799) : @E(Number_Of_BMU_cfg), @R(20.0, 950.0, 180.0, 19.0);
  @VF(170) : @E(Pack_CutoffHigh_Voltage), @R(1920.0, 1570.0, 200.0, 19.0);
  @VF(458) : @E(Pack_CutoffLow_Voltage), @R(1920.0, 1460.0, 200.0, 19.0);
  @C(459) : @F(DIV), @R(760.0, 870.0, 40.0, 38.0), REAL, @I(@N(IN1), @L(9.5)), @I(@N(IN2), @L(29.5)), @O(@N(DIV), @R(9.5));
  @C(479) : @F(MUL), @R(660.0, 870.0, 40.0, 38.0), REAL, @I(@N(IN1), @L(9.5)), @I(@N(IN2), @L(29.5)), @O(@N(MUL), @R(9.5));
  @VF(521) : @E(1000), @R(710.0, 890.0, 40.0, 19.0), REAL;
  @VF(522) : @E(Pack_CutoffHigh_Voltage), @R(810.0, 870.0, 200.0, 19.0);
  @VF(586) : @E(cellVolt_cutOffHigh), @R(320.0, 890.0, 180.0, 19.0);
  @C(1161) : @FB(GUICFG_INT4), @R(90.0, 530.0, 180.0, 38.0), @I(@N(CODE), @L(9.5)), @I(@N(R), @L(29.5)), @O(@N(VAL), @R(9.5));
  @C(1169) : @F(TO_UINT), @R(280.0, 530.0, 120.0, 18.0), DINT, @I(@N(IN), @L(9.5)), @O(@N(TO_UINT), @R(9.5));
  @C(1538) : @F(TO_UINT), @R(280.0, 570.0, 120.0, 18.0), DINT, @I(@N(IN), @L(9.5)), @O(@N(TO_UINT), @R(9.5));
  @C(1539) : @FB(GUICFG_INT5), @R(90.0, 570.0, 180.0, 38.0), @I(@N(CODE), @L(9.5)), @I(@N(R), @L(29.5)), @O(@N(VAL), @R(9.5));
  @C(1184) : @F(MIN), @R(410.0, 530.0, 80.0, 38.0), UINT, @I(@N(IN1), @L(9.5)), @I(@N(IN2), @L(29.5)), @O(@N(MIN), @R(9.5));
  @C(1194) : @F(MIN), @R(410.0, 570.0, 80.0, 38.0), UINT, @I(@N(IN1), @L(9.5)), @I(@N(IN2), @L(29.5)), @O(@N(MIN), @R(9.5));
  @VF(1177) : @E(2001), @R(20.0, 530.0, 50.0, 19.0), UDINT;
  @VF(1179) : @E(1), @R(20.0, 550.0, 50.0, 19.0), BOOL;
  @VF(1541) : @E(2002), @R(20.0, 570.0, 50.0, 19.0), UDINT;
  @VF(1197) : @E(200), @R(330.0, 550.0, 50.0, 19.0), UINT;
  @VF(1199) : @E(300), @R(350.0, 590.0, 50.0, 19.0), UINT;
  @VF(1542) : @E(1), @R(20.0, 590.0, 50.0, 19.0), BOOL;
  @VF(912) : @E(maxDischargeAmprCfg), @R(500.0, 570.0, 160.0, 19.0);
  @C(932) : @F(NE), @R(2970.0, 2440.0, 40.0, 38.0), USINT, @I(@N(IN1), @L(9.5)), @I(@N(IN2), @L(29.5)), @O(@N(NE), @R(9.5));
  @C(1213) : @F(TO_DWORD), @R(2970.0, 2480.0, 120.0, 18.0), UDINT, @I(@N(IN), @L(9.5)), @O(@N(TO_DWORD), @R(9.5));
  @C(934) : @F(AND), @R(3140.0, 2520.0, 40.0, 38.0), DWORD, @I(@N(IN1), @L(9.5)), @I(@N(IN2), @L(29.5)), @O(@N(AND), @R(9.5));
  @C(1215) : @F(AND), @R(3140.0, 2480.0, 40.0, 38.0), DWORD, @I(@N(IN1), @L(9.5)), @I(@N(IN2), @L(29.5)), @O(@N(AND), @R(9.5));
  @C(1229) : @F(AND), @R(3140.0, 2560.0, 40.0, 38.0), DWORD, @I(@N(IN1), @L(9.5)), @I(@N(IN2), @L(29.5)), @O(@N(AND), @R(9.5));
  @C(935) : @FB(Tbuffer2), @R(3200.0, 2440.0, 120.0, 38.0), @I(@N(I), @L(9.5)), @I(@N(D), @L(29.5)), @O(@N(O), @R(9.5));
  @C(1227) : @F(TO_BOOL), @R(3200.0, 2560.0, 120.0, 18.0), DWORD, @I(@N(IN), @L(9.5)), @O(@N(TO_BOOL), @R(9.5));
  @C(1239) : @F(TO_BOOL), @R(3200.0, 2480.0, 120.0, 18.0), DWORD, @I(@N(IN), @L(9.5)), @O(@N(TO_BOOL), @R(9.5));
  @C(1233) : @F(TO_BOOL), @R(3200.0, 2520.0, 120.0, 18.0), DWORD, @I(@N(IN), @L(9.5)), @O(@N(TO_BOOL), @R(9.5));
  @C(1243) : @F(OR), @R(3340.0, 2500.0, 40.0, 58.0), BOOL, @I(@N(IN1), @L(9.5)), @I(@N(IN2), @L(29.5)), @I(@N(IN3), @L(49.5)), @O(@N(OR), @R(9.5));
  @C(1242) : @FB(Tbuffer7), @R(3450.0, 2500.0, 120.0, 38.0), @I(@N(I), @L(9.5)), @I(@N(D), @L(29.5)), @O(@N(O), @R(9.5));
  @C(1226) : @F(OR), @R(3590.0, 2440.0, 40.0, 48.0), BOOL, @I(@N(IN1), @L(9.5)), @I(@N(IN2), @L(29.5)), @O(@N(OR), @R(9.5));
  @VF(936) : @E(Number_Of_BMU), @R(2790.0, 2440.0, 160.0, 19.0);
  @VF(937) : @E(Number_Of_BMU_cfg), @R(2790.0, 2460.0, 160.0, 19.0);
  @VF(1212) : @E(Board_Error_Messages), @R(2770.0, 2480.0, 180.0, 19.0);
  @VF(1218) : @E(16#00000001), @R(2950.0, 2500.0, 140.0, 19.0), DWORD;
  @VF(1224) : @E(16#00000002), @R(2950.0, 2540.0, 140.0, 19.0), DWORD;
  @VF(938) : @E(T#3s), @R(3130.0, 2460.0, 50.0, 19.0);
  @VF(1230) : @E(16#00000004), @R(2950.0, 2580.0, 140.0, 19.0), DWORD;
  @VF(1950) : @E(T#3s), @R(3390.0, 2520.0, 50.0, 19.0);
  @VF(939) : @E(Fault_Pack_BMU), @R(3640.0, 2440.0, 140.0, 19.0);
  @VF(585) : @E(prechargeComplete), @R(150.0, 2130.0, 160.0, 19.0);
  @VF(651) : @E(cellVolt_warningOV), @R(1640.0, 250.0, 220.0, 19.0);
  @VF(652) : @E(3650), @R(1530.0, 250.0, 80.0, 19.0), WORD;
  @VF(553) : @E(cellVolt_warningOV), @R(1900.0, 1730.0, 150.0, 19.0);
  @VF(724) : @E(cellVolt_warningUV), @R(1640.0, 370.0, 220.0, 19.0);
  @VF(726) : @E(2730), @R(1530.0, 370.0, 80.0, 19.0), WORD;
  @VF(658) : @E(cellVolt_warningUV), @R(1900.0, 1810.0, 150.0, 19.0);
  @VF(822) : @E(PDUCAN), @R(20.0, 2720.0, 80.0, 19.0);
  @C(868) : @F(MIN), @R(410.0, 610.0, 80.0, 38.0), UINT, @I(@N(IN1), @L(9.5)), @I(@N(IN2), @L(29.5)), @O(@N(MIN), @R(9.5));
  @C(869) : @F(TO_UINT), @R(280.0, 610.0, 120.0, 18.0), DINT, @I(@N(IN), @L(9.5)), @O(@N(TO_UINT), @R(9.5));
  @C(870) : @FB(GUICFG_INT6), @R(90.0, 610.0, 180.0, 38.0), @I(@N(CODE), @L(9.5)), @I(@N(R), @L(29.5)), @O(@N(VAL), @R(9.5));
  @VF(872) : @E(250), @R(350.0, 630.0, 50.0, 19.0), UINT;
  @VF(875) : @E(2003), @R(20.0, 610.0, 50.0, 19.0), UDINT;
  @VF(876) : @E(1), @R(20.0, 630.0, 50.0, 19.0), BOOL;
  @VF(893) : @E(OCwarningAmpr), @R(500.0, 610.0, 140.0, 19.0);
  @VF(880) : @E(BatteryCurrent), @R(1910.0, 1610.0, 140.0, 19.0);
  @C(897) : @F(GE), @R(2160.0, 1610.0, 40.0, 38.0), REAL, @I(@N(IN1), @L(9.5)), @I(@N(IN2), @L(29.5)), @O(@N(GE), @R(9.5));
  @VF(900) : @E(OCwarningAmpr), @R(1910.0, 1630.0, 140.0, 19.0);
  @C(903) : @FB(Tbuffer1), @R(2300.0, 1610.0, 120.0, 38.0), @I(@N(I), @L(9.5)), @I(@N(D), @L(29.5)), @O(@N(O), @R(9.5));
  @VF(913) : @E(T#100ms), @R(2210.0, 1630.0, 80.0, 19.0);
  @VF(915) : @E(OC_warning), @R(2430.0, 1610.0, 110.0, 19.0);
  @C(917) : @F(GE), @R(2160.0, 1650.0, 40.0, 38.0), REAL, @I(@N(IN1), @L(9.5)), @I(@N(IN2), @L(29.5)), @O(@N(GE), @R(9.5));
  @VF(965) : @E(T#100ms), @R(2210.0, 1670.0, 80.0, 19.0);
  @C(961) : @FB(Tbuffer4), @R(2300.0, 1650.0, 120.0, 38.0), @I(@N(I), @L(9.5)), @I(@N(D), @L(29.5)), @O(@N(O), @R(9.5));
  @VF(970) : @E(OC_fault), @R(2430.0, 1650.0, 110.0, 19.0);
  @VF(977) : @E(Fault_Pack_BMU), @R(3190.0, 1840.0, 140.0, 19.0);
  @VF(991) : @E(isolationStatus), @R(2040.0, 230.0, 140.0, 19.0);
  @VF(999) : @E(contactNegEnable_batt), @R(780.0, 2130.0, 190.0, 19.0);
  @VF(694) : @E(ChargeInVoltage), @R(800.0, 2900.0, 140.0, 19.0);
  @VF(1048) : @E(prechargeError), @R(3190.0, 1880.0, 140.0, 19.0);
  @C(1092) : @F(NE), @R(2090.0, 2120.0, 40.0, 38.0), BOOL, @I(@N(IN1), @L(9.5)), @I(@N(IN2), @L(29.5)), @O(@N(NE), @R(9.5));
  @C(1093) : @FB(TOF8), @R(2300.0, 2120.0, 100.0, 38.0), @I(@N(IN), @L(9.5)), @I(@N(PT), @L(29.5)), @O(@N(Q), @R(9.5)), @O(@N(ET), @R(29.5));
  @C(1094) : @FB(Buffer22), @R(2170.0, 2120.0, 100.0, 18.0), @I(@N(I), @L(9.5)), @O(@N(O), @R(9.5));
  @VF(1095) : @E(T#3s), @R(2170.0, 2140.0, 100.0, 19.0);
  @VF(1096) : @E(contactFbkDischarge), @R(1910.0, 2140.0, 140.0, 19.0);
  @VF(1097) : @E(contactNegEnable), @R(1910.0, 2120.0, 160.0, 19.0);
  @VF(1098) : @E(Fault_Pack_Negative_Contactor), @R(2430.0, 2120.0, 260.0, 19.0);
  @C(1109) : @F(NE), @R(2090.0, 2160.0, 40.0, 38.0), BOOL, @I(@N(IN1), @L(9.5)), @I(@N(IN2), @L(29.5)), @O(@N(NE), @R(9.5));
  @C(1110) : @FB(TOF9), @R(2300.0, 2160.0, 100.0, 38.0), @I(@N(IN), @L(9.5)), @I(@N(PT), @L(29.5)), @O(@N(Q), @R(9.5)), @O(@N(ET), @R(29.5));
  @C(1111) : @FB(Buffer23), @R(2170.0, 2160.0, 100.0, 18.0), @I(@N(I), @L(9.5)), @O(@N(O), @R(9.5));
  @VF(1112) : @E(T#3s), @R(2170.0, 2180.0, 100.0, 19.0);
  @VF(1113) : @E(contactFbkCharge), @R(1910.0, 2180.0, 140.0, 19.0);
  @VF(1114) : @E(contactEnableCharge), @R(1910.0, 2160.0, 140.0, 19.0);
  @VF(1116) : @E(Fault_Pack_Charge_Contactor), @R(2430.0, 2160.0, 260.0, 19.0);
  @VF(1127) : @E(Fault_Pack_Negative_Contactor), @R(3070.0, 1860.0, 260.0, 19.0);
  @VF(1130) : @E(contactFbkDischarge), @R(2030.0, 210.0, 150.0, 19.0);
  @VF(1131) : @E(contactFbkCharge), @R(2030.0, 130.0, 150.0, 19.0);
  @VF(362) : @E(dischargeCMD), @R(3440.0, 410.0, 140.0, 19.0);
  @C(1258) : @F(ABS), @R(580.0, 2480.0, 60.0, 18.0), REAL, @I(@N(IN), @L(9.5)), @O(@N(ABS), @R(9.5));
  @C(1259) : @F(LT), @R(660.0, 2480.0, 40.0, 38.0), REAL, @I(@N(IN1), @L(9.5)), @I(@N(IN2), @L(29.5)), @O(@N(LT), @R(9.5));
  @VF(1262) : @E(3), @R(580.0, 2500.0, 60.0, 19.0), REAL;
  @VF(1264) : @E(shutdownComplete), @R(720.0, 2480.0, 160.0, 19.0);
  @VF(1266) : @E(shutdownComplete), @R(150.0, 2270.0, 150.0, 19.0);
  @VF(180) : @E(OC_fault), @R(3180.0, 1660.0, 140.0, 19.0);
  @VF(184) : @E(OC_warning), @R(3180.0, 1640.0, 140.0, 19.0);
  @OLT(1024) : @R(1010.0, 670.0, 80.0, 19.0), @S(954);
  @OLT(1025) : @R(1010.0, 710.0, 80.0, 19.0), @S(955);
  @OLT(1026) : @R(1010.0, 750.0, 80.0, 19.0), @S(506);
  @OLT(1027) : @R(1010.0, 790.0, 80.0, 19.0), @S(278);
  @OLT(1028) : @R(1010.0, 830.0, 80.0, 19.0), @S(1355);
  @OLT(1029) : @R(1010.0, 870.0, 80.0, 19.0), @S(522);
  @OLT(1031) : @R(510.0, 1080.0, 80.0, 19.0), @S(183);
  @OLT(1032) : @R(480.0, 1160.0, 80.0, 19.0), @S(179);
  @VF(76) : @E(Cell_Voltage_Min), @R(980.0, 1360.0, 200.0, 19.0);
  @C(246) : @F(LT), @R(1200.0, 1360.0, 40.0, 38.0), UDINT, @I(@N(IN1), @L(9.5)), @I(@N(IN2), @L(29.5)), @O(@N(LT), @R(9.5));
  @C(327) : @FB(Tbuffer6), @R(1490.0, 1360.0, 120.0, 38.0), @I(@N(I), @L(9.5)), @I(@N(D), @L(29.5)), @O(@N(O), @R(9.5));
  @VF(331) : @E(T#500ms), @R(1400.0, 1380.0, 80.0, 19.0);
  @C(341) : @F(LT), @R(1200.0, 1440.0, 40.0, 38.0), REAL, @I(@N(IN1), @L(9.5)), @I(@N(IN2), @L(29.5)), @O(@N(LT), @R(9.5));
  @VF(655) : @E(BatteryCurrent), @R(980.0, 1440.0, 200.0, 19.0);
  @C(328) : @F(AND), @R(1320.0, 1360.0, 40.0, 38.0), BOOL, @I(@N(IN1), @L(9.5)), @I(@N(IN2), @L(29.5)), @O(@N(AND), @R(9.5));
  @VF(323) : @E(cellVolt_dischargeOK), @R(980.0, 1380.0, 200.0, 19.0);
  @C(329) : @FB(SR2), @R(1640.0, 1360.0, 80.0, 38.0), @I(@N(S1), @L(9.5)), @I(@N(R), @L(29.5)), @O(@N(Q1), @R(9.5));
  @C(906) : @F(OR), @R(1260.0, 1360.0, 40.0, 38.0), BOOL, @I(@N(IN1), @L(9.5)), @I(@N(IN2), @L(29.5)), @O(@N(OR), @R(9.5));
  @VF(1322) : @E(Total_Voltage), @R(980.0, 1400.0, 200.0, 19.0);
  @C(1324) : @F(LT), @R(1200.0, 1400.0, 40.0, 38.0), REAL, @I(@N(IN1), @L(9.5)), @I(@N(IN2), @L(29.5)), @O(@N(LT), @R(9.5));
  @VF(1338) : @E(DichargeOK_Voltage_PACK), @R(980.0, 1420.0, 200.0, 19.0);
  @CF(840) : @R(2960.0, 2780.0, 60.0, 19.0), @T("AIN8on");
  @VF(335) : @E(HVCU_State), @R(3040.0, 370.0, 130.0, 19.0);
  @VF(241) : @E(inputSgn1Status), @R(2040.0, 310.0, 140.0, 19.0);
  @VF(242) : @E(inputSgn2Status), @R(2040.0, 330.0, 140.0, 19.0);
  @C(23) : @F(TO_UINT), @R(260.0, 50.0, 120.0, 18.0), DINT, @I(@N(IN), @L(9.5)), @O(@N(TO_UINT), @R(9.5));
  @C(61) : @F(TO_USINT), @R(260.0, 90.0, 120.0, 18.0), DINT, @I(@N(IN), @L(9.5)), @O(@N(TO_USINT), @R(9.5));
  @C(998) : @F(TO_UINT), @R(260.0, 130.0, 120.0, 18.0), DINT, @I(@N(IN), @L(9.5)), @O(@N(TO_UINT), @R(9.5));
  @C(1132) : @FB(GUICFG_INT7), @R(70.0, 130.0, 180.0, 38.0), @I(@N(CODE), @L(9.5)), @I(@N(R), @L(29.5)), @O(@N(VAL), @R(9.5));
  @VF(1133) : @E(101), @R(10.0, 130.0, 50.0, 19.0), UDINT;
  @VF(1134) : @E(1), @R(10.0, 150.0, 50.0, 19.0), BOOL;
  @VF(1394) : @E(cellVolt_cutOffHigh), @R(390.0, 130.0, 160.0, 19.0);
  @C(1401) : @F(TO_UINT), @R(260.0, 170.0, 120.0, 18.0), DINT, @I(@N(IN), @L(9.5)), @O(@N(TO_UINT), @R(9.5));
  @C(1402) : @FB(GUICFG_INT8), @R(70.0, 170.0, 180.0, 38.0), @I(@N(CODE), @L(9.5)), @I(@N(R), @L(29.5)), @O(@N(VAL), @R(9.5));
  @VF(1405) : @E(1), @R(10.0, 190.0, 50.0, 19.0), BOOL;
  @VF(1406) : @E(102), @R(10.0, 170.0, 50.0, 19.0), UDINT;
  @C(1426) : @F(TO_UINT), @R(260.0, 210.0, 120.0, 18.0), DINT, @I(@N(IN), @L(9.5)), @O(@N(TO_UINT), @R(9.5));
  @C(1428) : @FB(GUICFG_INT9), @R(70.0, 210.0, 180.0, 38.0), @I(@N(CODE), @L(9.5)), @I(@N(R), @L(29.5)), @O(@N(VAL), @R(9.5));
  @VF(1429) : @E(1), @R(10.0, 230.0, 50.0, 19.0), BOOL;
  @VF(1430) : @E(103), @R(10.0, 210.0, 50.0, 19.0), UDINT;
  @C(1466) : @F(TO_UINT), @R(260.0, 250.0, 120.0, 18.0), DINT, @I(@N(IN), @L(9.5)), @O(@N(TO_UINT), @R(9.5));
  @C(1468) : @FB(GUICFG_INT10), @R(70.0, 250.0, 180.0, 38.0), @I(@N(CODE), @L(9.5)), @I(@N(R), @L(29.5)), @O(@N(VAL), @R(9.5));
  @VF(1469) : @E(1), @R(10.0, 270.0, 50.0, 19.0), BOOL;
  @VF(1470) : @E(104), @R(10.0, 250.0, 50.0, 19.0), UDINT;
  @C(1477) : @F(TO_UINT), @R(260.0, 290.0, 120.0, 18.0), DINT, @I(@N(IN), @L(9.5)), @O(@N(TO_UINT), @R(9.5));
  @C(1478) : @FB(GUICFG_INT11), @R(70.0, 290.0, 180.0, 38.0), @I(@N(CODE), @L(9.5)), @I(@N(R), @L(29.5)), @O(@N(VAL), @R(9.5));
  @VF(1479) : @E(1), @R(10.0, 310.0, 50.0, 19.0), BOOL;
  @VF(1480) : @E(105), @R(10.0, 290.0, 50.0, 19.0), UDINT;
  @C(1486) : @F(TO_UINT), @R(260.0, 330.0, 120.0, 18.0), DINT, @I(@N(IN), @L(9.5)), @O(@N(TO_UINT), @R(9.5));
  @C(1487) : @FB(GUICFG_INT12), @R(70.0, 330.0, 180.0, 38.0), @I(@N(CODE), @L(9.5)), @I(@N(R), @L(29.5)), @O(@N(VAL), @R(9.5));
  @VF(1488) : @E(1), @R(10.0, 350.0, 50.0, 19.0), BOOL;
  @VF(1489) : @E(254), @R(10.0, 330.0, 50.0, 19.0), UDINT;
  @C(1497) : @F(TO_UINT), @R(260.0, 370.0, 120.0, 18.0), DINT, @I(@N(IN), @L(9.5)), @O(@N(TO_UINT), @R(9.5));
  @C(1501) : @FB(GUICFG_INT13), @R(70.0, 370.0, 180.0, 38.0), @I(@N(CODE), @L(9.5)), @I(@N(R), @L(29.5)), @O(@N(VAL), @R(9.5));
  @VF(1502) : @E(1), @R(10.0, 390.0, 50.0, 19.0), BOOL;
  @VF(1503) : @E(107), @R(10.0, 370.0, 50.0, 19.0), UDINT;
  @VF(1407) : @E(cellVolt_max), @R(390.0, 170.0, 150.0, 19.0);
  @VF(1431) : @E(cellVolt_maxCharge), @R(390.0, 210.0, 200.0, 19.0);
  @VF(1471) : @E(cellVolt_chargeOK), @R(390.0, 250.0, 190.0, 19.0);
  @VF(1481) : @E(cellVolt_warningOV), @R(390.0, 290.0, 170.0, 19.0);
  @VF(1491) : @E(cellVolt_balThres), @R(390.0, 330.0, 190.0, 19.0);
  @VF(1504) : @E(cellVolt_cutOffLow), @R(390.0, 370.0, 160.0, 19.0);
  @C(1509) : @F(TO_UINT), @R(260.0, 410.0, 120.0, 18.0), DINT, @I(@N(IN), @L(9.5)), @O(@N(TO_UINT), @R(9.5));
  @C(1510) : @FB(GUICFG_INT14), @R(70.0, 410.0, 180.0, 38.0), @I(@N(CODE), @L(9.5)), @I(@N(R), @L(29.5)), @O(@N(VAL), @R(9.5));
  @VF(1512) : @E(1), @R(10.0, 430.0, 50.0, 19.0), BOOL;
  @VF(1513) : @E(108), @R(10.0, 410.0, 50.0, 19.0), UDINT;
  @C(1534) : @F(TO_UINT), @R(260.0, 450.0, 120.0, 18.0), DINT, @I(@N(IN), @L(9.5)), @O(@N(TO_UINT), @R(9.5));
  @C(1537) : @FB(GUICFG_INT15), @R(70.0, 450.0, 180.0, 38.0), @I(@N(CODE), @L(9.5)), @I(@N(R), @L(29.5)), @O(@N(VAL), @R(9.5));
  @VF(1540) : @E(1), @R(10.0, 470.0, 50.0, 19.0), BOOL;
  @VF(1543) : @E(109), @R(10.0, 450.0, 50.0, 19.0), UDINT;
  @VF(1547) : @E(cellVolt_min), @R(390.0, 410.0, 150.0, 19.0);
  @VF(1549) : @E(cellVolt_minDischarge), @R(390.0, 450.0, 220.0, 19.0);
  @C(1551) : @FB(GUICFG_INT16), @R(690.0, 10.0, 180.0, 38.0), @I(@N(CODE), @L(9.5)), @I(@N(R), @L(29.5)), @O(@N(VAL), @R(9.5));
  @VF(1552) : @E(110), @R(630.0, 10.0, 50.0, 19.0), UDINT;
  @VF(1554) : @E(1), @R(630.0, 30.0, 50.0, 19.0), BOOL;
  @C(1567) : @F(TO_UINT), @R(890.0, 10.0, 120.0, 18.0), DINT, @I(@N(IN), @L(9.5)), @O(@N(TO_UINT), @R(9.5));
  @C(1570) : @FB(GUICFG_INT17), @R(690.0, 50.0, 180.0, 38.0), @I(@N(CODE), @L(9.5)), @I(@N(R), @L(29.5)), @O(@N(VAL), @R(9.5));
  @C(1574) : @F(TO_UINT), @R(890.0, 50.0, 120.0, 18.0), DINT, @I(@N(IN), @L(9.5)), @O(@N(TO_UINT), @R(9.5));
  @VF(1585) : @E(111), @R(630.0, 50.0, 50.0, 19.0), UDINT;
  @VF(1586) : @E(1), @R(630.0, 70.0, 50.0, 19.0), BOOL;
  @VF(1596) : @E(cellVolt_dischargeOK), @R(1020.0, 10.0, 220.0, 19.0);
  @VF(1605) : @E(cellVolt_warningUV), @R(1020.0, 50.0, 220.0, 19.0);
  @C(1608) : @FB(GUICFG_INT18), @R(690.0, 90.0, 180.0, 38.0), @I(@N(CODE), @L(9.5)), @I(@N(R), @L(29.5)), @O(@N(VAL), @R(9.5));
  @VF(1609) : @E(1), @R(630.0, 110.0, 50.0, 19.0), BOOL;
  @VF(1610) : @E(112), @R(630.0, 90.0, 50.0, 19.0), UDINT;
  @C(1613) : @F(TO_REAL), @R(890.0, 90.0, 120.0, 18.0), DINT, @I(@N(IN), @L(9.5)), @O(@N(TO_REAL), @R(9.5));
  @C(1615) : @FB(GUICFG_INT19), @R(690.0, 130.0, 180.0, 38.0), @I(@N(CODE), @L(9.5)), @I(@N(R), @L(29.5)), @O(@N(VAL), @R(9.5));
  @C(1616) : @F(TO_REAL), @R(890.0, 130.0, 120.0, 18.0), DINT, @I(@N(IN), @L(9.5)), @O(@N(TO_REAL), @R(9.5));
  @VF(1617) : @E(1), @R(630.0, 150.0, 50.0, 19.0), BOOL;
  @VF(1618) : @E(113), @R(630.0, 130.0, 50.0, 19.0), UDINT;
  @C(1622) : @FB(GUICFG_INT20), @R(690.0, 170.0, 180.0, 38.0), @I(@N(CODE), @L(9.5)), @I(@N(R), @L(29.5)), @O(@N(VAL), @R(9.5));
  @C(1623) : @F(TO_REAL), @R(890.0, 170.0, 120.0, 18.0), DINT, @I(@N(IN), @L(9.5)), @O(@N(TO_REAL), @R(9.5));
  @VF(1624) : @E(1), @R(630.0, 190.0, 50.0, 19.0), BOOL;
  @VF(1625) : @E(114), @R(630.0, 170.0, 50.0, 19.0), UDINT;
  @C(1629) : @FB(GUICFG_INT21), @R(690.0, 210.0, 180.0, 38.0), @I(@N(CODE), @L(9.5)), @I(@N(R), @L(29.5)), @O(@N(VAL), @R(9.5));
  @C(1630) : @F(TO_REAL), @R(890.0, 210.0, 120.0, 18.0), DINT, @I(@N(IN), @L(9.5)), @O(@N(TO_REAL), @R(9.5));
  @VF(1631) : @E(1), @R(630.0, 230.0, 50.0, 19.0), BOOL;
  @VF(1632) : @E(115), @R(630.0, 210.0, 50.0, 19.0), UDINT;
  @VF(1636) : @E(cellTemp_minLim), @R(1020.0, 170.0, 140.0, 19.0);
  @VF(1637) : @E(cellTemp_warningUT), @R(1020.0, 210.0, 220.0, 19.0);
  @VF(1722) : @E(cellTemp_warningOT), @R(1020.0, 130.0, 220.0, 19.0);
  @VF(1723) : @E(cellTemp_maxLim), @R(1020.0, 90.0, 140.0, 19.0);
  @C(1729) : @FB(GUICFG_INT22), @R(690.0, 250.0, 180.0, 38.0), @I(@N(CODE), @L(9.5)), @I(@N(R), @L(29.5)), @O(@N(VAL), @R(9.5));
  @VF(1732) : @E(200), @R(630.0, 250.0, 50.0, 19.0), UDINT;
  @VF(1733) : @E(1), @R(630.0, 270.0, 50.0, 19.0), BOOL;
  @VF(1737) : @E(cellVolt_nominal), @R(1020.0, 250.0, 220.0, 19.0);
  @C(1731) : @F(TO_UINT), @R(890.0, 250.0, 120.0, 18.0), DINT, @I(@N(IN), @L(9.5)), @O(@N(TO_UINT), @R(9.5));
  @C(1739) : @FB(GUICFG_INT23), @R(690.0, 290.0, 180.0, 38.0), @I(@N(CODE), @L(9.5)), @I(@N(R), @L(29.5)), @O(@N(VAL), @R(9.5));
  @C(1745) : @F(TO_UINT), @R(890.0, 290.0, 120.0, 18.0), DINT, @I(@N(IN), @L(9.5)), @O(@N(TO_UINT), @R(9.5));
  @VF(1746) : @E(253), @R(630.0, 290.0, 50.0, 19.0), UDINT;
  @VF(1747) : @E(1), @R(630.0, 310.0, 50.0, 19.0), BOOL;
  @VF(520) : @E(BalanceDiff_Threshold), @R(230.0, 1800.0, 180.0, 19.0);
  @VF(1752) : @E(BalanceDiff_Threshold), @R(1020.0, 290.0, 220.0, 19.0);
  @VF(1757) : @E(1), @R(630.0, 350.0, 50.0, 19.0), BOOL;
  @VF(1758) : @E(120), @R(630.0, 330.0, 50.0, 19.0), UDINT;
  @C(1755) : @FB(GUICFG_REAL1), @R(690.0, 330.0, 180.0, 38.0), @I(@N(CODE), @L(9.5)), @I(@N(R), @L(29.5)), @O(@N(VAL), @R(9.5));
  @VF(1754) : @E(DoD_rate), @R(890.0, 330.0, 120.0, 19.0);
  @C(1799) : @F(TO_UINT), @R(890.0, 370.0, 120.0, 18.0), DINT, @I(@N(IN), @L(9.5)), @O(@N(TO_UINT), @R(9.5));
  @C(1903) : @FB(GUICFG_INT24), @R(690.0, 370.0, 180.0, 38.0), @I(@N(CODE), @L(9.5)), @I(@N(R), @L(29.5)), @O(@N(VAL), @R(9.5));
  @VF(1904) : @E(121), @R(630.0, 370.0, 50.0, 19.0), UDINT;
  @VF(1905) : @E(1), @R(630.0, 390.0, 50.0, 19.0), BOOL;
  @VF(1909) : @E(cyclesPerSOH), @R(1030.0, 370.0, 140.0, 19.0);
  @VF(1911) : @E(cyclesPerSOH), @R(40.0, 1310.0, 140.0, 19.0);
  @VF(1913) : @E(selClock), @R(340.0, 1050.0, 140.0, 19.0);
  @VF(1987) : @E(warningMdlBalT), @R(3200.0, 1940.0, 140.0, 19.0);
  @VF(1988) : @E(faultMdlBalT), @R(3200.0, 1960.0, 140.0, 19.0);
  @VF(2010) : @E(BCU_Fault_Warning), @R(2900.0, 1350.0, 160.0, 19.0);
  @C(2011) : @F(OR), @R(2850.0, 1350.0, 40.0, 98.0), BOOL, @I(@N(IN1), @L(9.5)), @I(@N(IN2), @L(29.5)), @I(@N(IN3), @L(49.5)), @I(@N(IN4), @L(69.5)), @I(@N(IN5), @L(89.5)), @O(@N(OR), @R(9.5));
  @VF(2012) : @E(Fault_Cell_Over_Voltage_Warning), @R(2580.0, 1350.0, 260.0, 19.0);
  @VF(2013) : @E(Fault_Cell_Under_Voltage_Warning), @R(2580.0, 1370.0, 260.0, 19.0);
  @VF(2014) : @E(Fault_Cell_Over_Temp_Warning), @R(2580.0, 1390.0, 260.0, 19.0);
  @VF(2015) : @E(Fault_Cell_Under_Temp_Warning), @R(2580.0, 1410.0, 260.0, 19.0);
  @VF(2016) : @E(warningMdlBalT), @R(2700.0, 1430.0, 140.0, 19.0);
  @C(2030) : @F(OR), @R(2850.0, 1480.0, 40.0, 278.0), BOOL, @I(@N(IN1), @L(9.5)), @I(@N(IN2), @L(29.5)), @I(@N(IN3), @L(49.5)), @I(@N(IN4), @L(69.5)), @I(@N(IN5), @L(89.5)), @I(@N(IN6), @L(109.5)), @I(@N(IN7), @L(129.5)), @I(@N(IN8), @L(149.5)), @I(@N(IN9), @L(169.5)), @I(@N(IN10), @L(189.5)), @I(@N(IN11), @L(209.5)), @I(@N(IN12), @L(229.5)), @I(@N(IN13), @L(249.5)), @I(@N(IN14), @L(269.5)), @O(@N(OR), @R(9.5));
  @VF(2031) : @E(Fault_Cell_Under_Temp_Danger), @R(2620.0, 1500.0, 220.0, 19.0);
  @VF(2032) : @E(Fault_Cell_Over_Temp_Danger), @R(2620.0, 1480.0, 220.0, 19.0);
  @VF(2033) : @E(Fault_Pack_HVIL_1), @R(2620.0, 1540.0, 220.0, 19.0);
  @VF(2034) : @E(Fault_CAN_Communication), @R(2620.0, 1520.0, 220.0, 19.0);
  @VF(2035) : @E(Fault_Pack_BMU), @R(2620.0, 1560.0, 220.0, 19.0);
  @VF(2036) : @E(Fault_Pack_Discharge_Contactor), @R(2620.0, 1580.0, 220.0, 19.0);
  @VF(2039) : @E(OC_fault), @R(2700.0, 1640.0, 140.0, 19.0);
  @VF(2040) : @E(faultMdlBalT), @R(2700.0, 1660.0, 140.0, 19.0);
  @VF(2041) : @E(Fault_Pack_HVIL_2), @R(2640.0, 1680.0, 200.0, 19.0);
  @VF(2024) : @E(BCU_Fault_Danger), @R(2900.0, 1480.0, 150.0, 19.0);
  @VF(2023) : @E(Fault_Pack_Negative_Contactor), @R(2620.0, 1700.0, 220.0, 19.0);
  @VF(2037) : @E(Fault_Cell_Over_Voltage_Danger), @R(2590.0, 1600.0, 250.0, 19.0);
  @VF(2038) : @E(Fault_Cell_Under_Voltage_Danger), @R(2590.0, 1620.0, 250.0, 19.0);
  @VF(2054) : @E(Fault_Pack_Charge_Contactor), @R(2610.0, 1720.0, 230.0, 19.0);
  @C(2056) : @F(OR), @R(2850.0, 1770.0, 40.0, 258.0), BOOL, @I(@N(IN1), @L(9.5)), @I(@N(IN2), @L(29.5)), @I(@N(IN3), @L(49.5)), @I(@N(IN4), @L(69.5)), @I(@N(IN5), @L(89.5)), @I(@N(IN6), @L(109.5)), @I(@N(IN7), @L(129.5)), @I(@N(IN8), @L(149.5)), @I(@N(IN9), @L(169.5)), @I(@N(IN10), @L(189.5)), @I(@N(IN11), @L(209.5)), @I(@N(IN12), @L(229.5)), @I(@N(IN13), @L(249.5)), @O(@N(OR), @R(9.5));
  @VF(2057) : @E(Fault_Cell_Under_Temp_Danger), @R(2610.0, 1790.0, 220.0, 19.0);
  @VF(2058) : @E(Fault_Pack_Discharge_Contactor), @R(2610.0, 1870.0, 220.0, 19.0);
  @VF(2059) : @E(Fault_Cell_Over_Temp_Danger), @R(2610.0, 1770.0, 220.0, 19.0);
  @VF(2060) : @E(Fault_Pack_HVIL_1), @R(2610.0, 1830.0, 220.0, 19.0);
  @VF(2061) : @E(Fault_CAN_Communication), @R(2610.0, 1810.0, 220.0, 19.0);
  @VF(2062) : @E(Fault_Pack_BMU), @R(2610.0, 1850.0, 220.0, 19.0);
  @VF(2063) : @E(UV_fault), @R(2690.0, 1910.0, 140.0, 19.0);
  @VF(2064) : @E(OV_fault), @R(2690.0, 1890.0, 140.0, 19.0);
  @VF(2065) : @E(OC_fault), @R(2690.0, 1930.0, 140.0, 19.0);
  @VF(2066) : @E(faultMdlBalT), @R(2690.0, 1950.0, 140.0, 19.0);
  @VF(2088) : @E(FaultForState), @R(2900.0, 1770.0, 140.0, 19.0);
  @VF(2090) : @E(Fault_Pack_Negative_Contactor), @R(2610.0, 1970.0, 220.0, 19.0);
  @VF(2095) : @E(Fault_Pack_Charge_Contactor), @R(2610.0, 1990.0, 220.0, 19.0);
  @VF(195) : @E(FaultForState), @R(150.0, 2290.0, 150.0, 19.0);
  @VF(65) : @E(maxChargeAmprCfg), @R(500.0, 530.0, 150.0, 19.0);
  @VF(2135) : @E(HVIL2_status), @R(2410.0, 3400.0, 140.0, 19.0);
  @C(2152) : @FB(TOF10), @R(2300.0, 2630.0, 100.0, 38.0), @I(@N(IN), @L(9.5)), @I(@N(PT), @L(29.5)), @O(@N(Q), @R(9.5)), @O(@N(ET), @R(29.5));
  @C(2153) : @FB(Buffer13), @R(2170.0, 2630.0, 100.0, 18.0), @I(@N(I), @L(9.5)), @O(@N(O), @R(9.5));
  @C(2154) : @F(NOT), @R(2080.0, 2630.0, 60.0, 18.0), BOOL, @I(@N(IN), @L(9.5)), @O(@N(NOT), @R(9.5));
  @VF(2155) : @E(Fault_Pack_HVIL_2), @R(2430.0, 2630.0, 220.0, 19.0);
  @VF(2156) : @E(T#3s), @R(2220.0, 2650.0, 50.0, 19.0);
  @VF(2157) : @E(HVIL2_status), @R(1910.0, 2630.0, 140.0, 19.0);
  @VF(1237) : @E(Total_Voltage), @R(1920.0, 1440.0, 200.0, 19.0);
  @VF(71) : @E(bmuCellVolt[4]), @R(1270.0, 1730.0, 140.0, 19.0);
  @VF(685) : @E(bmuCellVolt[5]), @R(1270.0, 1750.0, 140.0, 19.0);
  @VF(2116) : @E(bmuCellVolt[6]), @R(1270.0, 1770.0, 140.0, 19.0);
  @C(2168) : @FB(GUICFG_INT25), @R(690.0, 410.0, 180.0, 38.0), @I(@N(CODE), @L(9.5)), @I(@N(R), @L(29.5)), @O(@N(VAL), @R(9.5));
  @VF(2175) : @E(130), @R(630.0, 410.0, 50.0, 19.0), UDINT;
  @VF(2176) : @E(1), @R(630.0, 430.0, 50.0, 19.0), BOOL;
  @C(2174) : @F(TO_UDINT), @R(890.0, 410.0, 120.0, 18.0), DINT, @I(@N(IN), @L(9.5)), @O(@N(TO_UDINT), @R(9.5));
  @VF(2179) : @E(prechargeInterval), @R(1030.0, 410.0, 140.0, 19.0);
  @C(2201) : @F(TO_UDINT), @R(890.0, 450.0, 120.0, 18.0), DINT, @I(@N(IN), @L(9.5)), @O(@N(TO_UDINT), @R(9.5));
  @C(2202) : @FB(GUICFG_INT26), @R(690.0, 450.0, 180.0, 38.0), @I(@N(CODE), @L(9.5)), @I(@N(R), @L(29.5)), @O(@N(VAL), @R(9.5));
  @VF(2203) : @E(266), @R(630.0, 450.0, 50.0, 19.0), UDINT;
  @VF(2204) : @E(1), @R(630.0, 470.0, 50.0, 19.0), BOOL;
  @VF(2208) : @E(ntcBETA), @R(1030.0, 450.0, 140.0, 19.0);
  @VF(117) : @E(ntcBETA), @R(1100.0, 920.0, 80.0, 19.0);
  @C(265) : @F(TO_REAL), @R(1190.0, 920.0, 120.0, 18.0), UDINT, @I(@N(IN), @L(9.5)), @O(@N(TO_REAL), @R(9.5));
  @C(2214) : @FB(GUICFG_INT27), @R(690.0, 490.0, 180.0, 38.0), @I(@N(CODE), @L(9.5)), @I(@N(R), @L(29.5)), @O(@N(VAL), @R(9.5));
  @VF(2237) : @E(OCfaultAmpr), @R(1030.0, 490.0, 140.0, 19.0);
  @VF(2242) : @E(2004), @R(630.0, 490.0, 50.0, 19.0), UDINT;
  @VF(2243) : @E(1), @R(630.0, 510.0, 50.0, 19.0), BOOL;
  @C(2096) : @F(TO_UINT), @R(890.0, 490.0, 120.0, 18.0), DINT, @I(@N(IN), @L(9.5)), @O(@N(TO_UINT), @R(9.5));
  @VF(953) : @E(OCfaultAmpr), @R(1910.0, 1670.0, 140.0, 19.0);
  @C(2251) : @F(ABS), @R(2070.0, 1610.0, 60.0, 18.0), REAL, @I(@N(IN), @L(9.5)), @O(@N(ABS), @R(9.5));
  @VF(106) : @E(Fault_Pack_CMS), @R(2610.0, 2010.0, 220.0, 19.0);
  @VF(616) : @E(Fault_Pack_CMS), @R(2620.0, 1740.0, 220.0, 19.0);
  @VF(109) : @E(bmuCellVolt[0]), @R(1270.0, 1610.0, 140.0, 19.0);
  @VF(110) : @E(bmuCellVolt[3]), @R(1270.0, 1670.0, 140.0, 19.0);
  @VF(192) : @E(bmuCellVolt[2]), @R(1270.0, 1650.0, 140.0, 19.0);
  @VF(314) : @E(bmuCellVolt[1]), @R(1270.0, 1630.0, 140.0, 19.0);
  @VF(496) : @E(contactFbkDischarge), @R(150.0, 2170.0, 160.0, 19.0);
  @C(753) : @F(LT), @R(4080.0, 640.0, 40.0, 38.0), REAL, @I(@N(IN1), @L(9.5)), @I(@N(IN2), @L(29.5)), @O(@N(LT), @R(9.5));
  @C(755) : @F(GT), @R(4080.0, 690.0, 40.0, 38.0), REAL, @I(@N(IN1), @L(9.5)), @I(@N(IN2), @L(29.5)), @O(@N(GT), @R(9.5));
  @C(854) : @FB(Tbuffer15), @R(4200.0, 640.0, 120.0, 38.0), @I(@N(I), @L(9.5)), @I(@N(D), @L(29.5)), @O(@N(O), @R(9.5));
  @C(858) : @FB(Tbuffer16), @R(4200.0, 690.0, 120.0, 38.0), @I(@N(I), @L(9.5)), @I(@N(D), @L(29.5)), @O(@N(O), @R(9.5));
  @C(878) : @FB(SR5), @R(4410.0, 640.0, 80.0, 38.0), @I(@N(S1), @L(9.5)), @I(@N(R), @L(29.5)), @O(@N(Q1), @R(9.5));
  @VF(940) : @E(-0.2), @R(3950.0, 660.0, 60.0, 19.0), REAL;
  @VF(1001) : @E(0.1), @R(3950.0, 710.0, 60.0, 19.0), REAL;
  @VF(1209) : @E(T#1s), @R(4140.0, 710.0, 40.0, 19.0);
  @VF(1251) : @E(T#1s), @R(4140.0, 660.0, 40.0, 19.0);
  @VF(1253) : @E(batteryInCharge), @R(4510.0, 640.0, 140.0, 19.0);
  @C(2255) : @F(MUX_USINT), @R(3550.0, 30.0, 120.0, 98.0), USINT, @I(@N(K), @L(9.5)), @I(@N(IN0), @L(29.5)), @I(@N(IN1), @L(49.5)), @I(@N(IN2), @L(69.5)), @I(@N(IN3), @L(89.5)), @O(@N(MUX_USINT), @R(9.5));
  @C(2256) : @FB(HVCU_Control_State2), @R(3050.0, 50.0, 460.0, 118.0), @I(@N(CAN_ID), @L(29.5)), @I(@N(CAN_CH), @L(9.5)), @O(@N(Battey_State_BCU_00), @R(9.5)), @O(@N(Battey_State_BCU_01), @R(29.5)), @O(@N(Battey_State_BCU_02), @R(49.5)), @O(@N(Battey_State_BCU_03), @R(69.5)), @O(@N(IMDCtrl_BCU0), @R(89.5)), @O(@N(CAN_Error), @R(109.5));
  @VF(2258) : @E(HVCU_State), @R(3680.0, 30.0, 110.0, 19.0);
  @VF(2262) : @E(CAN_Fault_07), @R(3550.0, 150.0, 120.0, 19.0);
  @VF(2263) : @E(IMDenable), @R(3550.0, 130.0, 120.0, 19.0);
  @VF(2265) : @E(16#18FF01F3), @R(2900.0, 210.0, 110.0, 19.0), UDINT;
  @VF(2266) : @E(16#18FF201E), @R(2900.0, 70.0, 110.0, 19.0), UDINT;
  @VF(2267) : @E(BCU_CAN_CH), @R(2900.0, 50.0, 110.0, 19.0);
  @VF(82) : @E(BatteryCurrent), @R(3870.0, 640.0, 140.0, 19.0);
  @VF(1641) : @E(slaveMode), @R(3980.0, 890.0, 140.0, 19.0);
  @C(1642) : @F(SEL), @R(4160.0, 890.0, 120.0, 58.0), BOOL, @I(@N(G), @L(9.5)), @I(@N(IN0), @L(29.5)), @I(@N(IN1), @L(49.5)), @O(@N(SEL), @R(9.5));
  @VF(1644) : @E(dischargeCMD), @R(3980.0, 930.0, 140.0, 19.0);
  @VF(1645) : @E(dischargeENB), @R(4390.0, 870.0, 140.0, 19.0);
  @C(1648) : @F(SEL), @R(4160.0, 950.0, 120.0, 58.0), BOOL, @I(@N(G), @L(9.5)), @I(@N(IN0), @L(29.5)), @I(@N(IN1), @L(49.5)), @O(@N(SEL), @R(9.5));
  @VF(1649) : @E(chargeENB), @R(4390.0, 930.0, 140.0, 19.0);
  @VF(1651) : @E(chargeCMD), @R(3980.0, 990.0, 140.0, 19.0);
  @VF(2067) : @E(batteryInCharge), @R(3980.0, 970.0, 140.0, 19.0);
  @C(2185) : @F(SEL), @R(3470.0, 790.0, 120.0, 58.0), BOOL, @I(@N(G), @L(9.5)), @I(@N(IN0), @L(29.5)), @I(@N(IN1), @L(49.5)), @O(@N(SEL), @R(9.5));
  @C(659) : @F(SEL), @R(3470.0, 730.0, 120.0, 58.0), BOOL, @I(@N(G), @L(9.5)), @I(@N(IN0), @L(29.5)), @I(@N(IN1), @L(49.5)), @O(@N(SEL), @R(9.5));
  @C(543) : @F(SEL), @R(3470.0, 850.0, 120.0, 58.0), BOOL, @I(@N(G), @L(9.5)), @I(@N(IN0), @L(29.5)), @I(@N(IN1), @L(49.5)), @O(@N(SEL), @R(9.5));
  @VF(1203) : @E(cmdBCU), @R(3020.0, 750.0, 120.0, 19.0);
  @VF(1204) : @E(16#AA), @R(3070.0, 770.0, 70.0, 19.0), USINT;
  @VF(1210) : @E(forceDischarge), @R(3280.0, 770.0, 160.0, 19.0);
  @VF(2190) : @E(contactNegEnable_batt), @R(3230.0, 810.0, 210.0, 19.0);
  @VF(2192) : @E(forceNegative), @R(3280.0, 830.0, 160.0, 19.0);
  @VF(665) : @E(contactEnable), @R(3600.0, 730.0, 130.0, 19.0);
  @VF(2194) : @E(contactNegEnable), @R(3600.0, 790.0, 160.0, 19.0);
  @VF(1876) : @E(forceCharge), @R(3280.0, 890.0, 160.0, 19.0);
  @VF(684) : @E(contactEnableCharge), @R(3600.0, 850.0, 170.0, 19.0);
  @VF(621) : @E(dischargeENB), @R(150.0, 2050.0, 140.0, 19.0);
  @VF(1323) : @E(chargeENB), @R(150.0, 2070.0, 140.0, 19.0);
  @C(1646) : @F(AND), @R(4320.0, 870.0, 40.0, 38.0), BOOL, @I(@N(IN1), @L(9.5)), @I(@N(IN2), @L(29.5)), @O(@N(AND), @R(9.5));
  @C(2630) : @F(AND), @R(4320.0, 930.0, 40.0, 38.0), BOOL, @I(@N(IN1), @L(9.5)), @I(@N(IN2), @L(29.5)), @O(@N(AND), @R(9.5));
  @VF(2633) : @E(currentProtection), @R(3960.0, 870.0, 160.0, 19.0), @ONEG;
  @C(2595) : @F(GE), @R(4070.0, 70.0, 40.0, 38.0), REAL, @I(@N(IN1), @L(9.5)), @I(@N(IN2), @L(29.5)), @O(@N(GE), @R(9.5));
  @C(2605) : @F(LE), @R(4070.0, 110.0, 40.0, 38.0), REAL, @I(@N(IN1), @L(9.5)), @I(@N(IN2), @L(29.5)), @O(@N(LE), @R(9.5));
  @C(1278) : @F(OR), @R(4070.0, 170.0, 40.0, 38.0), BOOL, @I(@N(IN1), @L(9.5)), @I(@N(IN2), @L(29.5)), @O(@N(OR), @R(9.5));
  @C(2609) : @FB(Tbuffer20), @R(4220.0, 110.0, 120.0, 38.0), @I(@N(I), @L(9.5)), @I(@N(D), @L(29.5)), @O(@N(O), @R(9.5));
  @C(2599) : @FB(Tbuffer19), @R(4220.0, 70.0, 120.0, 38.0), @I(@N(I), @L(9.5)), @I(@N(D), @L(29.5)), @O(@N(O), @R(9.5));
  @C(1304) : @F(OR), @R(4480.0, 210.0, 40.0, 38.0), BOOL, @I(@N(IN1), @L(9.5)), @I(@N(IN2), @L(29.5)), @O(@N(OR), @R(9.5));
  @C(1296) : @F(GT), @R(4070.0, 210.0, 40.0, 38.0), REAL, @I(@N(IN1), @L(9.5)), @I(@N(IN2), @L(29.5)), @O(@N(GT), @R(9.5));
  @C(1302) : @FB(TON17), @R(4340.0, 210.0, 100.0, 38.0), @I(@N(IN), @L(9.5)), @I(@N(PT), @L(29.5)), @O(@N(Q), @R(9.5)), @O(@N(ET), @R(29.5));
  @C(1300) : @F(AND), @R(4550.0, 170.0, 40.0, 38.0), BOOL, @I(@N(IN1), @L(9.5)), @I(@N(IN2), @L(29.5)), @O(@N(AND), @R(9.5));
  @C(1287) : @FB(TON2), @R(4340.0, 250.0, 100.0, 38.0), @I(@N(IN), @L(9.5)), @I(@N(PT), @L(29.5)), @O(@N(Q), @R(9.5)), @O(@N(ET), @R(29.5));
  @C(2618) : @F(AND), @R(4560.0, 310.0, 40.0, 38.0), BOOL, @I(@N(IN1), @L(9.5)), @I(@N(IN2), @L(29.5)), @O(@N(AND), @R(9.5));
  @C(1315) : @F(OR), @R(4070.0, 310.0, 40.0, 38.0), BOOL, @I(@N(IN1), @L(9.5)), @I(@N(IN2), @L(29.5)), @O(@N(OR), @R(9.5));
  @C(1282) : @F(OR), @R(4490.0, 350.0, 40.0, 38.0), BOOL, @I(@N(IN1), @L(9.5)), @I(@N(IN2), @L(29.5)), @O(@N(OR), @R(9.5));
  @C(1283) : @F(LT), @R(4070.0, 350.0, 40.0, 38.0), REAL, @I(@N(IN1), @L(9.5)), @I(@N(IN2), @L(29.5)), @O(@N(LT), @R(9.5));
  @C(1284) : @FB(TON19), @R(4350.0, 350.0, 100.0, 38.0), @I(@N(IN), @L(9.5)), @I(@N(PT), @L(29.5)), @O(@N(Q), @R(9.5)), @O(@N(ET), @R(29.5));
  @C(1035) : @FB(TON18), @R(4350.0, 390.0, 100.0, 38.0), @I(@N(IN), @L(9.5)), @I(@N(PT), @L(29.5)), @O(@N(Q), @R(9.5)), @O(@N(ET), @R(29.5));
  @C(2624) : @F(OR), @R(4410.0, 450.0, 40.0, 58.0), BOOL, @I(@N(IN1), @L(9.5)), @I(@N(IN2), @L(29.5)), @I(@N(IN3), @L(49.5)), @O(@N(OR), @R(9.5));
  @VF(2597) : @E(0.5), @R(3970.0, 90.0, 50.0, 19.0), REAL;
  @VF(2594) : @E(BatteryCurrent), @R(3880.0, 70.0, 140.0, 19.0);
  @VF(2607) : @E(-0.5), @R(3970.0, 130.0, 50.0, 19.0), REAL;
  @VF(2610) : @E(T#500ms), @R(4120.0, 130.0, 80.0, 19.0);
  @VF(2601) : @E(T#500ms), @R(4120.0, 90.0, 80.0, 19.0);
  @VF(1277) : @E(UV_danger), @R(3850.0, 170.0, 160.0, 19.0);
  @VF(1279) : @E(dischargeComplete), @R(3850.0, 190.0, 160.0, 19.0);
  @VF(1295) : @E(BatteryCurrent), @R(3850.0, 210.0, 160.0, 19.0);
  @VF(1298) : @E(5), @R(3960.0, 230.0, 50.0, 19.0), REAL;
  @VF(1303) : @E(T#3s), @R(4250.0, 230.0, 80.0, 19.0);
  @VF(1293) : @E(BatteryDischarging), @R(3850.0, 250.0, 160.0, 19.0);
  @VF(1289) : @E(T#120s), @R(4250.0, 270.0, 80.0, 19.0);
  @VF(2613) : @E(BatteryCharging), @R(4380.0, 110.0, 160.0, 19.0);
  @VF(2603) : @E(BatteryDischarging), @R(4380.0, 70.0, 160.0, 19.0);
  @VF(1329) : @E(OV_danger), @R(3850.0, 310.0, 170.0, 19.0);
  @VF(1336) : @E(BCU_Charge_Complete), @R(3850.0, 330.0, 170.0, 19.0);
  @VF(1292) : @E(dischargeOff), @R(4610.0, 170.0, 150.0, 19.0);
  @VF(1314) : @E(chargeOff), @R(4620.0, 310.0, 150.0, 19.0);
  @VF(1311) : @E(BatteryCurrent), @R(3850.0, 350.0, 160.0, 19.0);
  @VF(1306) : @E(-5), @R(3960.0, 370.0, 50.0, 19.0), REAL;
  @VF(1286) : @E(T#3s), @R(4250.0, 370.0, 90.0, 19.0);
  @VF(1308) : @E(BatteryCharging), @R(3850.0, 390.0, 160.0, 19.0);
  @VF(1285) : @E(T#120s), @R(4250.0, 410.0, 90.0, 19.0);
  @VF(2622) : @E(chargeOff), @R(4220.0, 450.0, 140.0, 19.0);
  @VF(2627) : @E(currentProtection), @R(4470.0, 450.0, 160.0, 19.0);
  @VF(2623) : @E(dischargeOff), @R(4220.0, 470.0, 140.0, 19.0);
  @VF(1656) : @E(batteryInCharge), @R(3980.0, 910.0, 140.0, 19.0), @ONEG;
  @VF(2636) : @E(chargeProtect), @R(4620.0, 290.0, 150.0, 19.0);
  @VF(2638) : @E(dischargeProtect), @R(4610.0, 150.0, 150.0, 19.0);
  @CF(2640) : @R(4390.0, 950.0, 170.0, 59.0), @T("State selection for master(ESS)$Nand slave mode");
  @C(70) : @FB(essState11), @R(350.0, 2050.0, 400.0, 258.0), @I(@N(discharge), @L(9.5)), @I(@N(charge), @L(29.5)), @I(@N(shutdown), @L(49.5)), @I(@N(prechargeOk), @L(89.5)), @I(@N(contactFbk), @L(109.5)), @I(@N(contactFbkNeg), @L(129.5)), @I(@N(dischargeProtect), @L(169.5)), @I(@N(chargeProtect), @L(189.5)), @I(@N(shutdownComplete), @L(229.5)), @I(@N(fault), @L(249.5)), @O(@N(STATE), @R(9.5)), @O(@N(prechargeOn), @R(49.5)), @O(@N(contact), @R(69.5)), @O(@N(contactNeg), @R(89.5));
  @VF(564) : @E(chargeProtect), @R(150.0, 2230.0, 160.0, 19.0);
  @VF(617) : @E(dischargeProtect), @R(150.0, 2210.0, 160.0, 19.0);
  @VF(360) : @E(shutdownEnb), @R(150.0, 2090.0, 140.0, 19.0);
  @CF(2646) : @R(4460.0, 680.0, 170.0, 39.0), @T("ESS charge discharge decision");
  @VF(820) : @E(1), @R(2340.0, 3400.0, 60.0, 19.0), BOOL;
  @VF(2130) : @E(sim100NotFound), @R(1270.0, 1790.0, 140.0, 19.0);
  @CF(1802) : @R(3800.0, 0.0, 200.0, 49.0), @T("charge/discharge transition$Nprotection$N");
  @CF(1863) : @R(1900.0, 0.0, 170.0, 39.0), @T("CAN communication");
  @CF(2086) : @R(1900.0, 1340.0, 160.0, 29.0), @T("Fault generation");
  @CF(2732) : @R(1900.0, 2680.0, 120.0, 29.0), @T("IO");
  @VF(535) : @E(10), @R(330.0, 1970.0, 80.0, 19.0), UDINT;
  @VF(2310) : @E(slaveMode), @R(2110.0, 2530.0, 140.0, 19.0);
  @C(132) : @F(AND), @R(2330.0, 2530.0, 40.0, 38.0), BOOL, @I(@N(IN1), @L(9.5)), @I(@N(IN2), @L(29.5)), @O(@N(AND), @R(9.5));
  @C(42) : @FB(F_TRIG3), @R(250.0, 3850.0, 140.0, 18.0), @I(@N(CLK), @L(9.5)), @O(@N(Q), @R(9.5));
  @C(1887) : @F(OR), @R(400.0, 3830.0, 40.0, 38.0), BOOL, @I(@N(IN1), @L(9.5)), @I(@N(IN2), @L(29.5)), @O(@N(OR), @R(9.5));
  @C(2320) : @FB(F_TRIG4), @R(240.0, 3620.0, 140.0, 18.0), @I(@N(CLK), @L(9.5)), @O(@N(Q), @R(9.5));
  @C(2321) : @FB(R_TRIG9), @R(240.0, 3600.0, 140.0, 18.0), @I(@N(CLK), @L(9.5)), @O(@N(Q), @R(9.5));
  @C(2322) : @F(OR), @R(390.0, 3600.0, 40.0, 38.0), BOOL, @I(@N(IN1), @L(9.5)), @I(@N(IN2), @L(29.5)), @O(@N(OR), @R(9.5));
  @VF(2236) : @E(emergencyBtn), @R(4220.0, 490.0, 140.0, 19.0);
  @VF(427) : @E(whInstant), @R(460.0, 2940.0, 140.0, 19.0);
  @C(1291) : @F(AND), @R(4190.0, 210.0, 40.0, 38.0), BOOL, @I(@N(IN1), @L(9.5)), @I(@N(IN2), @L(29.5)), @O(@N(AND), @R(9.5));
  @C(2358) : @F(AND), @R(4190.0, 250.0, 40.0, 38.0), BOOL, @I(@N(IN1), @L(9.5)), @I(@N(IN2), @L(29.5)), @O(@N(AND), @R(9.5));
  @C(1313) : @F(AND), @R(4190.0, 390.0, 40.0, 38.0), BOOL, @I(@N(IN1), @L(9.5)), @I(@N(IN2), @L(29.5)), @O(@N(AND), @R(9.5));
  @C(1375) : @F(AND), @R(4190.0, 350.0, 40.0, 38.0), BOOL, @I(@N(IN1), @L(9.5)), @I(@N(IN2), @L(29.5)), @O(@N(AND), @R(9.5));
  @VF(1003) : @E(prechargeComplete), @R(720.0, 2420.0, 160.0, 19.0);
  @VF(1963) : @E(prechargeEnable), @R(430.0, 2420.0, 190.0, 19.0);
  @VF(178) : @E(dischargeProtect), @R(2040.0, 270.0, 140.0, 19.0);
  @VF(238) : @E(chargeProtect), @R(2040.0, 250.0, 140.0, 19.0);
  @VF(69) : @E(10), @R(1140.0, 1460.0, 40.0, 19.0), REAL;
  @C(435) : @F(SEL), @R(670.0, 1470.0, 120.0, 58.0), REAL, @I(@N(G), @L(9.5)), @I(@N(IN0), @L(29.5)), @I(@N(IN1), @L(49.5)), @O(@N(SEL), @R(9.5));
  @VF(437) : @E(socChComp), @R(810.0, 1470.0, 100.0, 19.0);
  @VF(560) : @E(SoCreal), @R(570.0, 1510.0, 80.0, 19.0);
  @VF(562) : @E(socChComp), @R(550.0, 1490.0, 100.0, 19.0);
  @C(565) : @FB(R_TRIG2), @R(510.0, 1470.0, 140.0, 18.0), @I(@N(CLK), @L(9.5)), @O(@N(Q), @R(9.5));
  @VF(567) : @E(mainChargeComplete), @R(320.0, 1470.0, 170.0, 19.0);
  @VF(569) : @E(socChComp), @R(380.0, 1410.0, 100.0, 19.0);
  @C(582) : @F(SUB), @R(490.0, 1410.0, 40.0, 38.0), REAL, @I(@N(IN1), @L(9.5)), @I(@N(IN2), @L(29.5)), @O(@N(SUB), @R(9.5));
  @VF(739) : @E(SoCreal), @R(400.0, 1430.0, 80.0, 19.0);
  @C(742) : @F(GT), @R(600.0, 1410.0, 40.0, 38.0), REAL, @I(@N(IN1), @L(9.5)), @I(@N(IN2), @L(29.5)), @O(@N(GT), @R(9.5));
  @VF(750) : @E(2), @R(540.0, 1430.0, 50.0, 19.0), REAL;
  @C(757) : @F(GE), @R(240.0, 1440.0, 40.0, 38.0), REAL, @I(@N(IN1), @L(9.5)), @I(@N(IN2), @L(29.5)), @O(@N(GE), @R(9.5));
  @C(861) : @F(SEL), @R(1620.0, 1470.0, 120.0, 58.0), REAL, @I(@N(G), @L(9.5)), @I(@N(IN0), @L(29.5)), @I(@N(IN1), @L(49.5)), @O(@N(SEL), @R(9.5));
  @C(866) : @FB(R_TRIG3), @R(1460.0, 1470.0, 140.0, 18.0), @I(@N(CLK), @L(9.5)), @O(@N(Q), @R(9.5));
  @VF(886) : @E(SoCreal), @R(1520.0, 1510.0, 80.0, 19.0);
  @VF(889) : @E(socDchComp), @R(1480.0, 1490.0, 120.0, 19.0);
  @VF(890) : @E(dischargeComplete), @R(1270.0, 1470.0, 160.0, 19.0);
  @VF(867) : @E(socDchComp), @R(1750.0, 1470.0, 120.0, 19.0);
  @C(926) : @F(GT), @R(1580.0, 1420.0, 40.0, 38.0), REAL, @I(@N(IN1), @L(9.5)), @I(@N(IN2), @L(29.5)), @O(@N(GT), @R(9.5));
  @C(944) : @F(SUB), @R(1480.0, 1420.0, 40.0, 38.0), REAL, @I(@N(IN1), @L(9.5)), @I(@N(IN2), @L(29.5)), @O(@N(SUB), @R(9.5));
  @VF(952) : @E(4), @R(1530.0, 1440.0, 40.0, 19.0), REAL;
  @VF(987) : @E(SoCreal), @R(1350.0, 1420.0, 110.0, 19.0);
  @VF(1020) : @E(socDchComp), @R(1350.0, 1440.0, 110.0, 19.0);
  @C(90) : @FB(HVCU_Config1), @R(3050.0, 190.0, 460.0, 98.0), @I(@N(CAN_CH), @L(9.5)), @I(@N(CAN_ID), @L(29.5)), @O(@N(cmd0), @R(9.5)), @O(@N(CAN_Error), @R(89.5)), @O(@N(cmd1), @R(29.5)), @O(@N(cmd2), @R(49.5)), @O(@N(cmd3), @R(69.5));
  @C(91) : @F(MUX_USINT), @R(3550.0, 170.0, 120.0, 98.0), USINT, @I(@N(K), @L(9.5)), @I(@N(IN0), @L(29.5)), @I(@N(IN1), @L(49.5)), @I(@N(IN2), @L(69.5)), @I(@N(IN3), @L(89.5)), @O(@N(MUX_USINT), @R(9.5));
  @VF(355) : @E(cmdBCU), @R(3680.0, 170.0, 110.0, 19.0);
  @VF(380) : @E(Selected_Pack_Number), @R(3330.0, 30.0, 180.0, 19.0);
  @VF(383) : @E(cmdBCU), @R(3120.0, 570.0, 90.0, 19.0);
  @C(384) : @F(EQ), @R(3230.0, 570.0, 40.0, 38.0), USINT, @I(@N(IN1), @L(9.5)), @I(@N(IN2), @L(29.5)), @O(@N(EQ), @R(9.5));
  @VF(386) : @E(16#AB), @R(3120.0, 590.0, 90.0, 19.0), USINT;
  @VF(619) : @E(forceDischarge), @R(3290.0, 570.0, 140.0, 19.0);
  @C(859) : @F(EQ), @R(3230.0, 610.0, 40.0, 38.0), USINT, @I(@N(IN1), @L(9.5)), @I(@N(IN2), @L(29.5)), @O(@N(EQ), @R(9.5));
  @VF(864) : @E(16#AC), @R(3120.0, 630.0, 90.0, 19.0), USINT;
  @VF(1091) : @E(cmdBCU), @R(3120.0, 610.0, 90.0, 19.0);
  @VF(1115) : @E(forceCharge), @R(3290.0, 610.0, 140.0, 19.0);
  @C(1139) : @F(EQ), @R(3230.0, 650.0, 40.0, 38.0), USINT, @I(@N(IN1), @L(9.5)), @I(@N(IN2), @L(29.5)), @O(@N(EQ), @R(9.5));
  @VF(1140) : @E(16#AD), @R(3120.0, 670.0, 90.0, 19.0), USINT;
  @VF(1142) : @E(cmdBCU), @R(3120.0, 650.0, 90.0, 19.0);
  @VF(1143) : @E(forceNegative), @R(3290.0, 650.0, 140.0, 19.0);
  @C(657) : @F(GT), @R(3160.0, 750.0, 40.0, 38.0), USINT, @I(@N(IN1), @L(9.5)), @I(@N(IN2), @L(29.5)), @O(@N(GT), @R(9.5));
  @C(672) : @F(AND), @R(3230.0, 730.0, 40.0, 38.0), BOOL, @I(@N(IN1), @L(9.5)), @I(@N(IN2), @L(29.5)), @O(@N(AND), @R(9.5));
  @VF(1148) : @E(cmdTmt), @R(3550.0, 270.0, 120.0, 19.0);
  @VF(1150) : @E(cmdTmt), @R(3020.0, 730.0, 120.0, 19.0), @ONEG;
  @VF(690) : @E(multAmpChar), @R(1710.0, 2720.0, 120.0, 19.0);
  @VF(812) : @E(Cell_Temp_Max), @R(1130.0, 2720.0, 160.0, 19.0);
  @VF(819) : @E(Cell_Temp_Min), @R(1130.0, 2740.0, 160.0, 19.0);
  @C(838) : @F(MIN), @R(1540.0, 2720.0, 80.0, 38.0), REAL, @I(@N(IN1), @L(9.5)), @I(@N(IN2), @L(29.5)), @O(@N(MIN), @R(9.5));
  @VF(1077) : @E(Cell_Temp_Max), @R(1130.0, 2810.0, 160.0, 19.0);
  @VF(1191) : @E(Cell_Temp_Min), @R(1130.0, 2830.0, 160.0, 19.0);
  @C(1195) : @F(MIN), @R(1540.0, 2810.0, 80.0, 38.0), REAL, @I(@N(IN1), @L(9.5)), @I(@N(IN2), @L(29.5)), @O(@N(MIN), @R(9.5));
  @VF(1200) : @E(multAmpDisch), @R(1710.0, 2810.0, 120.0, 19.0);
  @C(699) : @FB(ampMultTemp1), @R(1320.0, 2720.0, 200.0, 18.0), @I(@N(temp), @L(9.5)), @O(@N(mult), @R(9.5));
  @C(817) : @FB(ampMultTemp2), @R(1320.0, 2740.0, 200.0, 18.0), @I(@N(temp), @L(9.5)), @O(@N(mult), @R(9.5));
  @C(1014) : @FB(ampMultTempDis1), @R(1320.0, 2810.0, 200.0, 18.0), @I(@N(temp), @L(9.5)), @O(@N(mult), @R(9.5));
  @C(1192) : @FB(ampMultTempDis2), @R(1320.0, 2830.0, 200.0, 18.0), @I(@N(temp), @L(9.5)), @O(@N(mult), @R(9.5));
  @C(1201) : @F(MUL), @R(1650.0, 2810.0, 40.0, 38.0), REAL, @I(@N(IN1), @L(9.5)), @I(@N(IN2), @L(29.5)), @O(@N(MUL), @R(9.5));
  @C(1207) : @FB(ampMultVoltChar1), @R(1320.0, 2760.0, 200.0, 38.0), @I(@N(chargeOn), @L(9.5)), @I(@N(maxCell), @L(29.5)), @O(@N(mult), @R(9.5));
  @C(1016) : @F(MUL), @R(1650.0, 2720.0, 40.0, 38.0), REAL, @I(@N(IN1), @L(9.5)), @I(@N(IN2), @L(29.5)), @O(@N(MUL), @R(9.5));
  @VF(1231) : @E(Cell_Voltage_Max), @R(1130.0, 2780.0, 160.0, 19.0);
  @C(1198) : @FB(ampMultVoltDisc1), @R(1320.0, 2850.0, 200.0, 38.0), @I(@N(discOn), @L(9.5)), @I(@N(minCell), @L(29.5)), @O(@N(mult), @R(9.5));
  @VF(1235) : @E(Cell_Voltage_Min), @R(1130.0, 2870.0, 160.0, 19.0);
  @VF(1240) : @E(BatteryCharging), @R(1130.0, 2760.0, 160.0, 19.0);
  @VF(1247) : @E(BatteryDischarging), @R(1130.0, 2850.0, 160.0, 19.0);
  @VF(198) : @E(increaseDischargeAmp), @R(660.0, 3180.0, 180.0, 19.0);
  @C(302) : @FB(TON21), @R(460.0, 3130.0, 100.0, 38.0), @I(@N(IN), @L(9.5)), @I(@N(PT), @L(29.5)), @O(@N(Q), @R(9.5)), @O(@N(ET), @R(29.5));
  @C(303) : @F(EQ), @R(330.0, 3130.0, 40.0, 38.0), USINT, @I(@N(IN1), @L(9.5)), @I(@N(IN2), @L(29.5)), @O(@N(EQ), @R(9.5));
  @VF(357) : @E(BMS_State), @R(130.0, 3130.0, 180.0, 19.0);
  @VF(379) : @E(BATTSTATE#DISCHARGE), @R(130.0, 3150.0, 180.0, 19.0), USINT;
  @VF(555) : @E(T#5s), @R(400.0, 3150.0, 40.0, 19.0);
  @VF(831) : @E(dischargeAmpEnb), @R(660.0, 3130.0, 180.0, 19.0);
  @C(874) : @F(GE), @R(330.0, 3180.0, 40.0, 38.0), UDINT, @I(@N(IN1), @L(9.5)), @I(@N(IN2), @L(29.5)), @O(@N(GE), @R(9.5));
  @C(904) : @F(AND), @R(540.0, 3180.0, 40.0, 38.0), BOOL, @I(@N(IN1), @L(9.5)), @I(@N(IN2), @L(29.5)), @O(@N(AND), @R(9.5));
  @VF(905) : @E(Cell_Voltage_Min), @R(130.0, 3180.0, 180.0, 19.0);
  @VF(909) : @E(cellVolt_dischargeOK), @R(130.0, 3200.0, 180.0, 19.0);
  @VF(923) : @E(dischargeAmpEnb), @R(380.0, 3200.0, 140.0, 19.0);
  @VF(1252) : @E(decreaseDischargeAmp), @R(660.0, 3250.0, 180.0, 19.0);
  @VF(1267) : @E(Cell_Voltage_Min), @R(130.0, 3310.0, 180.0, 19.0);
  @C(1274) : @F(LT), @R(330.0, 3230.0, 40.0, 38.0), REAL, @I(@N(IN1), @L(9.5)), @I(@N(IN2), @L(29.5)), @O(@N(LT), @R(9.5));
  @VF(1280) : @E(Pack_Discharge_Voltage), @R(120.0, 3250.0, 190.0, 19.0);
  @VF(1294) : @E(BatteryVoltage), @R(120.0, 3230.0, 190.0, 19.0);
  @VF(1318) : @E(cellVolt_minDischarge), @R(130.0, 3330.0, 180.0, 19.0);
  @C(1319) : @F(LE), @R(330.0, 3310.0, 40.0, 38.0), UDINT, @I(@N(IN1), @L(9.5)), @I(@N(IN2), @L(29.5)), @O(@N(LE), @R(9.5));
  @C(1450) : @F(OR), @R(330.0, 3270.0, 40.0, 38.0), BOOL, @I(@N(IN1), @L(9.5)), @I(@N(IN2), @L(29.5)), @O(@N(OR), @R(9.5));
  @VF(1453) : @E(OT_danger_risk), @R(170.0, 3270.0, 140.0, 19.0);
  @VF(1461) : @E(UT_danger_risk), @R(170.0, 3290.0, 140.0, 19.0);
  @C(1640) : @F(AND), @R(540.0, 3310.0, 40.0, 38.0), BOOL, @I(@N(IN1), @L(9.5)), @I(@N(IN2), @L(29.5)), @O(@N(AND), @R(9.5));
  @VF(1653) : @E(dischargeAmpEnb), @R(380.0, 3330.0, 140.0, 19.0);
  @C(1709) : @F(OR), @R(600.0, 3250.0, 40.0, 58.0), BOOL, @I(@N(IN1), @L(9.5)), @I(@N(IN2), @L(29.5)), @I(@N(IN3), @L(49.5)), @O(@N(OR), @R(9.5));
  @VF(625) : @E(dischargeAmpEnb), @R(60.0, 3600.0, 140.0, 19.0);
  @VF(873) : @E(increaseDischargeAmp), @R(240.0, 3470.0, 180.0, 19.0);
  @VF(1761) : @E(decreaseDischargeAmp), @R(240.0, 3490.0, 180.0, 19.0);
  @VF(1765) : @E(dischargeUnitAmp), @R(680.0, 3560.0, 150.0, 19.0);
  @VF(1767) : @E(dischargeUnitAmp), @R(60.0, 3570.0, 150.0, 19.0);
  @VF(1769) : @E(dischargeAmpEnb), @R(820.0, 3480.0, 140.0, 19.0);
  @VF(1794) : @E(chargeAmpEnb), @R(1590.0, 3130.0, 160.0, 19.0);
  @C(1795) : @F(EQ), @R(1220.0, 3130.0, 40.0, 38.0), USINT, @I(@N(IN1), @L(9.5)), @I(@N(IN2), @L(29.5)), @O(@N(EQ), @R(9.5));
  @C(1796) : @FB(TON22), @R(1330.0, 3130.0, 100.0, 38.0), @I(@N(IN), @L(9.5)), @I(@N(PT), @L(29.5)), @O(@N(Q), @R(9.5)), @O(@N(ET), @R(29.5));
  @VF(1797) : @E(BATTSTATE#CHARGE), @R(1030.0, 3150.0, 170.0, 19.0), USINT;
  @VF(1798) : @E(BMS_State), @R(1030.0, 3130.0, 170.0, 19.0);
  @VF(1800) : @E(T#5s), @R(1280.0, 3150.0, 40.0, 19.0);
  @C(1847) : @F(LE), @R(1220.0, 3180.0, 40.0, 38.0), UDINT, @I(@N(IN1), @L(9.5)), @I(@N(IN2), @L(29.5)), @O(@N(LE), @R(9.5));
  @VF(1853) : @E(cellVolt_chargeOK), @R(1030.0, 3200.0, 170.0, 19.0);
  @VF(1854) : @E(Cell_Voltage_Max), @R(1030.0, 3180.0, 170.0, 19.0);
  @C(1864) : @F(AND), @R(1460.0, 3180.0, 40.0, 58.0), BOOL, @I(@N(IN1), @L(9.5)), @I(@N(IN2), @L(29.5)), @I(@N(IN3), @L(49.5)), @O(@N(AND), @R(9.5));
  @VF(1867) : @E(chargeAmpEnb), @R(1270.0, 3200.0, 160.0, 19.0);
  @VF(1891) : @E(Balance_Enable_Rq), @R(1270.0, 3220.0, 160.0, 19.0), @ONEG;
  @VF(1855) : @E(increaseChargeAmp), @R(1590.0, 3180.0, 160.0, 19.0);
  @VF(2026) : @E(cellVolt_maxCharge), @R(1030.0, 3310.0, 170.0, 19.0);
  @VF(2027) : @E(Cell_Voltage_Max), @R(1030.0, 3290.0, 170.0, 19.0);
  @C(2028) : @F(GE), @R(1220.0, 3290.0, 40.0, 38.0), UDINT, @I(@N(IN1), @L(9.5)), @I(@N(IN2), @L(29.5)), @O(@N(GE), @R(9.5));
  @C(2092) : @F(GT), @R(1220.0, 3250.0, 40.0, 38.0), REAL, @I(@N(IN1), @L(9.5)), @I(@N(IN2), @L(29.5)), @O(@N(GT), @R(9.5));
  @VF(2097) : @E(BatteryVoltage), @R(1030.0, 3250.0, 170.0, 19.0);
  @VF(2098) : @E(Pack_Charge_Voltage), @R(1030.0, 3270.0, 170.0, 19.0);
  @C(2101) : @F(OR), @R(1530.0, 3270.0, 40.0, 58.0), BOOL, @I(@N(IN1), @L(9.5)), @I(@N(IN2), @L(29.5)), @I(@N(IN3), @L(49.5)), @O(@N(OR), @R(9.5));
  @C(2103) : @F(AND), @R(1460.0, 3290.0, 40.0, 58.0), BOOL, @I(@N(IN1), @L(9.5)), @I(@N(IN2), @L(29.5)), @I(@N(IN3), @L(49.5)), @O(@N(AND), @R(9.5));
  @VF(2105) : @E(chargeAmpEnb), @R(1280.0, 3310.0, 160.0, 19.0);
  @VF(2107) : @E(Balance_Enable_Rq), @R(1280.0, 3330.0, 160.0, 19.0), @ONEG;
  @C(2110) : @F(OR), @R(1460.0, 3350.0, 40.0, 38.0), BOOL, @I(@N(IN1), @L(9.5)), @I(@N(IN2), @L(29.5)), @O(@N(OR), @R(9.5));
  @VF(2111) : @E(UT_danger_risk), @R(1280.0, 3370.0, 140.0, 19.0);
  @VF(2112) : @E(OT_danger_risk), @R(1280.0, 3350.0, 140.0, 19.0);
  @VF(2117) : @E(decreaseChargeAmp), @R(1590.0, 3270.0, 160.0, 19.0);
  @VF(356) : @E(chargeUnitAmp), @R(90.0, 3800.0, 140.0, 19.0);
  @VF(1775) : @E(decreaseChargeAmp), @R(270.0, 3720.0, 160.0, 19.0);
  @VF(1778) : @E(increaseChargeAmp), @R(270.0, 3700.0, 160.0, 19.0);
  @VF(1803) : @E(chargeUnitAmp), @R(690.0, 3790.0, 140.0, 19.0);
  @VF(1807) : @E(chargeAmpEnb), @R(90.0, 3830.0, 120.0, 19.0);
  @VF(1812) : @E(chargeAmpEnb), @R(830.0, 3710.0, 140.0, 19.0);
  @C(64) : @F(MAX), @R(910.0, 3520.0, 80.0, 38.0), REAL, @I(@N(IN1), @L(9.5)), @I(@N(IN2), @L(29.5)), @O(@N(MAX), @R(9.5));
  @C(1848) : @F(MAX), @R(920.0, 3750.0, 80.0, 38.0), REAL, @I(@N(IN1), @L(9.5)), @I(@N(IN2), @L(29.5)), @O(@N(MAX), @R(9.5));
  @CF(1851) : @R(750.0, 3730.0, 90.0, 19.0), @T("testAmper");
  @VF(1841) : @E(maxChargeAmp), @R(1380.0, 2900.0, 140.0, 19.0);
  @VF(1869) : @E(maxChargeAmprCfg), @R(1130.0, 2920.0, 170.0, 19.0);
  @C(1872) : @F(MUL), @R(1320.0, 2900.0, 40.0, 38.0), REAL, @I(@N(IN1), @L(9.5)), @I(@N(IN2), @L(29.5)), @O(@N(MUL), @R(9.5));
  @VF(1874) : @E(multAmpChar), @R(1130.0, 2900.0, 170.0, 19.0);
  @VF(1888) : @E(multAmpDisch), @R(1130.0, 2940.0, 170.0, 19.0);
  @C(1889) : @F(MUL), @R(1320.0, 2940.0, 40.0, 38.0), REAL, @I(@N(IN1), @L(9.5)), @I(@N(IN2), @L(29.5)), @O(@N(MUL), @R(9.5));
  @VF(1892) : @E(maxDischargeAmprCfg), @R(1130.0, 2960.0, 170.0, 19.0);
  @VF(1894) : @E(maxDischargeAmp), @R(1380.0, 2940.0, 140.0, 19.0);
  @VF(63) : @E(maxChargeAmp), @R(90.0, 3780.0, 140.0, 19.0);
  @VF(1760) : @E(maxDischargeAmp), @R(60.0, 3550.0, 150.0, 19.0);
  @C(1759) : @FB(UpDownCntTim1), @R(450.0, 3470.0, 210.0, 118.0), @I(@N(CU), @L(9.5)), @I(@N(CD), @L(29.5)), @I(@N(uPer), @L(49.5)), @I(@N(dPer), @L(69.5)), @I(@N(PV), @L(89.5)), @I(@N(RST), @L(109.5)), @O(@N(CV), @R(9.5)), @O(@N(QD), @R(29.5)), @O(@N(QU), @R(49.5));
  @C(1776) : @FB(UpDownCntTim2), @R(460.0, 3700.0, 210.0, 118.0), @I(@N(CU), @L(9.5)), @I(@N(CD), @L(29.5)), @I(@N(uPer), @L(49.5)), @I(@N(dPer), @L(69.5)), @I(@N(PV), @L(89.5)), @I(@N(RST), @L(109.5)), @O(@N(CV), @R(9.5)), @O(@N(QD), @R(29.5)), @O(@N(QU), @R(49.5));
  @C(83) : @FB(BCU_status21), @R(2220.0, 690.0, 500.0, 178.0), @I(@N(Max_Temp_BMU_Loc), @L(69.5)), @I(@N(Max_Temp_Cell_Loc), @L(49.5)), @I(@N(Min_Temp_BMU_Loc), @L(109.5)), @I(@N(Min_Temp_Cell_Loc), @L(89.5)), @I(@N(Max_Cell_Temp), @L(129.5)), @I(@N(Min_Cell_Temp), @L(149.5)), @I(@N(CAN_ID), @L(29.5)), @I(@N(CAN_CH), @L(9.5)), @I(@N(outVolt), @L(169.5)), @O(@N(CAN_Error), @R(149.5));
  @C(136) : @FB(BCU_State_Message1), @R(2220.0, 50.0, 500.0, 298.0), @I(@N(CAN_ID), @L(29.5)), @I(@N(State), @L(49.5)), @I(@N(Contactor_Status), @L(69.5)), @I(@N(ChargeContact), @L(89.5)), @I(@N(Ambient_Temp), @L(109.5)), @I(@N(DMDC), @L(129.5)), @I(@N(DMCC), @L(149.5)), @I(@N(CAN_CH), @L(9.5)), @I(@N(NegContact), @L(169.5)), @I(@N(isolationStatus), @L(189.5)), @I(@N(chargeComplete), @L(209.5)), @I(@N(dischargeComplete), @L(229.5)), @I(@N(emergencyButton), @L(249.5)), @I(@N(in1Status), @L(269.5)), @I(@N(in2Status), @L(289.5)), @O(@N(CAN_Error), @R(149.5));
  @VF(518) : @E(OutputVoltage), @R(2040.0, 850.0, 140.0, 19.0);
  @C(84) : @FB(BCU_Battery_Status1), @R(2220.0, 870.0, 500.0, 138.0), @I(@N(SoC), @L(49.5)), @I(@N(SoH), @L(69.5)), @I(@N(Duty_Cycle), @L(89.5)), @I(@N(Remain_Energy), @L(129.5)), @I(@N(CAN_ID), @L(29.5)), @I(@N(CAN_CH), @L(9.5)), @I(@N(Available_Energy), @L(109.5)), @O(@N(CAN_Error), @R(129.5));
  @C(700) : @FB(GUICFG_INT28), @R(760.0, 540.0, 180.0, 38.0), @I(@N(CODE), @L(9.5)), @I(@N(R), @L(29.5)), @O(@N(VAL), @R(9.5));
  @VF(983) : @E(1), @R(700.0, 560.0, 50.0, 19.0), BOOL;
  @VF(1166) : @E(testValue0), @R(1310.0, 540.0, 140.0, 19.0);
  @VF(1167) : @E(400), @R(700.0, 540.0, 50.0, 19.0), UDINT;
  @C(1172) : @F(TO_TIME), @R(1090.0, 540.0, 120.0, 18.0), UDINT, @I(@N(IN), @L(9.5)), @O(@N(TO_TIME), @R(9.5));
  @C(733) : @F(TO_UDINT), @R(950.0, 540.0, 120.0, 18.0), DINT, @I(@N(IN), @L(9.5)), @O(@N(TO_UDINT), @R(9.5));
  @C(1176) : @F(DIV_TIME), @R(1240.0, 540.0, 40.0, 38.0), UINT, @I(@N(IN1), @L(9.5)), @I(@N(IN2), @L(29.5)), @O(@N(DIV_TIME), @R(9.5));
  @VF(1366) : @E(1000), @R(1080.0, 560.0, 140.0, 19.0), UINT;
  @C(1371) : @FB(TON4), @R(1490.0, -120.0, 100.0, 38.0), @I(@N(IN), @L(9.5)), @I(@N(PT), @L(29.5)), @O(@N(Q), @R(9.5)), @O(@N(ET), @R(29.5));
  @C(1372) : @FB(TON5), @R(1220.0, -120.0, 100.0, 38.0), @I(@N(IN), @L(9.5)), @I(@N(PT), @L(29.5)), @O(@N(Q), @R(9.5)), @O(@N(ET), @R(29.5));
  @C(1373) : @FB(IOWR4), @R(480.0, -110.0, 120.0, 58.0), @I(@N(PORT), @L(9.5)), @I(@N(PIN), @L(29.5)), @I(@N(VAL), @L(49.5));
  @C(1374) : @FB(FLASH3), @R(330.0, -70.0, 120.0, 38.0), @I(@N(IN), @L(9.5)), @I(@N(PER), @L(29.5)), @O(@N(OUT), @R(9.5));
  @C(1376) : @FB(SAFETY_POWER1), @R(300.0, -210.0, 300.0, 78.0), @I(@N(EN_VSOUT1), @L(9.5)), @I(@N(ENDRV), @L(29.5)), @I(@N(WD_PER), @L(49.5)), @I(@N(SLEEP_RDY), @L(69.5)), @O(@N(DEV_STATE), @R(9.5)), @O(@N(DRV_STAT), @R(29.5)), @O(@N(VSOUT1_STAT), @R(49.5)), @O(@N(WD_FAIL), @R(69.5));
  @C(1378) : @FB(ANLG14), @R(960.0, -210.0, 120.0, 58.0), @I(@N(ADC), @L(9.5)), @I(@N(GRP), @L(29.5)), @I(@N(CH), @L(49.5)), @O(@N(VAL), @R(9.5));
  @C(1379) : @F(GT), @R(1160.0, -210.0, 40.0, 38.0), UINT, @I(@N(IN1), @L(9.5)), @I(@N(IN2), @L(29.5)), @O(@N(GT), @R(9.5));
  @C(1380) : @FB(TON1), @R(1230.0, -210.0, 100.0, 38.0), @I(@N(IN), @L(9.5)), @I(@N(PT), @L(29.5)), @O(@N(Q), @R(9.5)), @O(@N(ET), @R(29.5));
  @C(1381) : @FB(TOF15), @R(1460.0, -210.0, 100.0, 38.0), @I(@N(IN), @L(9.5)), @I(@N(PT), @L(29.5)), @O(@N(Q), @R(9.5)), @O(@N(ET), @R(29.5));
  @VF(1382) : @E(BATTSTACK_DISABLE), @R(1370.0, -40.0, 170.0, 19.0);
  @VF(1383) : @E(CAN_DISABLE), @R(1370.0, -60.0, 170.0, 19.0);
  @VF(1384) : @E(T#1500ms), @R(1370.0, -100.0, 90.0, 19.0);
  @VF(1385) : @E(T#500ms), @R(1110.0, -100.0, 90.0, 19.0);
  @VF(1386) : @E(RDY_TO_SLEEP), @R(1610.0, -120.0, 190.0, 19.0);
  @VF(1387) : @E(IGNITION_KL15), @R(690.0, -120.0, 190.0, 19.0), @ONEG;
  @VF(1392) : @E(7), @R(800.0, -170.0, 110.0, 19.0), USINT;
  @VF(1393) : @E(T#250ms), @R(1100.0, -170.0, 80.0, 19.0);
  @VF(1638) : @E(28), @R(370.0, -90.0, 80.0, 19.0), UINT;
  @VF(1639) : @E(100), @R(1100.0, -190.0, 40.0, 19.0), UINT;
  @VF(1915) : @E(T#800ms), @R(1360.0, -190.0, 80.0, 19.0);
  @VF(1916) : @E(TMSADCGRP#G1), @R(690.0, -190.0, 220.0, 19.0);
  @VF(1917) : @E(TMS570_GIO#HET1), @R(310.0, -110.0, 140.0, 19.0);
  @VF(1918) : @E(T#250ms), @R(220.0, -50.0, 90.0, 19.0);
  @VF(1919) : @E(TMSADC#A1), @R(690.0, -210.0, 220.0, 19.0);
  @VF(1920) : @E(IGNITION_KL15), @R(1580.0, -210.0, 190.0, 19.0);
  @VF(1921) : @E(IGNITION_KL15), @R(120.0, -70.0, 190.0, 19.0);
  @VF(1922) : @E(RDY_TO_SLEEP), @R(90.0, -150.0, 180.0, 19.0);
  @VF(1923) : @E(AN_KL15), @R(1160.0, -230.0, 140.0, 19.0);
  @CF(1924) : @R(690.0, -170.0, 110.0, 19.0), @T("KL15");
  @CF(1925) : @R(490.0, -50.0, 100.0, 19.0), @T("BMSMU LED");
  @C(1957) : @F(EQ), @R(3370.0, 3220.0, 40.0, 38.0), BYTE, @I(@N(IN1), @L(9.5)), @I(@N(IN2), @L(29.5)), @O(@N(EQ), @R(9.5));
  @C(1958) : @F(SEL), @R(3490.0, 3220.0, 120.0, 58.0), BOOL, @I(@N(G), @L(9.5)), @I(@N(IN0), @L(29.5)), @I(@N(IN1), @L(49.5)), @O(@N(SEL), @R(9.5));
  @C(1959) : @FB(IOWR19), @R(3650.0, 3180.0, 120.0, 58.0), @I(@N(PORT), @L(9.5)), @I(@N(PIN), @L(29.5)), @I(@N(VAL), @L(49.5));
  @C(1960) : @FB(IOWR6), @R(190.0, -560.0, 120.0, 58.0), @I(@N(PORT), @L(9.5)), @I(@N(PIN), @L(29.5)), @I(@N(VAL), @L(49.5));
  @C(1961) : @FB(IOWR5), @R(190.0, -640.0, 120.0, 58.0), @I(@N(PORT), @L(9.5)), @I(@N(PIN), @L(29.5)), @I(@N(VAL), @L(49.5));
  @C(1962) : @FB(IOWR18), @R(3650.0, 3520.0, 120.0, 58.0), @I(@N(PORT), @L(9.5)), @I(@N(PIN), @L(29.5)), @I(@N(VAL), @L(49.5));
  @C(1964) : @FB(IOWR20), @R(3650.0, 3580.0, 120.0, 58.0), @I(@N(PORT), @L(9.5)), @I(@N(PIN), @L(29.5)), @I(@N(VAL), @L(49.5));
  @C(1965) : @FB(IOWR21), @R(3650.0, 3650.0, 120.0, 58.0), @I(@N(PORT), @L(9.5)), @I(@N(PIN), @L(29.5)), @I(@N(VAL), @L(49.5));
  @C(1966) : @FB(FLASH4), @R(3500.0, 3690.0, 120.0, 38.0), @I(@N(IN), @L(9.5)), @I(@N(PER), @L(29.5)), @O(@N(OUT), @R(9.5));
  @VF(1967) : @E(1), @R(3280.0, 3240.0, 50.0, 19.0), BYTE;
  @VF(1968) : @E(HW_version), @R(3210.0, 3220.0, 120.0, 19.0);
  @VF(1969) : @E(1), @R(3430.0, 3260.0, 50.0, 19.0), BOOL;
  @VF(1970) : @E(0), @R(3430.0, 3240.0, 50.0, 19.0), BOOL;
  @VF(1971) : @E(TMS570_GIO#SPI2), @R(3380.0, 3180.0, 150.0, 19.0);
  @VF(1972) : @E(10), @R(3470.0, 3200.0, 60.0, 19.0), UINT;
  @VF(1973) : @E(TMS570_GIO#HET1), @R(20.0, -640.0, 140.0, 19.0);
  @VF(1974) : @E(24), @R(100.0, -620.0, 60.0, 19.0), UINT;
  @VF(1975) : @E(1), @R(100.0, -600.0, 60.0, 19.0), BOOL;
  @VF(1976) : @E(TMS570_GIO#SPI3), @R(20.0, -560.0, 140.0, 19.0);
  @VF(2008) : @E(8), @R(100.0, -540.0, 60.0, 19.0), UINT;
  @VF(2009) : @E(1), @R(100.0, -520.0, 60.0, 19.0), BOOL;
  @VF(2119) : @E(TMS570_GIO#SPI2), @R(3490.0, 3520.0, 140.0, 19.0);
  @VF(2120) : @E(0), @R(3570.0, 3540.0, 60.0, 19.0), UINT;
  @VF(2121) : @E(1), @R(3570.0, 3560.0, 60.0, 19.0), BOOL;
  @VF(2122) : @E(TMS570_GIO#SPI2), @R(3490.0, 3580.0, 140.0, 19.0);
  @VF(2123) : @E(11), @R(3570.0, 3600.0, 60.0, 19.0), UINT;
  @VF(2124) : @E(1), @R(3570.0, 3620.0, 60.0, 19.0), BOOL;
  @VF(2125) : @E(TMS570_GIO#SPI2), @R(3490.0, 3650.0, 140.0, 19.0);
  @VF(2126) : @E(9), @R(3570.0, 3670.0, 60.0, 19.0), UINT;
  @VF(2127) : @E(1), @R(3390.0, 3690.0, 60.0, 19.0), BOOL;
  @VF(2128) : @E(T#3s), @R(3390.0, 3710.0, 60.0, 19.0);
  @CF(2129) : @R(110.0, -580.0, 200.0, 19.0), @T("CAN_EN");
  @CF(2131) : @R(100.0, -660.0, 200.0, 19.0), @T("CAN1 enable");
  @CF(2132) : @R(120.0, -500.0, 200.0, 19.0), @T("CAN_STB_N");
  @CF(2136) : @R(3550.0, 3110.0, 210.0, 59.0), @T("BQ comm enb (NOT) for V2$NAnlg4 5V enb for V1");
  @CF(2142) : @R(3460.0, 3540.0, 110.0, 19.0), @T("AIN-1 CTRL");
  @CF(2143) : @R(3460.0, 3600.0, 110.0, 19.0), @T("AIN-2 CTRL");
  @CF(2144) : @R(3400.0, 3740.0, 180.0, 39.0), @T("5V control for V2$NAnlg3 5v enb for V1");
  @C(2223) : @FB(IOWR9), @R(2120.0, 3020.0, 120.0, 58.0), @I(@N(PORT), @L(9.5)), @I(@N(PIN), @L(29.5)), @I(@N(VAL), @L(49.5));
  @C(2224) : @FB(IOWR7), @R(2120.0, 2960.0, 120.0, 58.0), @I(@N(PORT), @L(9.5)), @I(@N(PIN), @L(29.5)), @I(@N(VAL), @L(49.5));
  @C(2225) : @FB(IOWR22), @R(2120.0, 2840.0, 120.0, 58.0), @I(@N(PORT), @L(9.5)), @I(@N(PIN), @L(29.5)), @I(@N(VAL), @L(49.5));
  @C(2226) : @FB(IOWR23), @R(2120.0, 2900.0, 120.0, 58.0), @I(@N(PORT), @L(9.5)), @I(@N(PIN), @L(29.5)), @I(@N(VAL), @L(49.5));
  @C(2227) : @FB(IOWR10), @R(2120.0, 2780.0, 120.0, 58.0), @I(@N(PORT), @L(9.5)), @I(@N(PIN), @L(29.5)), @I(@N(VAL), @L(49.5));
  @C(2228) : @FB(IOWR24), @R(2120.0, 2720.0, 120.0, 58.0), @I(@N(PORT), @L(9.5)), @I(@N(PIN), @L(29.5)), @I(@N(VAL), @L(49.5));
  @VF(2229) : @E(8), @R(2010.0, 3040.0, 60.0, 19.0), UINT;
  @VF(2230) : @E(22), @R(2010.0, 2980.0, 60.0, 19.0), UINT;
  @VF(2231) : @E(7), @R(2010.0, 2860.0, 60.0, 19.0), UINT;
  @VF(2232) : @E(6), @R(2010.0, 2920.0, 60.0, 19.0), UINT;
  @VF(2233) : @E(0), @R(2010.0, 2800.0, 60.0, 19.0), UINT;
  @VF(2234) : @E(2), @R(2010.0, 2740.0, 60.0, 19.0), UINT;
  @VF(2235) : @E(TMS570_GIO#A), @R(1930.0, 2900.0, 140.0, 19.0);
  @VF(2238) : @E(TMS570_GIO#HET1), @R(1930.0, 2960.0, 140.0, 19.0);
  @VF(2239) : @E(TMS570_GIO#A), @R(1930.0, 2840.0, 140.0, 19.0);
  @VF(2240) : @E(TMS570_GIO#HET1), @R(1930.0, 3020.0, 140.0, 19.0);
  @VF(2241) : @E(TMS570_GIO#HET1), @R(1930.0, 2780.0, 140.0, 19.0);
  @VF(2249) : @E(TMS570_GIO#HET1), @R(1930.0, 2720.0, 140.0, 19.0);
  @CF(2250) : @R(1940.0, 3040.0, 70.0, 19.0), @T("out6");
  @CF(2253) : @R(1940.0, 2980.0, 70.0, 19.0), @T("out5");
  @CF(2257) : @R(1940.0, 2920.0, 70.0, 19.0), @T("out4");
  @CF(2259) : @R(1940.0, 2860.0, 70.0, 19.0), @T("out3");
  @CF(2260) : @R(1940.0, 2800.0, 70.0, 19.0), @T("out2");
  @CF(2261) : @R(1940.0, 2740.0, 70.0, 19.0), @T("out1");
  @C(200) : @FB(ANLG4), @R(2120.0, 3670.0, 120.0, 58.0), @I(@N(ADC), @L(9.5)), @I(@N(GRP), @L(29.5)), @I(@N(CH), @L(49.5)), @O(@N(VAL), @R(9.5));
  @C(240) : @FB(ANLG3), @R(2120.0, 3610.0, 120.0, 58.0), @I(@N(ADC), @L(9.5)), @I(@N(GRP), @L(29.5)), @I(@N(CH), @L(49.5)), @O(@N(VAL), @R(9.5));
  @C(452) : @FB(ANLG1), @R(2120.0, 3490.0, 120.0, 58.0), @I(@N(ADC), @L(9.5)), @I(@N(GRP), @L(29.5)), @I(@N(CH), @L(49.5)), @O(@N(VAL), @R(9.5));
  @C(471) : @FB(ANLG2), @R(2120.0, 3550.0, 120.0, 58.0), @I(@N(ADC), @L(9.5)), @I(@N(GRP), @L(29.5)), @I(@N(CH), @L(49.5)), @O(@N(VAL), @R(9.5));
  @VF(487) : @E(6), @R(2020.0, 3530.0, 60.0, 19.0), USINT;
  @VF(1438) : @E(TMSADCGRP#G1), @R(1940.0, 3510.0, 140.0, 19.0);
  @VF(491) : @E(5), @R(2020.0, 3590.0, 60.0, 19.0), USINT;
  @VF(705) : @E(TMSADC#A1), @R(1940.0, 3490.0, 140.0, 19.0);
  @VF(707) : @E(8), @R(2020.0, 3650.0, 60.0, 19.0), USINT;
  @VF(1444) : @E(11), @R(2020.0, 3710.0, 60.0, 19.0), USINT;
  @CF(708) : @R(1940.0, 3530.0, 70.0, 19.0), @T("AIN-1");
  @CF(710) : @R(1940.0, 3590.0, 70.0, 19.0), @T("AIN-2");
  @CF(712) : @R(1940.0, 3650.0, 70.0, 19.0), @T("AIN-3");
  @CF(716) : @R(1940.0, 3710.0, 70.0, 19.0), @T("AIN-4");
  @C(1018) : @FB(IORD5), @R(2120.0, 3330.0, 120.0, 38.0), @I(@N(PORT), @L(9.5)), @I(@N(PIN), @L(29.5)), @O(@N(OUT), @R(9.5));
  @C(1340) : @FB(IORD4), @R(2120.0, 3290.0, 120.0, 38.0), @I(@N(PORT), @L(9.5)), @I(@N(PIN), @L(29.5)), @O(@N(OUT), @R(9.5));
  @C(1341) : @FB(IORD1), @R(2120.0, 3250.0, 120.0, 38.0), @I(@N(PORT), @L(9.5)), @I(@N(PIN), @L(29.5)), @O(@N(OUT), @R(9.5));
  @C(1350) : @FB(dgtIn8), @R(2090.0, 3230.0, 150.0, 18.0), @I(@N(ch), @L(9.5)), @O(@N(stat), @R(9.5));
  @C(1361) : @FB(dgtIn3), @R(2090.0, 3210.0, 150.0, 18.0), @I(@N(ch), @L(9.5)), @O(@N(stat), @R(9.5));
  @C(1362) : @FB(dgtIn4), @R(2090.0, 3190.0, 150.0, 18.0), @I(@N(ch), @L(9.5)), @O(@N(stat), @R(9.5));
  @C(1388) : @FB(IORD2), @R(2120.0, 3370.0, 120.0, 38.0), @I(@N(PORT), @L(9.5)), @I(@N(PIN), @L(29.5)), @O(@N(OUT), @R(9.5));
  @C(1397) : @FB(IORD3), @R(2120.0, 3410.0, 120.0, 38.0), @I(@N(PORT), @L(9.5)), @I(@N(PIN), @L(29.5)), @O(@N(OUT), @R(9.5));
  @VF(1398) : @E(4), @R(2020.0, 3230.0, 60.0, 19.0), USINT;
  @VF(1439) : @E(3), @R(2020.0, 3210.0, 60.0, 19.0), USINT;
  @VF(1440) : @E(2), @R(2020.0, 3190.0, 60.0, 19.0), USINT;
  @VF(1442) : @E(TMS570_GIO#HET1), @R(1940.0, 3250.0, 140.0, 19.0);
  @VF(1443) : @E(12), @R(2020.0, 3270.0, 60.0, 19.0), UINT;
  @VF(2264) : @E(TMS570_GIO#HET1), @R(1940.0, 3290.0, 140.0, 19.0);
  @VF(2287) : @E(16), @R(2020.0, 3310.0, 60.0, 19.0), UINT;
  @VF(2291) : @E(TMS570_GIO#HET1), @R(1940.0, 3330.0, 140.0, 19.0);
  @VF(2292) : @E(14), @R(2020.0, 3350.0, 60.0, 19.0), UINT;
  @VF(2293) : @E(TMS570_GIO#HET1), @R(1940.0, 3370.0, 140.0, 19.0);
  @VF(2294) : @E(18), @R(2020.0, 3390.0, 60.0, 19.0), UINT;
  @VF(2295) : @E(TMS570_GIO#HET1), @R(1940.0, 3410.0, 140.0, 19.0);
  @VF(2296) : @E(17), @R(2020.0, 3430.0, 60.0, 19.0), UINT;
  @CF(2297) : @R(1940.0, 3190.0, 80.0, 19.0), @T("DIN-1");
  @CF(2298) : @R(1940.0, 3270.0, 80.0, 19.0), @T("DIN-4");
  @CF(2299) : @R(1940.0, 3230.0, 80.0, 19.0), @T("DIN-3");
  @CF(2300) : @R(1940.0, 3210.0, 80.0, 19.0), @T("DIN-2");
  @CF(2301) : @R(1940.0, 3310.0, 80.0, 19.0), @T("DIN-5");
  @CF(2302) : @R(1940.0, 3350.0, 80.0, 19.0), @T("DIN-6");
  @CF(2303) : @R(1940.0, 3390.0, 80.0, 19.0), @T("DIN-7");
  @CF(2304) : @R(1940.0, 3430.0, 80.0, 19.0), @T("DIN-8");
  @VF(139) : @E(TMSADC#A1), @R(1940.0, 3550.0, 140.0, 19.0);
  @VF(140) : @E(TMSADCGRP#G1), @R(1940.0, 3570.0, 140.0, 19.0);
  @VF(145) : @E(TMSADC#A1), @R(1940.0, 3610.0, 140.0, 19.0);
  @VF(147) : @E(TMSADCGRP#G1), @R(1940.0, 3630.0, 140.0, 19.0);
  @VF(148) : @E(TMSADC#A1), @R(1940.0, 3670.0, 140.0, 19.0);
  @VF(150) : @E(TMSADCGRP#G1), @R(1940.0, 3690.0, 140.0, 19.0);
  @C(223) : @F(OR), @R(330.0, 1650.0, 40.0, 38.0), BOOL, @I(@N(IN1), @L(9.5)), @I(@N(IN2), @L(29.5)), @O(@N(OR), @R(9.5));
  @C(226) : @FB(F_TRIG2), @R(180.0, 1670.0, 140.0, 18.0), @I(@N(CLK), @L(9.5)), @O(@N(Q), @R(9.5));
  @VF(232) : @E(IGNITION_KL15), @R(30.0, 1670.0, 130.0, 19.0);
  @C(1427) : @FB(NTC2), @R(2430.0, 3490.0, 120.0, 118.0), @I(@N(VOLT), @L(9.5)), @I(@N(VSUP), @L(29.5)), @I(@N(RS), @L(49.5)), @I(@N(BETA), @L(69.5)), @I(@N(TNOM), @L(89.5)), @I(@N(RNOM), @L(109.5)), @O(@N(TEMP), @R(9.5));
  @VF(1467) : @E(Pack_Temperature), @R(2570.0, 3490.0, 150.0, 19.0);
  @VF(1456) : @E(298.15), @R(2330.0, 3570.0, 80.0, 19.0), REAL;
  @VF(1457) : @E(10000), @R(2330.0, 3530.0, 80.0, 19.0), REAL;
  @VF(1458) : @E(7000), @R(2330.0, 3510.0, 80.0, 19.0), REAL;
  @VF(1459) : @E(3950), @R(2330.0, 3550.0, 80.0, 19.0), REAL;
  @VF(1460) : @E(10000), @R(2330.0, 3590.0, 80.0, 19.0), REAL;
  @VF(469) : @E(1), @R(2340.0, 3370.0, 60.0, 19.0), BOOL;
  @C(43) : @F(DIV), @R(740.0, 2930.0, 40.0, 38.0), REAL, @I(@N(IN1), @L(9.5)), @I(@N(IN2), @L(29.5)), @O(@N(DIV), @R(9.5));
  @VF(46) : @E(emergencyBtn), @R(1900.0, 290.0, 140.0, 19.0);
  @VF(239) : @E(contactEnable_batt), @R(430.0, 2370.0, 190.0, 19.0);
  @VF(448) : @E(contactNegEnable_batt), @R(430.0, 2390.0, 190.0, 19.0);
  @VF(756) : @E(new_CHG_CONTACT), @R(720.0, 2370.0, 160.0, 19.0);
  @VF(759) : @E(new_DCHG_CONTACT), @R(720.0, 2390.0, 160.0, 19.0);
  @VF(747) : @E(DischargeInVoltage), @R(800.0, 2930.0, 140.0, 19.0);
  @C(833) : @F(OR), @R(2780.0, 3580.0, 40.0, 38.0), BOOL, @I(@N(IN1), @L(9.5)), @I(@N(IN2), @L(29.5)), @O(@N(OR), @R(9.5));
  @VF(834) : @E(contactFbk), @R(2830.0, 3580.0, 150.0, 19.0);
  @VF(837) : @E(contactFbkCharge), @R(2620.0, 3580.0, 140.0, 19.0);
  @VF(844) : @E(contactFbkDischarge), @R(2620.0, 3600.0, 140.0, 19.0);
  @VF(853) : @E(Number_Of_MaxCell), @R(20.0, 1030.0, 140.0, 19.0);
  @C(1002) : @F(TO_USINT), @R(180.0, 1030.0, 120.0, 18.0), UINT, @I(@N(IN), @L(9.5)), @O(@N(TO_USINT), @R(9.5));
  @C(804) : @FB(ARR2VAL2), @R(1070.0, 1130.0, 200.0, 78.0), @I(@N(MaxBMU), @L(9.5)), @I(@N(indx), @L(29.5)), @I(@N(Map), @L(49.5)), @I(@N(CellCounter), @L(69.5)), @O(@N(numofCell), @R(9.5)), @O(@N(Reset), @R(29.5));
  @VF(1007) : @E(Selected_Cell_Loc), @R(920.0, 1190.0, 140.0, 19.0);
  @VF(1009) : @E(NumOfCells), @R(920.0, 1170.0, 140.0, 19.0);
  @VF(1010) : @E(Selected_BMU_Loc), @R(920.0, 1150.0, 140.0, 19.0);
  @VF(1011) : @E(Number_Of_MaxCell), @R(1280.0, 1130.0, 140.0, 19.0);
  @VF(1062) : @E(NEWBMU_RESET), @R(1280.0, 1150.0, 140.0, 19.0);
  @VF(1063) : @E(Number_Of_BMU_cfg), @R(920.0, 1130.0, 140.0, 19.0);
  @VF(231) : @E(NEWBMU_RESET), @R(380.0, 920.0, 140.0, 19.0);
  @VF(359) : @E(contactFbkCharge), @R(150.0, 2150.0, 140.0, 19.0);
  @C(3226) : @FB(prechargeCAN1), @R(1450.0, 1880.0, 250.0, 118.0), @I(@N(CAN_CH), @L(9.5)), @I(@N(ENB), @L(29.5)), @I(@N(RST), @L(49.5), @NEG), @O(@N(CANerr), @R(9.5)), @O(@N(outFbk), @R(29.5)), @O(@N(igbtFlt), @R(49.5)), @O(@N(igbtRdy), @R(69.5)), @O(@N(igbtRst), @R(89.5)), @O(@N(inVal), @R(109.5));
  @VF(3241) : @E(PDUCAN), @R(1330.0, 1880.0, 80.0, 19.0);
  @VF(3239) : @E(prechargeEnable), @R(1210.0, 1900.0, 140.0, 19.0);
  @VF(3249) : @E(prechargeBoardErr), @R(1710.0, 1880.0, 170.0, 19.0);
  @C(3224) : @F(TO_TIME), @R(1230.0, 2160.0, 120.0, 18.0), UDINT, @I(@N(IN), @L(9.5)), @O(@N(TO_TIME), @R(9.5));
  @C(3229) : @F(ABS), @R(1300.0, 2240.0, 60.0, 18.0), REAL, @I(@N(IN), @L(9.5)), @O(@N(ABS), @R(9.5));
  @C(3225) : @F(DIV_TIME), @R(1380.0, 2160.0, 40.0, 38.0), UINT, @I(@N(IN1), @L(9.5)), @I(@N(IN2), @L(29.5)), @O(@N(DIV_TIME), @R(9.5));
  @C(3228) : @F(GT), @R(1380.0, 2200.0, 40.0, 38.0), REAL, @I(@N(IN1), @L(9.5)), @I(@N(IN2), @L(29.5)), @O(@N(GT), @R(9.5));
  @C(3231) : @F(SUB), @R(1160.0, 2240.0, 40.0, 38.0), REAL, @I(@N(IN1), @L(9.5)), @I(@N(IN2), @L(29.5)), @O(@N(SUB), @R(9.5));
  @C(3232) : @F(LT), @R(1380.0, 2240.0, 40.0, 38.0), REAL, @I(@N(IN1), @L(9.5)), @I(@N(IN2), @L(29.5)), @O(@N(LT), @R(9.5));
  @C(3233) : @F(GT), @R(1380.0, 2280.0, 40.0, 38.0), REAL, @I(@N(IN1), @L(9.5)), @I(@N(IN2), @L(29.5)), @O(@N(GT), @R(9.5));
  @C(3230) : @FB(TON26), @R(1500.0, 2240.0, 100.0, 38.0), @I(@N(IN), @L(9.5)), @I(@N(PT), @L(29.5)), @O(@N(Q), @R(9.5)), @O(@N(ET), @R(29.5));
  @C(3235) : @F(ABS), @R(1300.0, 2320.0, 60.0, 18.0), REAL, @I(@N(IN), @L(9.5)), @O(@N(ABS), @R(9.5));
  @C(3227) : @F(AND), @R(1630.0, 2200.0, 40.0, 38.0), BOOL, @I(@N(IN1), @L(9.5)), @I(@N(IN2), @L(29.5)), @O(@N(AND), @R(9.5));
  @C(3234) : @F(AND), @R(1630.0, 2280.0, 40.0, 38.0), BOOL, @I(@N(IN1), @L(9.5)), @I(@N(IN2), @L(29.5)), @O(@N(AND), @R(9.5));
  @C(3238) : @FB(TON27), @R(1500.0, 2320.0, 100.0, 38.0), @I(@N(IN), @L(9.5)), @I(@N(PT), @L(29.5)), @O(@N(Q), @R(9.5)), @O(@N(ET), @R(29.5));
  @C(3237) : @F(LT), @R(1380.0, 2320.0, 40.0, 38.0), REAL, @I(@N(IN1), @L(9.5)), @I(@N(IN2), @L(29.5)), @O(@N(LT), @R(9.5));
  @C(3236) : @F(SUB), @R(1160.0, 2320.0, 40.0, 38.0), REAL, @I(@N(IN1), @L(9.5)), @I(@N(IN2), @L(29.5)), @O(@N(SUB), @R(9.5));
  @VF(3243) : @E(1000), @R(1150.0, 2180.0, 60.0, 19.0), UINT;
  @VF(3242) : @E(prechargeInterval), @R(1050.0, 2160.0, 160.0, 19.0);
  @VF(3244) : @E(Pack_CutoffLow_Voltage), @R(1160.0, 2220.0, 190.0, 19.0);
  @VF(3245) : @E(BatteryVoltage), @R(990.0, 2240.0, 150.0, 19.0);
  @VF(3247) : @E(8), @R(1320.0, 2260.0, 40.0, 19.0), REAL;
  @VF(3246) : @E(OutputVoltage), @R(990.0, 2260.0, 150.0, 19.0);
  @VF(3250) : @E(Pack_CutoffLow_Voltage), @R(1170.0, 2300.0, 190.0, 19.0);
  @VF(3252) : @E(BatteryVoltage), @R(990.0, 2320.0, 150.0, 19.0);
  @VF(3254) : @E(ChargeInVoltage), @R(990.0, 2340.0, 150.0, 19.0);
  @VF(3253) : @E(8), @R(1320.0, 2340.0, 40.0, 19.0), REAL;
  @VF(3248) : @E(prechargeComplete), @R(1690.0, 2200.0, 180.0, 19.0);
  @VF(3251) : @E(prechargeCompleteCharge), @R(1690.0, 2280.0, 200.0, 19.0);
  @VF(237) : @E(new_DCHG_CONTACT), @R(1930.0, 2760.0, 140.0, 19.0);
  @VF(236) : @E(new_CHG_CONTACT), @R(1930.0, 2820.0, 140.0, 19.0);
  @C(850) : @F(EQ), @R(2270.0, 3170.0, 40.0, 38.0), USINT, @I(@N(IN1), @L(9.5)), @I(@N(IN2), @L(29.5)), @O(@N(EQ), @R(9.5));
  @C(175) : @F(EQ), @R(2270.0, 3210.0, 40.0, 38.0), USINT, @I(@N(IN1), @L(9.5)), @I(@N(IN2), @L(29.5)), @O(@N(EQ), @R(9.5));
  @VF(310) : @E(1), @R(2110.0, 3120.0, 130.0, 19.0), USINT;
  @VF(722) : @E(contactFbkDischarge), @R(2320.0, 3170.0, 140.0, 19.0);
  @VF(723) : @E(contactFbkCharge), @R(2320.0, 3210.0, 140.0, 19.0);
  @VF(196) : @E(contactEnable_batt), @R(3280.0, 870.0, 160.0, 19.0);
  @VF(811) : @E(contactEnable_batt), @R(1030.0, 2080.0, 190.0, 19.0);
  @VF(821) : @E(contactNegEnable_batt), @R(1030.0, 2100.0, 190.0, 19.0);
  @C(908) : @F(OR), @R(1240.0, 2080.0, 40.0, 38.0), BOOL, @I(@N(IN1), @L(9.5)), @I(@N(IN2), @L(29.5)), @O(@N(OR), @R(9.5));
  @VF(1074) : @E(AllcontacstEnable), @R(1300.0, 2080.0, 140.0, 19.0);
  @VF(662) : @E(AllcontacstEnable), @R(3280.0, 750.0, 140.0, 19.0);
  @VF(1076) : @E(prechargeBoardErr), @R(2040.0, 290.0, 140.0, 19.0);
  @C(1083) : @F(AND), @R(1380.0, 1920.0, 40.0, 38.0), BOOL, @I(@N(IN1), @L(9.5)), @I(@N(IN2), @L(29.5)), @O(@N(AND), @R(9.5));
  @VF(1086) : @E(prechargeBoardErr), @R(1190.0, 1940.0, 170.0, 19.0), @ONEG;
  @C(1082) : @F(SEL), @R(1110.0, 2480.0, 120.0, 58.0), BOOL, @I(@N(G), @L(9.5)), @I(@N(IN0), @L(29.5)), @I(@N(IN1), @L(49.5)), @O(@N(SEL), @R(9.5));
  @C(14) : @FB(GUICFG_INT1), @R(70.0, 10.0, 180.0, 38.0), @I(@N(CODE), @L(9.5)), @I(@N(R), @L(29.5)), @O(@N(VAL), @R(9.5));
  @C(1079) : @F(TO_USINT), @R(270.0, 10.0, 120.0, 18.0), DINT, @I(@N(IN), @L(9.5)), @O(@N(TO_USINT), @R(9.5));
  @VF(410) : @E(Cell_Temp_Min), @R(1960.0, 150.0, 220.0, 19.0);
  @CP(467) : 2199.5, 59.5;
  @CP(1326) : 2199.5, 359.5;
  @CP(640) : 2199.5, 519.5;
  @CP(1521) : 719.5, 2799.5;
  @CP(1584) : 2089.5, 1799.5;
  @CP(1579) : 2089.5, 1719.5;
  @CP(1589) : 2089.5, 1889.5;
  @CP(1590) : 2069.5, 1909.5;
  @CP(1664) : 2089.5, 1989.5;
  @CP(1601) : 2069.5, 2009.5;
  @CP(399) : 1609.5, 1579.5;
  @CP(477) : 639.5, 679.5;
  @CP(787) : 459.5, 979.5;
  @CP(1714) : 3199.5, 379.5;
  @CP(194) : 339.5, 1189.5;
  @CP(135) : 749.5, 1619.5;
  @CP(138) : 3339.5, 379.5;
  @CP(1223) : 3119.5, 2489.5;
  @CP(823) : 119.5, 2729.5;
  @CP(365) : 3299.5, 419.5;
  @CP(1914) : 319.5, 999.5;
  @CP(176) : 2149.5, 1449.5;
  @CP(957) : 2149.5, 1619.5;
  @CP(2269) : 3029.5, 59.5;
  @CP(88) : 4069.5, 649.5;
  @CP(1655) : 4139.5, 899.5;
  @CP(2193) : 3449.5, 739.5;
  @CP(1884) : 789.5, 2889.5;
  @CP(2635) : 4299.5, 879.5;
  @CP(2606) : 4049.5, 79.5;
  @CP(1040) : 4519.5, 179.5;
  @CP(1041) : 4529.5, 319.5;
  @CP(2366) : 4149.5, 179.5;
  @CP(2373) : 4149.5, 319.5;
  @CP(1000) : 749.5, 1599.5;
  @CP(382) : 3529.5, 39.5;
  @CP(738) : 219.5, 3609.5;
  @CP(1811) : 229.5, 3839.5;
  @CP(1846) : 889.5, 3509.5;
  @CP(1866) : 899.5, 3739.5;
  @CP(353) : 2199.5, 699.5;
  @CP(1926) : 1349.5, -110.5;
  @CP(1927) : 1119.5, -200.5;
  @CP(3256) : 1149.5, 2249.5;
  @CP(3257) : 1479.5, 2269.5;
  @CP(3258) : 1149.5, 2329.5;
  @CP(436) : 2259.5, 3149.5;
  @CP(776) : 1359.5, 1909.5;
